	NOP 0
	NOP 0
	NOP 0
	NOP 0
	NOP 0
	NOP 0
	NOP 0
	NOP 0
	NOP 0
	NOP 0
	NOP 0
	NOP 0
	NOP 0
	NOP 0
	NOP 0
	NOP 0
	NOP 0
	NOP 0
	NOP 0
	NOP 0
	NOP 0
	NOP 0
	NOP 0
	NOP 0
	NOP 0
	NOP 0
	NOP 0
	NOP 0
	NOP 0
	NOP 0
	NOP 0
	NOP 0
	NOP 0
	NOP 0
	NOP 0
	NOP 0
	NOP 0
	NOP 0
	NOP 0
	NOP 0
	NOP 0
	NOP 0
	NOP 0
	NOP 0
	NOP 0
	NOP 0
	NOP 0
	NOP 0
	NOP 0
	NOP 0
	NOP 0
	NOP 0
	NOP 0
	NOP 0
	NOP 0
	NOP 0
	NOP 0
	NOP 0
	NOP 0
	NOP 0
	NOP 0
	NOP 0
	NOP 0
	NOP 0
	NOP 0
	NOP 0
	NOP 0
	NOP 0
	NOP 0
	NOP 0
	NOP 0
	NOP 0
	NOP 0
	NOP 0
	NOP 0
	NOP 0
	NOP 0
	NOP 0
	NOP 0
	NOP 0
	NOP 0
	NOP 0
	NOP 0
	NOP 0
	NOP 0
	NOP 0
	NOP 0
	NOP 0
	NOP 0
	NOP 0
	NOP 0
	NOP 0
	NOP 0
	NOP 0
	NOP 0
	NOP 0
	NOP 0
	NOP 0
	NOP 0
	NOP 0
	NOP 0
	NOP 0
	NOP 0
	NOP 0
	NOP 0
	NOP 0
	NOP 0
	NOP 0
	NOP 0
	NOP 0
	NOP 0
	NOP 0
	NOP 0
	NOP 0
	NOP 0
	NOP 0
	NOP 0
	NOP 0
	NOP 0
	NOP 0
	NOP 0
	NOP 0
	NOP 0
	NOP 0
	NOP 0
	NOP 0
	NOP 0
	NOP 0
	NOP 0
	NOP 0
	NOP 0
	NOP 0
	NOP 0
	NOP 0
	NOP 0
	NOP 0
	NOP 0
	NOP 0
	NOP 0
	NOP 0
	NOP 0
	NOP 0
	NOP 0
	NOP 0
	NOP 0
	NOP 0
	NOP 0
	NOP 0
	NOP 0
	NOP 0
	NOP 0
	NOP 0
	NOP 0
	NOP 0
	NOP 0
	NOP 0
	NOP 0
	NOP 0
	NOP 0
	NOP 0
	NOP 0
	NOP 0
	NOP 0
	NOP 0
	NOP 0
	NOP 0
	NOP 0
	NOP 0
	NOP 0
	NOP 0
	NOP 0
	NOP 0
	NOP 0
	NOP 0
	NOP 0
	NOP 0
	NOP 0
	NOP 0
	NOP 0
	NOP 0
	NOP 0
	NOP 0
	NOP 0
	NOP 0
	NOP 0
	NOP 0
	NOP 0
	NOP 0
	NOP 0
	NOP 0
	NOP 0
	NOP 0
	NOP 0
	NOP 0
	NOP 0
	NOP 0
	NOP 0
	NOP 0
	NOP 0
	NOP 0
	NOP 0
	NOP 0
	NOP 0
	NOP 0
	NOP 0
	NOP 0
	NOP 0
	NOP 0
	NOP 0
	NOP 0
	NOP 0
	NOP 0
	NOP 0
	NOP 0
	NOP 0
	NOP 0
	NOP 0
	NOP 0
	NOP 0
	NOP 0
	NOP 0
	NOP 0
	NOP 0
	NOP 0
	NOP 0
	NOP 0
	NOP 0
	NOP 0
	NOP 0
	NOP 0
	NOP 0
	NOP 0
	NOP 0
	NOP 0
	NOP 0
	NOP 0
	NOP 0
	NOP 0
	NOP 0
	NOP 0
	NOP 0
	NOP 0
	NOP 0
	NOP 0
	NOP 0
	NOP 0
	NOP 0
	NOP 0
	NOP 0
	NOP 0
	NOP 0
	NOP 0
	NOP 0
	NOP 0
	NOP 0
	NOP 0
	NOP 0
	NOP 0
	NOP 0
	NOP 0
	NOP 0
	NOP 0
	NOP 0
	NOP 0
	NOP 0
	NOP 0
	NOP 0
	NOP 0
	NOP 0
	NOP 0
	NOP 0
	NOP 0
	NOP 0
	NOP 0
	NOP 0
	NOP 0
	NOP 0
	NOP 0
	NOP 0
	NOP 0
	NOP 0
	NOP 0
	NOP 0
	NOP 0
	NOP 0
	NOP 0
	NOP 0
	NOP 0
	NOP 0
	NOP 0
	NOP 0
	NOP 0
	NOP 0
	NOP 0
	NOP 0
	NOP 0
	NOP 0
	NOP 0
	NOP 0
	NOP 0
	NOP 0
	NOP 0
	NOP 0
	NOP 0
	NOP 0
	NOP 0
	NOP 0
	NOP 0
	NOP 0
	NOP 0
	NOP 0
	NOP 0
	NOP 0
	NOP 0
	NOP 0
	NOP 0
	NOP 0
	NOP 0
	NOP 0
	NOP 0
	NOP 0
	NOP 0
	NOP 0
	NOP 0
	NOP 0
	NOP 0
	NOP 0
	NOP 0
	NOP 0
	NOP 0
	NOP 0
	NOP 0
	NOP 0
	NOP 0
	NOP 0
	NOP 0
	NOP 0
	NOP 0
	NOP 0
	NOP 0
	NOP 0
	NOP 0
	NOP 0
	NOP 0
	NOP 0
	NOP 0
	NOP 0
	NOP 0
	NOP 0
	NOP 0
	NOP 0
	NOP 0
	NOP 0
	NOP 0
	NOP 0
	NOP 0
	NOP 0
	NOP 0
	NOP 0
	NOP 0
	NOP 0
	NOP 0
	NOP 0
	NOP 0
	NOP 0
	NOP 0
	NOP 0
	NOP 0
	NOP 0
	NOP 0
	NOP 0
	NOP 0
	NOP 0
	NOP 0
	NOP 0
	NOP 0
	NOP 0
	NOP 0
	NOP 0
	NOP 0
	NOP 0
	NOP 0
	NOP 0
	NOP 0
	NOP 0
	NOP 0
	NOP 0
	NOP 0
	NOP 0
	NOP 0
	NOP 0
	NOP 0
	NOP 0
	NOP 0
	NOP 0
	NOP 0
	NOP 0
	NOP 0
	NOP 0
	NOP 0
	NOP 0
	NOP 0
	NOP 0
	NOP 0
	NOP 0
	NOP 0
	NOP 0
	NOP 0
	NOP 0
	NOP 0
	NOP 0
	NOP 0
	NOP 0
	NOP 0
	NOP 0
	NOP 0
	NOP 0
	NOP 0
	NOP 0
	NOP 0
	NOP 0
	NOP 0
	NOP 0
	NOP 0
	NOP 0
	NOP 0
	NOP 0
	NOP 0
	NOP 0
	NOP 0
	NOP 0
	NOP 0
	NOP 0
	NOP 0
	NOP 0
	NOP 0
	NOP 0
	NOP 0
	NOP 0
	NOP 0
	NOP 0
	NOP 0
	NOP 0
	NOP 0
	NOP 0
	NOP 0
	NOP 0
	NOP 0
	NOP 0
	NOP 0
	NOP 0
	NOP 0
	NOP 0
	NOP 0
	NOP 0
	NOP 0
	NOP 0
	NOP 0
	NOP 0
	NOP 0
	NOP 0
	NOP 0
	NOP 0
	NOP 0
	NOP 0
	NOP 0
	NOP 0
	NOP 0
	NOP 0
	NOP 0
	NOP 0
	NOP 0
	NOP 0
	NOP 0
	NOP 0
	NOP 0
	NOP 0
	NOP 0
	NOP 0
	NOP 0
	NOP 0
	NOP 0
	NOP 0
	NOP 0
	NOP 0
	NOP 0
	NOP 0
	NOP 0
	NOP 0
	NOP 0
	NOP 0
	NOP 0
	NOP 0
	NOP 0
	NOP 0
	NOP 0
	NOP 0
	NOP 0
	NOP 0
	NOP 0
	NOP 0
	NOP 0
	NOP 0
	NOP 0
	NOP 0
	NOP 0
	NOP 0
	NOP 0
	NOP 0
	NOP 0
	NOP 0
	NOP 0
	NOP 0
	NOP 0
	NOP 0
	NOP 0
	NOP 0
	NOP 0
	NOP 0
	NOP 0
	NOP 0
	NOP 0
	NOP 0
	NOP 0
	NOP 0
	NOP 0
	NOP 0
	NOP 0
	NOP 0
	NOP 0
	NOP 0
	NOP 0
	NOP 0
	NOP 0
	NOP 0
	NOP 0
	NOP 0
	NOP 0
	NOP 0
	NOP 0
	NOP 0
	NOP 0
	NOP 0
	NOP 0
	NOP 0
	NOP 0
	NOP 0
	NOP 0
	NOP 0
	NOP 0
	NOP 0
	NOP 0
	NOP 0
	NOP 0
	NOP 0
	NOP 0
	NOP 0
	NOP 0
	NOP 0
	NOP 0
	NOP 0
	NOP 0
	NOP 0
	NOP 0
	NOP 0
	NOP 0
	NOP 0
	NOP 0
	NOP 0
	NOP 0
	NOP 0
	NOP 0
	NOP 0
	NOP 0
	NOP 0
	NOP 0
	NOP 0
	NOP 0
	NOP 0
	NOP 0
	NOP 0
	NOP 0
	NOP 0
	NOP 0
	NOP 0
	NOP 0
	NOP 0
	NOP 0
	NOP 0
	NOP 0
	NOP 0
	NOP 0
	NOP 0
	NOP 0
	NOP 0
	NOP 0
	NOP 0
	NOP 0
	NOP 0
	NOP 0
	NOP 0
	NOP 0
	NOP 0
	NOP 0
	NOP 0
	NOP 0
	NOP 0
	NOP 0
	NOP 0
	NOP 0
	NOP 0
	NOP 0
	NOP 0
	NOP 0
	NOP 0
	NOP 0
	NOP 0
	NOP 0
	NOP 0
	NOP 0
	NOP 0
	NOP 0
	NOP 0
	NOP 0
	NOP 0
	NOP 0
	NOP 0
	NOP 0
	NOP 0
	NOP 0
	NOP 0
	NOP 0
	NOP 0
	NOP 0
	NOP 0
	NOP 0
	NOP 0
	NOP 0
	NOP 0
	NOP 0
	NOP 0
	NOP 0
	NOP 0
	NOP 0
	NOP 0
	NOP 0
	NOP 0
	NOP 0
	NOP 0
	NOP 0
	NOP 0
	NOP 0
	NOP 0
	NOP 0
	NOP 0
	NOP 0
	NOP 0
	NOP 0
	NOP 0
	NOP 0
	NOP 0
	NOP 0
	NOP 0
	NOP 0
	NOP 0
	NOP 0
	NOP 0
	NOP 0
	NOP 0
	NOP 0
	NOP 0
	NOP 0
	NOP 0
	NOP 0
	NOP 0
	NOP 0
	NOP 0
	NOP 0
	NOP 0
	NOP 0
	NOP 0
	NOP 0
	NOP 0
	NOP 0
	NOP 0
	NOP 0
	NOP 0
	NOP 0
	NOP 0
	NOP 0
	NOP 0
	NOP 0
	NOP 0
	NOP 0
	NOP 0
	NOP 0
	NOP 0
	NOP 0
	NOP 0
	NOP 0
	NOP 0
	NOP 0
	NOP 0
	NOP 0
	NOP 0
	NOP 0
	NOP 0
	NOP 0
	NOP 0
	NOP 0
	NOP 0
	NOP 0
	NOP 0
	NOP 0
	NOP 0
	NOP 0
	NOP 0
	NOP 0
	NOP 0
	NOP 0
	NOP 0
	NOP 0
	NOP 0
	NOP 0
	NOP 0
	NOP 0
	NOP 0
	NOP 0
	NOP 0
	NOP 0
	NOP 0
	NOP 0
	NOP 0
	NOP 0
	NOP 0
	NOP 0
	NOP 0
	NOP 0
	NOP 0
	NOP 0
	NOP 0
	NOP 0
	NOP 0
	NOP 0
	NOP 0
	NOP 0
	NOP 0
	NOP 0
	NOP 0
	NOP 0
	NOP 0
	NOP 0
	NOP 0
	NOP 0
	NOP 0
	NOP 0
	NOP 0
	NOP 0
	NOP 0
	NOP 0
	NOP 0
	NOP 0
	NOP 0
	NOP 0
	NOP 0
	NOP 0
	NOP 0
	NOP 0
	NOP 0
	NOP 0
	NOP 0
	NOP 0
	NOP 0
	NOP 0
	NOP 0
	NOP 0
	NOP 0
	NOP 0
	NOP 0
	NOP 0
	NOP 0
	NOP 0
	NOP 0
	NOP 0
	NOP 0
	NOP 0
	NOP 0
	NOP 0
	NOP 0
	NOP 0
	NOP 0
	NOP 0
	NOP 0
	NOP 0
	NOP 0
	NOP 0
	NOP 0
	NOP 0
	NOP 0
	NOP 0
	NOP 0
	NOP 0
	NOP 0
	NOP 0
	NOP 0
	NOP 0
	NOP 0
	NOP 0
	NOP 0
	NOP 0
	NOP 0
	NOP 0
	NOP 0
	NOP 0
	NOP 0
	NOP 0
	NOP 0
	NOP 0
	NOP 0
	NOP 0
	NOP 0
	NOP 0
	NOP 0
	NOP 0
	NOP 0
	NOP 0
	NOP 0
	NOP 0
	NOP 0
	NOP 0
	NOP 0
	NOP 0
	NOP 0
	NOP 0
	NOP 0
	NOP 0
	NOP 0
	NOP 0
	NOP 0
	NOP 0
	NOP 0
	NOP 0
	NOP 0
	NOP 0
	NOP 0
	NOP 0
	NOP 0
	NOP 0
	NOP 0
	NOP 0
	NOP 0
	NOP 0
	NOP 0
	NOP 0
	NOP 0
	NOP 0
	NOP 0
	NOP 0
	NOP 0
	NOP 0
	NOP 0
	NOP 0
	NOP 0
	NOP 0
	NOP 0
	NOP 0
	NOP 0
	NOP 0
	NOP 0
	NOP 0
	NOP 0
	NOP 0
	NOP 0
	NOP 0
	NOP 0
	NOP 0
	NOP 0
	NOP 0
	NOP 0
	NOP 0
	NOP 0
	NOP 0
	NOP 0
	NOP 0
	NOP 0
	NOP 0
	NOP 0
	NOP 0
	NOP 0
	NOP 0
	NOP 0
	NOP 0
	NOP 0
	NOP 0
	NOP 0
	NOP 0
	NOP 0
	NOP 0
	NOP 0
	NOP 0
	NOP 0
	NOP 0
	NOP 0
	NOP 0
	NOP 0
	NOP 0
	NOP 0
	NOP 0
	NOP 0
	NOP 0
	NOP 0
	NOP 0
	NOP 0
	NOP 0
	NOP 0
	NOP 0
	NOP 0
	NOP 0
	NOP 0
	NOP 0
	NOP 0
	NOP 0
	NOP 0
	NOP 0
	NOP 0
	NOP 0
	NOP 0
	NOP 0
	NOP 0
	NOP 0
	NOP 0
	NOP 0
	NOP 0
	NOP 0
	NOP 0
	NOP 0
	NOP 0
	NOP 0
	NOP 0
	NOP 0
	NOP 0
	NOP 0
	NOP 0
	NOP 0
	NOP 0
	NOP 0
	NOP 0
	NOP 0
	NOP 0
	NOP 0
	NOP 0
	NOP 0
	NOP 0
	NOP 0
	NOP 0
	NOP 0
	NOP 0
	NOP 0
	NOP 0
	NOP 0
	NOP 0
	NOP 0
	NOP 0
	NOP 0
	NOP 0
	NOP 0
	NOP 0
	NOP 0
	NOP 0
	NOP 0
	NOP 0
	NOP 0
	NOP 0
	NOP 0
	NOP 0
	NOP 0
	NOP 0
	NOP 0
	NOP 0
	NOP 0
	NOP 0
	NOP 0
	NOP 0
	NOP 0
	NOP 0
	NOP 0
	NOP 0
	NOP 0
	NOP 0
	NOP 0
	NOP 0
	NOP 0
	NOP 0
	NOP 0
	NOP 0
	NOP 0
	NOP 0
	NOP 0
	NOP 0
	NOP 0
	NOP 0
	NOP 0
	NOP 0
	NOP 0
	NOP 0
	NOP 0
	NOP 0
	NOP 0
	NOP 0
	NOP 0
	NOP 0
	NOP 0
	NOP 0
	NOP 0
	NOP 0
	NOP 0
	NOP 0
	NOP 0
	NOP 0
	NOP 0
	NOP 0
	NOP 0
	NOP 0
	NOP 0
	NOP 0
	NOP 0
	NOP 0
	NOP 0
	NOP 0
	NOP 0
	NOP 0
	NOP 0
	NOP 0
	NOP 0
	NOP 0
	NOP 0
	NOP 0
	NOP 0
	NOP 0
	NOP 0
	NOP 0
	NOP 0
	NOP 0
	NOP 0
	NOP 0
	NOP 0
	NOP 0
	NOP 0
	NOP 0
	NOP 0
	NOP 0
	NOP 0
	NOP 0
	NOP 0
	NOP 0
	NOP 0
	NOP 0
	NOP 0
	NOP 0
	NOP 0
	NOP 0
	NOP 0
	NOP 0
	NOP 0
	NOP 0
	NOP 0
	NOP 0
	NOP 0
	NOP 0
	NOP 0
	NOP 0
	NOP 0
	NOP 0
	NOP 0
	NOP 0
	NOP 0
	NOP 0
	NOP 0
	NOP 0
	NOP 0
	NOP 0
	NOP 0
	NOP 0
	NOP 0
	NOP 0
	NOP 0
	NOP 0
	NOP 0
	NOP 0
	NOP 0
	NOP 0
	NOP 0
	NOP 0
	NOP 0
	NOP 0
	NOP 0
	NOP 0
	NOP 0
	NOP 0
	NOP 0
	NOP 0
	NOP 0
	NOP 0
	NOP 0
	NOP 0
	NOP 0
	NOP 0
	NOP 0
	NOP 0
	NOP 0
	NOP 0
	NOP 0
	NOP 0
	NOP 0
	NOP 0
	NOP 0
	NOP 0
	NOP 0
	NOP 0
	NOP 0
	NOP 0
	NOP 0
	NOP 0
	NOP 0
	NOP 0
	NOP 0
	NOP 0
	NOP 0
	NOP 0
	NOP 0
	NOP 0
	NOP 0
	NOP 0
	NOP 0
	NOP 0
	NOP 0
	NOP 0
	NOP 0
	NOP 0
	NOP 0
	NOP 0
	NOP 0
	NOP 0
	NOP 0
	NOP 0
	NOP 0
	NOP 0
	NOP 0
	NOP 0
	NOP 0
	NOP 0
	NOP 0
	NOP 0
	NOP 0
	NOP 0
	NOP 0
	NOP 0
	NOP 0
	NOP 0
	NOP 0
	NOP 0
	NOP 0
	NOP 0
	NOP 0
	NOP 0
	NOP 0
	NOP 0
	NOP 0
	NOP 0
	NOP 0
	NOP 0
	NOP 0
	NOP 0
	NOP 0
	NOP 0
	NOP 0
	NOP 0
	NOP 0
	NOP 0
	NOP 0
	NOP 0
	NOP 0
	NOP 0
	NOP 0
	NOP 0
	NOP 0
	NOP 0
	NOP 0
	NOP 0
	NOP 0
	NOP 0
	NOP 0
	NOP 0
	NOP 0
	NOP 0
	NOP 0
	NOP 0
	NOP 0
	NOP 0
	NOP 0
	NOP 0
	NOP 0
	NOP 0
	NOP 0
	NOP 0
	NOP 0
	NOP 0
	NOP 0
	NOP 0
	NOP 0
	NOP 0
	NOP 0
	NOP 0
	NOP 0
	NOP 0
	NOP 0
	NOP 0
	NOP 0
	NOP 0
	NOP 0
	NOP 0
	NOP 0
	NOP 0
	NOP 0
	NOP 0
	NOP 0
	NOP 0
	NOP 0
	NOP 0
	NOP 0
	NOP 0
	NOP 0
	NOP 0
	NOP 0
	NOP 0
	NOP 0
	NOP 0
	NOP 0
	NOP 0
	NOP 0
	NOP 0
	NOP 0
	NOP 0
	NOP 0
	NOP 0
	NOP 0
	NOP 0
	NOP 0
	NOP 0
	NOP 0
	NOP 0
	NOP 0
	NOP 0
	NOP 0
	NOP 0
	NOP 0
	NOP 0
	NOP 0
	NOP 0
	NOP 0
	NOP 0
	NOP 0
	NOP 0
	NOP 0
	NOP 0
	NOP 0
	NOP 0
	NOP 0
	NOP 0
	NOP 0
	NOP 0
	NOP 0
	NOP 0
	NOP 0
	NOP 0
	NOP 0
	NOP 0
	NOP 0
	NOP 0
	NOP 0
	NOP 0
	NOP 0
	NOP 0
	NOP 0
	NOP 0
	NOP 0
	NOP 0
	NOP 0
	NOP 0
	NOP 0
	NOP 0
	NOP 0
	NOP 0
	NOP 0
	NOP 0
	NOP 0
	NOP 0
	NOP 0
	NOP 0
	NOP 0
	NOP 0
	NOP 0
	NOP 0
	NOP 0
	NOP 0
	NOP 0
	NOP 0
	NOP 0
	NOP 0
	NOP 0
	NOP 0
	NOP 0
	NOP 0
	NOP 0
	NOP 0
	NOP 0
	NOP 0
	NOP 0
	NOP 0
	NOP 0
	NOP 0
	NOP 0
	NOP 0
	NOP 0
	NOP 0
	NOP 0
	NOP 0
	NOP 0
	NOP 0
	NOP 0
	NOP 0
	NOP 0
	NOP 0
	NOP 0
	NOP 0
	NOP 0
	NOP 0
	NOP 0
	NOP 0
	NOP 0
	NOP 0
	NOP 0
	NOP 0
	NOP 0
	NOP 0
	NOP 0
	NOP 0
	NOP 0
	NOP 0
	NOP 0
	NOP 0
	NOP 0
	NOP 0
	NOP 0
	NOP 0
	NOP 0
	NOP 0
	NOP 0
	NOP 0
	NOP 0
	NOP 0
	NOP 0
	NOP 0
	NOP 0
	NOP 0
	NOP 0
	NOP 0
	NOP 0
	NOP 0
	NOP 0
	NOP 0
	NOP 0
	NOP 0
	NOP 0
	NOP 0
	NOP 0
	NOP 0
	NOP 0
	NOP 0
	NOP 0
	NOP 0
	NOP 0
	NOP 0
	NOP 0
	NOP 0
	NOP 0
	NOP 0
	NOP 0
	NOP 0
	NOP 0
	NOP 0
	NOP 0
	NOP 0
	NOP 0
	NOP 0
	NOP 0
	NOP 0
	NOP 0
	NOP 0
	NOP 0
	NOP 0
	NOP 0
	NOP 0
	NOP 0
	NOP 0
	NOP 0
	NOP 0
	NOP 0
	NOP 0
	NOP 0
	NOP 0
	NOP 0
	NOP 0
	NOP 0
	NOP 0
	NOP 0
	NOP 0
	NOP 0
	NOP 0
	NOP 0
	NOP 0
	NOP 0
	NOP 0
	NOP 0
	NOP 0
	NOP 0
	NOP 0
	NOP 0
	NOP 0
	NOP 0
	NOP 0
	NOP 0
	NOP 0
	NOP 0
	NOP 0
	NOP 0
	NOP 0
	NOP 0
	NOP 0
	NOP 0
	NOP 0
	NOP 0
	NOP 0
	NOP 0
	NOP 0
	NOP 0
	NOP 0
	NOP 0
	NOP 0
	NOP 0
	NOP 0
	NOP 0
	NOP 0
	NOP 0
	NOP 0
	NOP 0
	NOP 0
	NOP 0
	NOP 0
	NOP 0
	NOP 0
	NOP 0
	NOP 0
	NOP 0
	NOP 0
	NOP 0
	NOP 0
	NOP 0
	NOP 0
	NOP 0
	NOP 0
	NOP 0
	NOP 0
	NOP 0
	NOP 0
	NOP 0
	NOP 0
	NOP 0
	NOP 0
	NOP 0
	NOP 0
	NOP 0
	NOP 0
	NOP 0
	NOP 0
	NOP 0
	NOP 0
	NOP 0
	NOP 0
	NOP 0
	NOP 0
	NOP 0
	NOP 0
	NOP 0
	NOP 0
	NOP 0
	NOP 0
	NOP 0
	NOP 0
	NOP 0
	NOP 0
	NOP 0
	NOP 0
	NOP 0
	NOP 0
	NOP 0
	NOP 0
	NOP 0
	NOP 0
	NOP 0
	NOP 0
	NOP 0
	NOP 0
	NOP 0
	NOP 0
	NOP 0
	NOP 0
	NOP 0
	NOP 0
	NOP 0
	NOP 0
	NOP 0
	NOP 0
	NOP 0
	NOP 0
	NOP 0
	NOP 0
	NOP 0
	NOP 0
	NOP 0
	NOP 0
	NOP 0
	NOP 0
	NOP 0
	NOP 0
	NOP 0
	NOP 0
	NOP 0
	NOP 0
	NOP 0
	NOP 0
	NOP 0
	NOP 0
	NOP 0
	NOP 0
	NOP 0
	NOP 0
	NOP 0
	NOP 0
	NOP 0
	NOP 0
	NOP 0
	NOP 0
	NOP 0
	NOP 0
	NOP 0
	NOP 0
	NOP 0
	NOP 0
	NOP 0
	NOP 0
	NOP 0
	NOP 0
	NOP 0
	NOP 0
	NOP 0
	NOP 0
	NOP 0
	NOP 0
	NOP 0
	NOP 0
	NOP 0
	NOP 0
	NOP 0
	NOP 0
	NOP 0
	NOP 0
	NOP 0
	NOP 0
	NOP 0
	NOP 0
	NOP 0
	NOP 0
	NOP 0
	NOP 0
	NOP 0
	NOP 0
	NOP 0
	NOP 0
	NOP 0
	NOP 0
	NOP 0
	NOP 0
	NOP 0
	NOP 0
	NOP 0
	NOP 0
	NOP 0
	NOP 0
	NOP 0
	NOP 0
	NOP 0
	NOP 0
	NOP 0
	NOP 0
	NOP 0
	NOP 0
	NOP 0
	NOP 0
	NOP 0
	NOP 0
	NOP 0
	NOP 0
	NOP 0
	NOP 0
	NOP 0
	NOP 0
	NOP 0
	NOP 0
	NOP 0
	NOP 0
	NOP 0
	NOP 0
	NOP 0
	NOP 0
	NOP 0
	NOP 0
	NOP 0
	NOP 0
	NOP 0
	NOP 0
	NOP 0
	NOP 0
	NOP 0
	NOP 0
	NOP 0
	NOP 0
	NOP 0
	NOP 0
	NOP 0
	NOP 0
	NOP 0
	NOP 0
	NOP 0
	NOP 0
	NOP 0
	NOP 0
	NOP 0
	NOP 0
	NOP 0
	NOP 0
	NOP 0
	NOP 0
	NOP 0
	NOP 0
	NOP 0
	NOP 0
	NOP 0
	NOP 0
	NOP 0
	NOP 0
	NOP 0
	NOP 0
	NOP 0
	NOP 0
	NOP 0
	NOP 0
	NOP 0
	NOP 0
	NOP 0
	NOP 0
	NOP 0
	NOP 0
	NOP 0
	NOP 0
	NOP 0
	NOP 0
	NOP 0
	NOP 0
	NOP 0
	NOP 0
	NOP 0
	NOP 0
	NOP 0
	NOP 0
	NOP 0
	NOP 0
	NOP 0
	NOP 0
	NOP 0
	NOP 0
	NOP 0
	NOP 0
	NOP 0
	NOP 0
	NOP 0
	NOP 0
	NOP 0
	NOP 0
	NOP 0
	NOP 0
	NOP 0
	NOP 0
	NOP 0
	NOP 0
	NOP 0
	NOP 0
	NOP 0
	NOP 0
	NOP 0
	NOP 0
	NOP 0
	NOP 0
	NOP 0
	NOP 0
	NOP 0
	NOP 0
	NOP 0
	NOP 0
	NOP 0
	NOP 0
	NOP 0
	NOP 0
	NOP 0
	NOP 0
	NOP 0
	NOP 0
	NOP 0
	NOP 0
	NOP 0
	NOP 0
	NOP 0
	NOP 0
	NOP 0
	NOP 0
	NOP 0
	NOP 0
	NOP 0
	NOP 0
	NOP 0
	NOP 0
	NOP 0
	NOP 0
	NOP 0
	NOP 0
	NOP 0
	NOP 0
	NOP 0
	NOP 0
	NOP 0
	NOP 0
	NOP 0
	NOP 0
	NOP 0
	NOP 0
	NOP 0
	NOP 0
	NOP 0
	NOP 0
	NOP 0
	NOP 0
	NOP 0
	NOP 0
	NOP 0
	NOP 0
	NOP 0
	NOP 0
	NOP 0
	NOP 0
	NOP 0
	NOP 0
	NOP 0
	NOP 0
	NOP 0
	NOP 0
	NOP 0
	NOP 0
	NOP 0
	NOP 0
	NOP 0
	NOP 0
	NOP 0
	NOP 0
	NOP 0
	NOP 0
	NOP 0
	NOP 0
	NOP 0
	NOP 0
	NOP 0
	NOP 0
	NOP 0
	NOP 0
	NOP 0
	NOP 0
	NOP 0
	NOP 0
	NOP 0
	NOP 0
	NOP 0
	NOP 0
	NOP 0
	NOP 0
	NOP 0
	NOP 0
	NOP 0
	NOP 0
	NOP 0
	NOP 0
	NOP 0
	NOP 0
	NOP 0
	NOP 0
	NOP 0
	NOP 0
	NOP 0
	NOP 0
	NOP 0
	NOP 0
	NOP 0
	NOP 0
	NOP 0
	NOP 0
	NOP 0
	NOP 0
	NOP 0
	NOP 0
	NOP 0
	NOP 0
	NOP 0
	NOP 0
	NOP 0
	NOP 0
	NOP 0
	NOP 0
	NOP 0
	NOP 0
	NOP 0
	NOP 0
	NOP 0
	NOP 0
	NOP 0
	NOP 0
	NOP 0
	NOP 0
	NOP 0
	NOP 0
	NOP 0
	NOP 0
	NOP 0
	NOP 0
	NOP 0
	NOP 0
	NOP 0
	NOP 0
	NOP 0
	NOP 0
	NOP 0
	NOP 0
	NOP 0
	NOP 0
	NOP 0
	NOP 0
	NOP 0
	NOP 0
	NOP 0
	NOP 0
	NOP 0
	NOP 0
	NOP 0
	NOP 0
	NOP 0
	NOP 0
	NOP 0
	NOP 0
	NOP 0
	NOP 0
	NOP 0
	NOP 0
	NOP 0
	NOP 0
	NOP 0
	NOP 0
	NOP 0
	NOP 0
	NOP 0
	NOP 0
	NOP 0
	NOP 0
	NOP 0
	NOP 0
	NOP 0
	NOP 0
	NOP 0
	NOP 0
	NOP 0
	NOP 0
	NOP 0
	NOP 0
	NOP 0
	NOP 0
	NOP 0
	NOP 0
	NOP 0
	NOP 0
	NOP 0
	NOP 0
	NOP 0
	NOP 0
	NOP 0
	NOP 0
	NOP 0
	NOP 0
	NOP 0
	NOP 0
	NOP 0
	NOP 0
	NOP 0
	NOP 0
	NOP 0
	NOP 0
	NOP 0
	NOP 0
	NOP 0
	NOP 0
	NOP 0
	NOP 0
	NOP 0
	NOP 0
	NOP 0
	NOP 0
	NOP 0
	NOP 0
	NOP 0
	NOP 0
	NOP 0
	NOP 0
	NOP 0
	NOP 0
	NOP 0
	NOP 0
	NOP 0
	NOP 0
	NOP 0
	NOP 0
	NOP 0
	NOP 0
	NOP 0
	NOP 0
	NOP 0
	NOP 0
	NOP 0
	NOP 0
	NOP 0
	NOP 0
	NOP 0
	NOP 0
	NOP 0
	NOP 0
	NOP 0
	NOP 0
	NOP 0
	NOP 0
	NOP 0
	NOP 0
	NOP 0
	NOP 0
	NOP 0
	NOP 0
	NOP 0
	NOP 0
	NOP 0
	NOP 0
	NOP 0
	NOP 0
	NOP 0
	NOP 0
	NOP 0
	NOP 0
	NOP 0
	NOP 0
	NOP 0
	NOP 0
	NOP 0
	NOP 0
	NOP 0
	NOP 0
	NOP 0
	NOP 0
	NOP 0
	NOP 0
	NOP 0
	NOP 0
	NOP 0
	NOP 0
	NOP 0
	NOP 0
	NOP 0
	NOP 0
	NOP 0
	NOP 0
	NOP 0
	NOP 0
	NOP 0
	NOP 0
	NOP 0
	NOP 0
	NOP 0
	NOP 0
	NOP 0
	NOP 0
	NOP 0
	NOP 0
	NOP 0
	NOP 0
	NOP 0
	NOP 0
	NOP 0
	NOP 0
	NOP 0
	NOP 0
	NOP 0
	NOP 0
	NOP 0
	NOP 0
	NOP 0
	NOP 0
	NOP 0
	NOP 0
	NOP 0
	NOP 0
	NOP 0
	NOP 0
	NOP 0
	NOP 0
	NOP 0
	NOP 0
	NOP 0
	NOP 0
	NOP 0
	NOP 0
	NOP 0
	NOP 0
	NOP 0
	NOP 0
	NOP 0
	NOP 0
	NOP 0
	NOP 0
	NOP 0
	NOP 0
	NOP 0
	NOP 0
	NOP 0
	NOP 0
	NOP 0
	NOP 0
	NOP 0
	NOP 0
	NOP 0
	NOP 0
	NOP 0
	NOP 0
	NOP 0
	NOP 0
	NOP 0
	NOP 0
	NOP 0
	NOP 0
	NOP 0
	NOP 0
	NOP 0
	NOP 0
	NOP 0
	NOP 0
	NOP 0
	NOP 0
	NOP 0
	NOP 0
	NOP 0
	NOP 0
	NOP 0
	NOP 0
	NOP 0
	NOP 0
	NOP 0
	NOP 0
	NOP 0
	NOP 0
	NOP 0
	NOP 0
	NOP 0
	NOP 0
	NOP 0
	NOP 0
	NOP 0
	NOP 0
	NOP 0
	NOP 0
	NOP 0
	NOP 0
	NOP 0
	NOP 0
	NOP 0
	NOP 0
	NOP 0
	NOP 0
	NOP 0
	NOP 0
	NOP 0
	NOP 0
	NOP 0
	NOP 0
	NOP 0
	NOP 0
	NOP 0
	NOP 0
	NOP 0
	NOP 0
	NOP 0
	NOP 0
	NOP 0
	NOP 0
	NOP 0
	NOP 0
	NOP 0
	NOP 0
	NOP 0
	NOP 0
	NOP 0
	NOP 0
	NOP 0
	NOP 0
	NOP 0
	NOP 0
	NOP 0
	NOP 0
	NOP 0
	NOP 0
	NOP 0
	NOP 0
	NOP 0
	NOP 0
	NOP 0
	NOP 0
	NOP 0
	NOP 0
	NOP 0
	NOP 0
	NOP 0
	NOP 0
	NOP 0
	NOP 0
	NOP 0
	NOP 0
	NOP 0
	NOP 0
	NOP 0
	NOP 0
	NOP 0
	NOP 0
	NOP 0
	NOP 0
	NOP 0
	NOP 0
	NOP 0
	NOP 0
	NOP 0
	NOP 0
	NOP 0
	NOP 0
	NOP 0
	NOP 0
	NOP 0
	NOP 0
	NOP 0
	NOP 0
	NOP 0
	NOP 0
	NOP 0
	NOP 0
	NOP 0
	NOP 0
	NOP 0
	NOP 0
	NOP 0
	NOP 0
	NOP 0
	NOP 0
	NOP 0
	NOP 0
	NOP 0
	NOP 0
	NOP 0
	NOP 0
	NOP 0
	NOP 0
	NOP 0
	NOP 0
	NOP 0
	NOP 0
	NOP 0
	NOP 0
	NOP 0
	NOP 0
	NOP 0
	NOP 0
	NOP 0
	NOP 0
	NOP 0
	NOP 0
	NOP 0
	NOP 0
	NOP 0
	NOP 0
	NOP 0
	NOP 0
	NOP 0
	NOP 0
	NOP 0
	NOP 0
	NOP 0
	NOP 0
	NOP 0
	NOP 0
	NOP 0
	NOP 0
	NOP 0
	NOP 0
	NOP 0
	NOP 0
	NOP 0
	NOP 0
	NOP 0
	NOP 0
	NOP 0
	NOP 0
	NOP 0
	NOP 0
	NOP 0
	NOP 0
	NOP 0
	NOP 0
	NOP 0
	NOP 0
	NOP 0
	NOP 0
	NOP 0
	NOP 0
	NOP 0
	NOP 0
	NOP 0
	NOP 0
	NOP 0
	NOP 0
	NOP 0
	NOP 0
	NOP 0
	NOP 0
	NOP 0
	NOP 0
	NOP 0
	NOP 0
	NOP 0
	NOP 0
	NOP 0
	NOP 0
	NOP 0
	NOP 0
	NOP 0
	NOP 0
	NOP 0
	NOP 0
	NOP 0
	NOP 0
	NOP 0
	NOP 0
	NOP 0
	NOP 0
	NOP 0
	NOP 0
	NOP 0
	NOP 0
	NOP 0
	NOP 0
	NOP 0
	NOP 0
	NOP 0
	NOP 0
	NOP 0
	NOP 0
	NOP 0
	NOP 0
	NOP 0
	NOP 0
	NOP 0
	NOP 0
	NOP 0
	NOP 0
	NOP 0
	NOP 0
	NOP 0
	NOP 0
	NOP 0
	NOP 0
	NOP 0
	NOP 0
	NOP 0
	NOP 0
	NOP 0
	NOP 0
	NOP 0
	NOP 0
	NOP 0
	NOP 0
	NOP 0
	NOP 0
	NOP 0
	NOP 0
	NOP 0
	NOP 0
	NOP 0
	NOP 0
	NOP 0
	NOP 0
	NOP 0
	NOP 0
	NOP 0
	NOP 0
	NOP 0
	NOP 0
	NOP 0
	NOP 0
	NOP 0
	NOP 0
	NOP 0
	NOP 0
	NOP 0
	NOP 0
	NOP 0
	NOP 0
	NOP 0
	NOP 0
	NOP 0
	NOP 0
	NOP 0
	NOP 0
	NOP 0
	NOP 0
	NOP 0
	NOP 0
	NOP 0
	NOP 0
	NOP 0
	NOP 0
	NOP 0
	NOP 0
	NOP 0
	NOP 0
	NOP 0
	NOP 0
	NOP 0
	NOP 0
	NOP 0
	NOP 0
	NOP 0
	NOP 0
	NOP 0
	NOP 0
	NOP 0
	NOP 0
	NOP 0
	NOP 0
	NOP 0
	NOP 0
	NOP 0
	NOP 0
	NOP 0
	NOP 0
	NOP 0
	NOP 0
	NOP 0
	NOP 0
	NOP 0
	NOP 0
	NOP 0
	NOP 0
	NOP 0
	NOP 0
	NOP 0
	NOP 0
	NOP 0
	NOP 0
	NOP 0
	NOP 0
	NOP 0
	NOP 0
	NOP 0
	NOP 0
	NOP 0
	NOP 0
	NOP 0
	NOP 0
	NOP 0
	NOP 0
	NOP 0
	NOP 0
	NOP 0
	NOP 0
	NOP 0
	NOP 0
	NOP 0
	NOP 0
	NOP 0
	NOP 0
	NOP 0
	NOP 0
	NOP 0
	NOP 0
	NOP 0
	NOP 0
	NOP 0
	NOP 0
	NOP 0
	NOP 0
	NOP 0
	NOP 0
	NOP 0
	NOP 0
	NOP 0
	NOP 0
	NOP 0
	NOP 0
	NOP 0
	NOP 0
	NOP 0
	NOP 0
	NOP 0
	NOP 0
	NOP 0
	NOP 0
	NOP 0
	NOP 0
	NOP 0
	NOP 0
	NOP 0
	NOP 0
	NOP 0
	NOP 0
	NOP 0
	NOP 0
	NOP 0
	NOP 0
	NOP 0
	NOP 0
	NOP 0
	NOP 0
	NOP 0
	NOP 0
	NOP 0
	NOP 0
	NOP 0
	NOP 0
	NOP 0
	NOP 0
	NOP 0
	NOP 0
	NOP 0
	NOP 0
	NOP 0
	NOP 0
	NOP 0
	NOP 0
	NOP 0
	NOP 0
	NOP 0
	NOP 0
	NOP 0
	NOP 0
	NOP 0
	NOP 0
	NOP 0
	NOP 0
	NOP 0
	NOP 0
	NOP 0
	NOP 0
	NOP 0
	NOP 0
	NOP 0
	NOP 0
	NOP 0
	NOP 0
	NOP 0
	NOP 0
	NOP 0
	NOP 0
	NOP 0
	NOP 0
	NOP 0
	NOP 0
	NOP 0
	NOP 0
	NOP 0
	NOP 0
	NOP 0
	NOP 0
	NOP 0
	NOP 0
	NOP 0
	NOP 0
	NOP 0
	NOP 0
	NOP 0
	NOP 0
	NOP 0
	NOP 0
	NOP 0
	NOP 0
	NOP 0
	NOP 0
	NOP 0
	NOP 0
	NOP 0
	NOP 0
	NOP 0
	NOP 0
	NOP 0
	NOP 0
	NOP 0
	NOP 0
	NOP 0
	NOP 0
	NOP 0
	NOP 0
	NOP 0
	NOP 0
	NOP 0
	NOP 0
	NOP 0
	NOP 0
	NOP 0
	NOP 0
	NOP 0
	NOP 0
	NOP 0
	NOP 0
	NOP 0
	NOP 0
	NOP 0
	NOP 0
	NOP 0
	NOP 0
	NOP 0
	NOP 0
	NOP 0
	NOP 0
	NOP 0
	NOP 0
	NOP 0
	NOP 0
	NOP 0
	NOP 0
	NOP 0
	NOP 0
	NOP 0
	NOP 0
	NOP 0
	NOP 0
	NOP 0
	NOP 0
	NOP 0
	NOP 0
	NOP 0
	NOP 0
	NOP 0
	NOP 0
	NOP 0
	NOP 0
	NOP 0
	NOP 0
	NOP 0
	NOP 0
	NOP 0
	NOP 0
	NOP 0
	NOP 0
	NOP 0
	NOP 0
	NOP 0
	NOP 0
	NOP 0
	NOP 0
	NOP 0
	NOP 0
	NOP 0
	NOP 0
	NOP 0
	NOP 0
	NOP 0
	NOP 0
	NOP 0
	NOP 0
	NOP 0
	NOP 0
	NOP 0
	NOP 0
	NOP 0
	NOP 0
	NOP 0
	NOP 0
	NOP 0
	NOP 0
	NOP 0
	NOP 0
	NOP 0
	NOP 0
	NOP 0
	NOP 0
	NOP 0
	NOP 0
	NOP 0
	NOP 0
	NOP 0
	NOP 0
	NOP 0
	NOP 0
	NOP 0
	NOP 0
	NOP 0
	NOP 0
	NOP 0
	NOP 0
	NOP 0
	NOP 0
	NOP 0
	NOP 0
	NOP 0
	NOP 0
	NOP 0
	NOP 0
	NOP 0
	NOP 0
	NOP 0
	NOP 0
	NOP 0
	NOP 0
	NOP 0
	NOP 0
	NOP 0
	NOP 0
	NOP 0
	NOP 0
	NOP 0
	NOP 0
	NOP 0
	NOP 0
	NOP 0
	NOP 0
	NOP 0
	NOP 0
	NOP 0
	NOP 0
	NOP 0
	NOP 0
	NOP 0
	NOP 0
	NOP 0
	NOP 0
	NOP 0
	NOP 0
	NOP 0
	NOP 0
	NOP 0
	NOP 0
	NOP 0
	NOP 0
	NOP 0
	NOP 0
	NOP 0
	NOP 0
	NOP 0
	NOP 0
	NOP 0
	NOP 0
	NOP 0
	NOP 0
	NOP 0
	NOP 0
	NOP 0
	NOP 0
	NOP 0
	NOP 0
	NOP 0
	NOP 0
	NOP 0
	NOP 0
	NOP 0
	NOP 0
	NOP 0
	NOP 0
	NOP 0
	NOP 0
	NOP 0
	NOP 0
	NOP 0
	NOP 0
	NOP 0
	NOP 0
	NOP 0
	NOP 0
	NOP 0
	NOP 0
	NOP 0
	NOP 0
	NOP 0
	NOP 0
	NOP 0
	NOP 0
	NOP 0
	NOP 0
	NOP 0
	NOP 0
	NOP 0
	NOP 0
	NOP 0
	NOP 0
	NOP 0
	NOP 0
	NOP 0
	NOP 0
	NOP 0
	NOP 0
	NOP 0
	NOP 0
	NOP 0
	NOP 0
	NOP 0
	NOP 0
	NOP 0
	NOP 0
	NOP 0
	NOP 0
	NOP 0
	NOP 0
	NOP 0
	NOP 0
	NOP 0
	NOP 0
	NOP 0
	NOP 0
	NOP 0
	NOP 0
	NOP 0
	NOP 0
	NOP 0
	NOP 0
	NOP 0
	NOP 0
	NOP 0
	NOP 0
	NOP 0
	NOP 0
	NOP 0
	NOP 0
	NOP 0
	NOP 0
	NOP 0
	NOP 0
	NOP 0
	NOP 0
	NOP 0
	NOP 0
	NOP 0
	NOP 0
	NOP 0
	NOP 0
	NOP 0
	NOP 0
	NOP 0
	NOP 0
	NOP 0
	NOP 0
	NOP 0
	NOP 0
	NOP 0
	NOP 0
	NOP 0
	NOP 0
	NOP 0
	NOP 0
	NOP 0
	NOP 0
	NOP 0
	NOP 0
	NOP 0
	NOP 0
	NOP 0
	NOP 0
	NOP 0
	NOP 0
	NOP 0
	NOP 0
	NOP 0
	NOP 0
	NOP 0
	NOP 0
	NOP 0
	NOP 0
	NOP 0
	NOP 0
	NOP 0
	NOP 0
	NOP 0
	NOP 0
	NOP 0
	NOP 0
	NOP 0
	NOP 0
	NOP 0
	NOP 0
	NOP 0
	NOP 0
	NOP 0
	NOP 0
	NOP 0
	NOP 0
	NOP 0
	NOP 0
	NOP 0
	NOP 0
	NOP 0
	NOP 0
	NOP 0
	NOP 0
	NOP 0
	NOP 0
	NOP 0
	NOP 0
	NOP 0
	NOP 0
	NOP 0
	NOP 0
	NOP 0
	NOP 0
	NOP 0
	NOP 0
	NOP 0
	NOP 0
	NOP 0
	NOP 0
	NOP 0
	NOP 0
	NOP 0
	NOP 0
	NOP 0
	NOP 0
	NOP 0
	NOP 0
	NOP 0
	NOP 0
	NOP 0
	NOP 0
	NOP 0
	NOP 0
	NOP 0
	NOP 0
	NOP 0
	NOP 0
	NOP 0
	NOP 0
	NOP 0
	NOP 0
	NOP 0
	NOP 0
	NOP 0
	NOP 0
	NOP 0
	NOP 0
	NOP 0
	NOP 0
	NOP 0
	NOP 0
	NOP 0
	NOP 0
	NOP 0
	NOP 0
	NOP 0
	NOP 0
	NOP 0
	NOP 0
	NOP 0
	NOP 0
	NOP 0
	NOP 0
	NOP 0
	NOP 0
	NOP 0
	NOP 0
	NOP 0
	NOP 0
	NOP 0
	NOP 0
	NOP 0
	NOP 0
	NOP 0
	NOP 0
	NOP 0
	NOP 0
	NOP 0
	NOP 0
	NOP 0
	NOP 0
	NOP 0
	NOP 0
	NOP 0
	NOP 0
	NOP 0
	NOP 0
	NOP 0
	NOP 0
	NOP 0
	NOP 0
	NOP 0
	NOP 0
	NOP 0
	NOP 0
	NOP 0
	NOP 0
	NOP 0
	NOP 0
	NOP 0
	NOP 0
	NOP 0
	NOP 0
	NOP 0
	NOP 0
	NOP 0
	NOP 0
	NOP 0
	NOP 0
	NOP 0
	NOP 0
	NOP 0
	NOP 0
	NOP 0
	NOP 0
	NOP 0
	NOP 0
	NOP 0
	NOP 0
	NOP 0
	NOP 0
	NOP 0
	NOP 0
	NOP 0
	NOP 0
	NOP 0
	NOP 0
	NOP 0
	NOP 0
	NOP 0
	NOP 0
	NOP 0
	NOP 0
	NOP 0
	NOP 0
	NOP 0
	NOP 0
	NOP 0
	NOP 0
	NOP 0
	NOP 0
	NOP 0
	NOP 0
	NOP 0
	NOP 0
	NOP 0
	NOP 0
	NOP 0
	NOP 0
	NOP 0
	NOP 0
	NOP 0
	NOP 0
	NOP 0
	NOP 0
	NOP 0
	NOP 0
	NOP 0
	NOP 0
	NOP 0
	NOP 0
	NOP 0
	NOP 0
	NOP 0
	NOP 0
	NOP 0
	NOP 0
	NOP 0
	NOP 0
	NOP 0
	NOP 0
	NOP 0
	NOP 0
	NOP 0
	NOP 0
	NOP 0
	NOP 0
	NOP 0
	NOP 0
	NOP 0
	NOP 0
	NOP 0
	NOP 0
	NOP 0
	NOP 0
	NOP 0
	NOP 0
	NOP 0
	NOP 0
	NOP 0
	NOP 0
	NOP 0
	NOP 0
	NOP 0
	NOP 0
	NOP 0
	NOP 0
	NOP 0
	NOP 0
	NOP 0
	NOP 0
	NOP 0
	NOP 0
	NOP 0
	NOP 0
	NOP 0
	NOP 0
	NOP 0
	NOP 0
	NOP 0
	NOP 0
	NOP 0
	NOP 0
	NOP 0
	NOP 0
	NOP 0
	NOP 0
	NOP 0
	NOP 0
	NOP 0
	NOP 0
	NOP 0
	NOP 0
	NOP 0
	NOP 0
	NOP 0
	NOP 0
	NOP 0
	NOP 0
	NOP 0
	NOP 0
	NOP 0
	NOP 0
	NOP 0
	NOP 0
	NOP 0
	NOP 0
	NOP 0
	NOP 0
	NOP 0
	NOP 0
	NOP 0
	NOP 0
	NOP 0
	NOP 0
	NOP 0
	NOP 0
	NOP 0
	NOP 0
	NOP 0
	NOP 0
	NOP 0
	NOP 0
	NOP 0
	NOP 0
	NOP 0
	NOP 0
	NOP 0
	NOP 0
	NOP 0
	NOP 0
	NOP 0
	NOP 0
	NOP 0
	NOP 0
	NOP 0
	NOP 0
	NOP 0
	NOP 0
	NOP 0
	NOP 0
	NOP 0
	NOP 0
	NOP 0
	NOP 0
	NOP 0
	NOP 0
	NOP 0
	NOP 0
	NOP 0
	NOP 0
	NOP 0
	NOP 0
	NOP 0
	NOP 0
	NOP 0
	NOP 0
	NOP 0
	NOP 0
	NOP 0
	NOP 0
	NOP 0
	NOP 0
	NOP 0
	NOP 0
	NOP 0
	NOP 0
	NOP 0
	NOP 0
	NOP 0
	NOP 0
	NOP 0
	NOP 0
	NOP 0
	NOP 0
	NOP 0
	NOP 0
	NOP 0
	NOP 0
	NOP 0
	NOP 0
	NOP 0
	NOP 0
	NOP 0
	NOP 0
	NOP 0
	NOP 0
	NOP 0
	NOP 0
	NOP 0
	NOP 0
	NOP 0
	NOP 0
	NOP 0
	NOP 0
	NOP 0
	NOP 0
	NOP 0
	NOP 0
	NOP 0
	NOP 0
	NOP 0
	NOP 0
	NOP 0
	NOP 0
	NOP 0
	NOP 0
	NOP 0
	NOP 0
	NOP 0
	NOP 0
	NOP 0
	NOP 0
	NOP 0
	NOP 0
	NOP 0
	NOP 0
	NOP 0
	NOP 0
	NOP 0
	NOP 0
	NOP 0
	NOP 0
	NOP 0
	NOP 0
	NOP 0
	NOP 0
	NOP 0
	NOP 0
	NOP 0
	NOP 0
	NOP 0
	NOP 0
	NOP 0
	NOP 0
	NOP 0
	NOP 0
	NOP 0
	NOP 0
	NOP 0
	NOP 0
	NOP 0
	NOP 0
	NOP 0
	NOP 0
	NOP 0
	NOP 0
	NOP 0
	NOP 0
	NOP 0
	NOP 0
	NOP 0
	NOP 0
	NOP 0
	NOP 0
	NOP 0
	NOP 0
	NOP 0
	NOP 0
	NOP 0
	NOP 0
	NOP 0
	NOP 0
	NOP 0
	NOP 0
	NOP 0
	NOP 0
	NOP 0
	NOP 0
	NOP 0
	NOP 0
	NOP 0
	NOP 0
	NOP 0
	NOP 0
	NOP 0
	NOP 0
	NOP 0
	NOP 0
	NOP 0
	NOP 0
	NOP 0
	NOP 0
	NOP 0
	NOP 0
	NOP 0
	NOP 0
	NOP 0
	NOP 0
	NOP 0
	NOP 0
	NOP 0
	NOP 0
	NOP 0
	NOP 0
	NOP 0
	NOP 0
	NOP 0
	NOP 0
	NOP 0
	NOP 0
	NOP 0
	NOP 0
	NOP 0
	NOP 0
	NOP 0
	NOP 0
	NOP 0
	NOP 0
	NOP 0
	NOP 0
	NOP 0
	NOP 0
	NOP 0
	NOP 0
	NOP 0
	NOP 0
	NOP 0
	NOP 0
	NOP 0
	NOP 0
	NOP 0
	NOP 0
	NOP 0
	NOP 0
	NOP 0
	NOP 0
	NOP 0
	NOP 0
	NOP 0
	NOP 0
	NOP 0
	NOP 0
	NOP 0
	NOP 0
	NOP 0
	NOP 0
	NOP 0
	NOP 0
	NOP 0
	NOP 0
	NOP 0
	NOP 0
	NOP 0
	NOP 0
	NOP 0
	NOP 0
	NOP 0
	NOP 0
	NOP 0
	NOP 0
	NOP 0
	NOP 0
	NOP 0
	NOP 0
	NOP 0
	NOP 0
	NOP 0
	NOP 0
	NOP 0
	NOP 0
	NOP 0
	NOP 0
	NOP 0
	NOP 0
	NOP 0
	NOP 0
	NOP 0
	NOP 0
	NOP 0
	NOP 0
	NOP 0
	NOP 0
	NOP 0
	NOP 0
	NOP 0
	NOP 0
	NOP 0
	NOP 0
	NOP 0
	NOP 0
	NOP 0
	NOP 0
	NOP 0
	NOP 0
	NOP 0
	NOP 0
	NOP 0
	NOP 0
	NOP 0
	NOP 0
	NOP 0
	NOP 0
	NOP 0
	NOP 0
	NOP 0
	NOP 0
	NOP 0
	NOP 0
	NOP 0
	NOP 0
	NOP 0
	NOP 0
	NOP 0
	NOP 0
	NOP 0
	NOP 0
	NOP 0
	NOP 0
	NOP 0
	NOP 0
	NOP 0
	NOP 0
	NOP 0
	NOP 0
	NOP 0
	NOP 0
	NOP 0
	NOP 0
	NOP 0
	NOP 0
	NOP 0
	NOP 0
	NOP 0
	NOP 0
	NOP 0
	NOP 0
	NOP 0
	NOP 0
	NOP 0
	NOP 0
	NOP 0
	NOP 0
	NOP 0
	NOP 0
	NOP 0
	NOP 0
	NOP 0
	NOP 0
	NOP 0
	NOP 0
	NOP 0
	NOP 0
	NOP 0
	NOP 0
	NOP 0
	NOP 0
	NOP 0
	NOP 0
	NOP 0
	NOP 0
	NOP 0
	NOP 0
	NOP 0
	NOP 0
	NOP 0
	NOP 0
	NOP 0
	NOP 0
	NOP 0
	NOP 0
	NOP 0
	NOP 0
	NOP 0
	NOP 0
	NOP 0
	NOP 0
	NOP 0
	NOP 0
	NOP 0
	NOP 0
	NOP 0
	NOP 0
	NOP 0
	NOP 0
	NOP 0
	NOP 0
	NOP 0
	NOP 0
	NOP 0
	NOP 0
	NOP 0
	NOP 0
	NOP 0
	NOP 0
	NOP 0
	NOP 0
	NOP 0
	NOP 0
	NOP 0
	NOP 0
	NOP 0
	NOP 0
	NOP 0
	NOP 0
	NOP 0
	NOP 0
	NOP 0
	NOP 0
	NOP 0
	NOP 0
	NOP 0
	NOP 0
	NOP 0
	NOP 0
	NOP 0
	NOP 0
	NOP 0
	NOP 0
	NOP 0
	NOP 0
	NOP 0
	NOP 0
	NOP 0
	NOP 0
	NOP 0
	NOP 0
	NOP 0
	NOP 0
	NOP 0
	NOP 0
	NOP 0
	NOP 0
	NOP 0
	NOP 0
	NOP 0
	NOP 0
	NOP 0
	NOP 0
	NOP 0
	NOP 0
	NOP 0
	NOP 0
	NOP 0
	NOP 0
	NOP 0
	NOP 0
	NOP 0
	NOP 0
	NOP 0
	NOP 0
	NOP 0
	NOP 0
	NOP 0
	NOP 0
	NOP 0
	NOP 0
	NOP 0
	NOP 0
	NOP 0
	NOP 0
	NOP 0
	NOP 0
	NOP 0
	NOP 0
	NOP 0
	NOP 0
	NOP 0
	NOP 0
	NOP 0
	NOP 0
	NOP 0
	NOP 0
	NOP 0
	NOP 0
	NOP 0
	NOP 0
	NOP 0
	NOP 0
	NOP 0
	NOP 0
	NOP 0
	NOP 0
	NOP 0
	NOP 0
	NOP 0
	NOP 0
	NOP 0
	NOP 0
	NOP 0
	NOP 0
	NOP 0
	NOP 0
	NOP 0
	NOP 0
	NOP 0
	NOP 0
	NOP 0
	NOP 0
	NOP 0
	NOP 0
	NOP 0
	NOP 0
	NOP 0
	NOP 0
	NOP 0
	NOP 0
	NOP 0
	NOP 0
	NOP 0
	NOP 0
	NOP 0
	NOP 0
	NOP 0
	NOP 0
	NOP 0
	NOP 0
	NOP 0
	NOP 0
	NOP 0
	NOP 0
	NOP 0
	NOP 0
	NOP 0
	NOP 0
	NOP 0
	NOP 0
	NOP 0
	NOP 0
	NOP 0
	NOP 0
	NOP 0
	NOP 0
	NOP 0
	NOP 0
	NOP 0
	NOP 0
	NOP 0
	NOP 0
	NOP 0
	NOP 0
	NOP 0
	NOP 0
	NOP 0
	NOP 0
	NOP 0
	NOP 0
	NOP 0
	NOP 0
	NOP 0
	NOP 0
	NOP 0
	NOP 0
	NOP 0
	NOP 0
	NOP 0
	NOP 0
	NOP 0
	NOP 0
	NOP 0
	NOP 0
	NOP 0
	NOP 0
	NOP 0
	NOP 0
	NOP 0
	NOP 0
	NOP 0
	NOP 0
	NOP 0
	NOP 0
	NOP 0
	NOP 0
	NOP 0
	NOP 0
	NOP 0
	NOP 0
	NOP 0
	NOP 0
	NOP 0
	NOP 0
	NOP 0
	NOP 0
	NOP 0
	NOP 0
	NOP 0
	NOP 0
	NOP 0
	NOP 0
	NOP 0
	NOP 0
	NOP 0
	NOP 0
	NOP 0
	NOP 0
	NOP 0
	NOP 0
	NOP 0
	NOP 0
	NOP 0
	NOP 0
	NOP 0
	NOP 0
	NOP 0
	NOP 0
	NOP 0
	NOP 0
	NOP 0
	NOP 0
	NOP 0
	NOP 0
	NOP 0
	NOP 0
	NOP 0
	NOP 0
	NOP 0
	NOP 0
	NOP 0
	NOP 0
	NOP 0
	NOP 0
	NOP 0
	NOP 0
	NOP 0
	NOP 0
	NOP 0
	NOP 0
	NOP 0
	NOP 0
	NOP 0
	NOP 0
	NOP 0
	NOP 0
	NOP 0
	NOP 0
	NOP 0
	NOP 0
	NOP 0
	NOP 0
	NOP 0
	NOP 0
	NOP 0
	NOP 0
	NOP 0
	NOP 0
	NOP 0
	NOP 0
	NOP 0
	NOP 0
	NOP 0
	NOP 0
	NOP 0
	NOP 0
	NOP 0
	NOP 0
	NOP 0
	NOP 0
	NOP 0
	NOP 0
	NOP 0
	NOP 0
	NOP 0
	NOP 0
	NOP 0
	NOP 0
	NOP 0
	NOP 0
	NOP 0
	NOP 0
	NOP 0
	NOP 0
	NOP 0
	NOP 0
	NOP 0
	NOP 0
	NOP 0
	NOP 0
	NOP 0
	NOP 0
	NOP 0
	NOP 0
	NOP 0
	NOP 0
	NOP 0
	NOP 0
	NOP 0
	NOP 0
	NOP 0
	NOP 0
	NOP 0
	NOP 0
	NOP 0
	NOP 0
	NOP 0
	NOP 0
	NOP 0
	NOP 0
	NOP 0
	NOP 0
	NOP 0
	NOP 0
	NOP 0
	NOP 0
	NOP 0
	NOP 0
	NOP 0
	NOP 0
	NOP 0
	NOP 0
	NOP 0
	NOP 0
	NOP 0
	NOP 0
	NOP 0
	NOP 0
	NOP 0
	NOP 0
	NOP 0
	NOP 0
	NOP 0
	NOP 0
	NOP 0
	NOP 0
	NOP 0
	NOP 0
	NOP 0
	NOP 0
	NOP 0
	NOP 0
	NOP 0
	NOP 0
	NOP 0
	NOP 0
	NOP 0
	NOP 0
	NOP 0
	NOP 0
	NOP 0
	NOP 0
	NOP 0
	NOP 0
	NOP 0
	NOP 0
	NOP 0
	NOP 0
	NOP 0
	NOP 0
	NOP 0
	NOP 0
	NOP 0
	NOP 0
	NOP 0
	NOP 0
	NOP 0
	NOP 0
	NOP 0
	NOP 0
	NOP 0
	NOP 0
	NOP 0
	NOP 0
	NOP 0
	NOP 0
	NOP 0
	NOP 0
	NOP 0
	NOP 0
	NOP 0
	NOP 0
	NOP 0
	NOP 0
	NOP 0
	NOP 0
	NOP 0
	NOP 0
	NOP 0
	NOP 0
	NOP 0
	NOP 0
	NOP 0
	NOP 0
	NOP 0
	NOP 0
	NOP 0
	NOP 0
	NOP 0
	NOP 0
	NOP 0
	NOP 0
	NOP 0
	NOP 0
	NOP 0
	NOP 0
	NOP 0
	NOP 0
	NOP 0
	NOP 0
	NOP 0
	NOP 0
	NOP 0
	NOP 0
	NOP 0
	NOP 0
	NOP 0
	NOP 0
	NOP 0
	NOP 0
	NOP 0
	NOP 0
	NOP 0
	NOP 0
	NOP 0
	NOP 0
	NOP 0
	NOP 0
	NOP 0
	NOP 0
	NOP 0
	NOP 0
	NOP 0
	NOP 0
	NOP 0
	NOP 0
	NOP 0
	NOP 0
	NOP 0
	NOP 0
	NOP 0
	NOP 0
	NOP 0
	NOP 0
	NOP 0
	NOP 0
	NOP 0
	NOP 0
	NOP 0
	NOP 0
	NOP 0
	NOP 0
	NOP 0
	NOP 0
	NOP 0
	NOP 0
	NOP 0
	NOP 0
	NOP 0
	NOP 0
	NOP 0
	NOP 0
	NOP 0
	NOP 0
	NOP 0
	NOP 0
	NOP 0
	NOP 0
	NOP 0
	NOP 0
	NOP 0
	NOP 0
	NOP 0
	NOP 0
	NOP 0
	NOP 0
	NOP 0
	NOP 0
	NOP 0
	NOP 0
	NOP 0
	NOP 0
	NOP 0
	NOP 0
	NOP 0
	NOP 0
	NOP 0
	NOP 0
	NOP 0
	NOP 0
	NOP 0
	NOP 0
	NOP 0
	NOP 0
	NOP 0
	NOP 0
	NOP 0
	NOP 0
	NOP 0
	NOP 0
	NOP 0
	NOP 0
	NOP 0
	NOP 0
	NOP 0
	NOP 0
	NOP 0
	NOP 0
	NOP 0
	NOP 0
	NOP 0
	NOP 0
	NOP 0
	NOP 0
	NOP 0
	NOP 0
	NOP 0
	NOP 0
	NOP 0
	NOP 0
	NOP 0
	NOP 0
	NOP 0
	NOP 0
	NOP 0
	NOP 0
	NOP 0
	NOP 0
	NOP 0
	NOP 0
	NOP 0
	NOP 0
	NOP 0
	NOP 0
	NOP 0
	NOP 0
	NOP 0
	NOP 0
	NOP 0
	NOP 0
	NOP 0
	NOP 0
	NOP 0
	NOP 0
	NOP 0
	NOP 0
	NOP 0
	NOP 0
	NOP 0
	NOP 0
	NOP 0
	NOP 0
	NOP 0
	NOP 0
	NOP 0
	NOP 0
	NOP 0
	NOP 0
	NOP 0
	NOP 0
	NOP 0
	NOP 0
	NOP 0
	NOP 0
	NOP 0
	NOP 0
	NOP 0
	NOP 0
	NOP 0
	NOP 0
	NOP 0
	NOP 0
	NOP 0
	NOP 0
	NOP 0
	NOP 0
	NOP 0
	NOP 0
	NOP 0
	NOP 0
	NOP 0
	NOP 0
	NOP 0
	NOP 0
	NOP 0
	NOP 0
	NOP 0
	NOP 0
	NOP 0
	NOP 0
	NOP 0
	NOP 0
	NOP 0
	NOP 0
	NOP 0
	NOP 0
	NOP 0
	NOP 0
	NOP 0
	NOP 0
	NOP 0
	NOP 0
	NOP 0
	NOP 0
	NOP 0
	NOP 0
	NOP 0
	NOP 0
	NOP 0
	NOP 0
	NOP 0
	NOP 0
	NOP 0
	NOP 0
	NOP 0
	NOP 0
	NOP 0
	NOP 0
	NOP 0
	NOP 0
	NOP 0
	NOP 0
	NOP 0
	NOP 0
	NOP 0
	NOP 0
	NOP 0
	NOP 0
	NOP 0
	NOP 0
	NOP 0
	NOP 0
	NOP 0
	NOP 0
	NOP 0
	NOP 0
	NOP 0
	NOP 0
	NOP 0
	NOP 0
	NOP 0
	NOP 0
	NOP 0
	NOP 0
	NOP 0
	NOP 0
	NOP 0
	NOP 0
	NOP 0
	NOP 0
	NOP 0
	NOP 0
	NOP 0
	NOP 0
	NOP 0
	NOP 0
	NOP 0
	NOP 0
	NOP 0
	NOP 0
	NOP 0
	NOP 0
	NOP 0
	NOP 0
	NOP 0
	NOP 0
	NOP 0
	NOP 0
	NOP 0
	NOP 0
	NOP 0
	NOP 0
	NOP 0
	NOP 0
	NOP 0
	NOP 0
	NOP 0
	NOP 0
	NOP 0
	NOP 0
	NOP 0
	NOP 0
	NOP 0
	NOP 0
	NOP 0
	NOP 0
	NOP 0
	NOP 0
	NOP 0
	NOP 0
	NOP 0
	NOP 0
	NOP 0
	NOP 0
	NOP 0
	NOP 0
	NOP 0
	NOP 0
	NOP 0
	NOP 0
	NOP 0
	NOP 0
	NOP 0
	NOP 0
	NOP 0
	NOP 0
	NOP 0
	NOP 0
	NOP 0
	NOP 0
	NOP 0
	NOP 0
	NOP 0
	NOP 0
	NOP 0
	NOP 0
	NOP 0
	NOP 0
	NOP 0
	NOP 0
	NOP 0
	NOP 0
	NOP 0
	NOP 0
	NOP 0
	NOP 0
	NOP 0
	NOP 0
	NOP 0
	NOP 0
	NOP 0
	NOP 0
	NOP 0
	NOP 0
	NOP 0
	NOP 0
	NOP 0
	NOP 0
	NOP 0
	NOP 0
	NOP 0
	NOP 0
	NOP 0
	NOP 0
	NOP 0
	NOP 0
	NOP 0
	NOP 0
	NOP 0
	NOP 0
	NOP 0
	NOP 0
	NOP 0
	NOP 0
	NOP 0
	NOP 0
	NOP 0
	NOP 0
	NOP 0
	NOP 0
	NOP 0
	NOP 0
	NOP 0
	NOP 0
	NOP 0
	NOP 0
	NOP 0
	NOP 0
	NOP 0
	NOP 0
	NOP 0
	NOP 0
	NOP 0
	NOP 0
	NOP 0
	NOP 0
	NOP 0
	NOP 0
	NOP 0
	NOP 0
	NOP 0
	NOP 0
	NOP 0
	NOP 0
	NOP 0
	NOP 0
	NOP 0
	NOP 0
	NOP 0
	NOP 0
	NOP 0
	NOP 0
	NOP 0
	NOP 0
	NOP 0
	NOP 0
	NOP 0
	NOP 0
	NOP 0
	NOP 0
	NOP 0
	NOP 0
	NOP 0
	NOP 0
	NOP 0
	NOP 0
	NOP 0
	NOP 0
	NOP 0
	NOP 0
	NOP 0
	NOP 0
	NOP 0
	NOP 0
	NOP 0
	NOP 0
	NOP 0
	NOP 0
	NOP 0
	NOP 0
	NOP 0
	NOP 0
	NOP 0
	NOP 0
	NOP 0
	NOP 0
	NOP 0
	NOP 0
	NOP 0
	NOP 0
	NOP 0
	NOP 0
	NOP 0
	NOP 0
	NOP 0
	NOP 0
	NOP 0
	NOP 0
	NOP 0
	NOP 0
	NOP 0
	NOP 0
	NOP 0
	NOP 0
	NOP 0
	NOP 0
	NOP 0
	NOP 0
	NOP 0
	NOP 0
	NOP 0
	NOP 0
	NOP 0
	NOP 0
	NOP 0
	NOP 0
	NOP 0
	NOP 0
	NOP 0
	NOP 0
	NOP 0
	NOP 0
	NOP 0
	NOP 0
	NOP 0
	NOP 0
	NOP 0
	NOP 0
	NOP 0
	NOP 0
	NOP 0
	NOP 0
	NOP 0
	NOP 0
	NOP 0
	NOP 0
	NOP 0
	NOP 0
	NOP 0
	NOP 0
	NOP 0
	NOP 0
	NOP 0
	NOP 0
	NOP 0
	NOP 0
	NOP 0
	NOP 0
	NOP 0
	NOP 0
	NOP 0
	NOP 0
	NOP 0
	NOP 0
	NOP 0
	NOP 0
	NOP 0
	NOP 0
	NOP 0
	NOP 0
	NOP 0
	NOP 0
	NOP 0
	NOP 0
	NOP 0
	NOP 0
	NOP 0
	NOP 0
	NOP 0
	NOP 0
	NOP 0
	NOP 0
	NOP 0
	NOP 0
	NOP 0
	NOP 0
	NOP 0
	NOP 0
	NOP 0
	NOP 0
	NOP 0
	NOP 0
	NOP 0
	NOP 0
	NOP 0
	NOP 0
	NOP 0
	NOP 0
	NOP 0
	NOP 0
	NOP 0
	NOP 0
	NOP 0
	NOP 0
	NOP 0
	NOP 0
	NOP 0
	NOP 0
	NOP 0
	NOP 0
	NOP 0
	NOP 0
	NOP 0
	NOP 0
	NOP 0
	NOP 0
	NOP 0
	NOP 0
	NOP 0
	NOP 0
	NOP 0
	NOP 0
	NOP 0
	NOP 0
	NOP 0
	NOP 0
	NOP 0
	NOP 0
	NOP 0
	NOP 0
	NOP 0
	NOP 0
	NOP 0
	NOP 0
	NOP 0
	NOP 0
	NOP 0
	NOP 0
	NOP 0
	NOP 0
	NOP 0
	NOP 0
	NOP 0
	NOP 0
	NOP 0
	NOP 0
	NOP 0
	NOP 0
	NOP 0
	NOP 0
	NOP 0
	NOP 0
	NOP 0
	NOP 0
	NOP 0
	NOP 0
	NOP 0
	NOP 0
	NOP 0
	NOP 0
	NOP 0
	NOP 0
	NOP 0
	NOP 0
	NOP 0
	NOP 0
	NOP 0
	NOP 0
	NOP 0
	NOP 0
	NOP 0
	NOP 0
	NOP 0
	NOP 0
	NOP 0
	NOP 0
	NOP 0
	NOP 0
	NOP 0
	NOP 0
	NOP 0
	NOP 0
	NOP 0
	NOP 0
	NOP 0
	NOP 0
	NOP 0
	NOP 0
	NOP 0
	NOP 0
	NOP 0
	NOP 0
	NOP 0
	NOP 0
	NOP 0
	NOP 0
	NOP 0
	NOP 0
	NOP 0
	NOP 0
	NOP 0
	NOP 0
	NOP 0
	NOP 0
	NOP 0
	NOP 0
	NOP 0
	NOP 0
	NOP 0
	NOP 0
	NOP 0
	NOP 0
	NOP 0
	NOP 0
	NOP 0
	NOP 0
	NOP 0
	NOP 0
	NOP 0
	NOP 0
	NOP 0
	NOP 0
	NOP 0
	NOP 0
	NOP 0
	NOP 0
	NOP 0
	NOP 0
	NOP 0
	NOP 0
	NOP 0
	NOP 0
	NOP 0
	NOP 0
	NOP 0
	NOP 0
	NOP 0
	NOP 0
	NOP 0
	NOP 0
	NOP 0
	NOP 0
	NOP 0
	NOP 0
	NOP 0
	NOP 0
	NOP 0
	NOP 0
	NOP 0
	NOP 0
	NOP 0
	NOP 0
	NOP 0
	NOP 0
	NOP 0
	NOP 0
	NOP 0
	NOP 0
	NOP 0
	NOP 0
	NOP 0
	NOP 0
	NOP 0
	NOP 0
	NOP 0
	NOP 0
	NOP 0
	NOP 0
	NOP 0
	NOP 0
	NOP 0
	NOP 0
	NOP 0
	NOP 0
	NOP 0
	NOP 0
	NOP 0
	NOP 0
	NOP 0
	NOP 0
	NOP 0
	NOP 0
	NOP 0
	NOP 0
	NOP 0
	NOP 0
	NOP 0
	NOP 0
	NOP 0
	NOP 0
	NOP 0
	NOP 0
	NOP 0
	NOP 0
	NOP 0
	NOP 0
	NOP 0
	NOP 0
	NOP 0
	NOP 0
	NOP 0
	NOP 0
	NOP 0
	NOP 0
	NOP 0
	NOP 0
	NOP 0
	NOP 0
	NOP 0
	NOP 0
	NOP 0
	NOP 0
	NOP 0
	NOP 0
	NOP 0
	NOP 0
	NOP 0
	NOP 0
	NOP 0
	NOP 0
	NOP 0
	NOP 0
	NOP 0
	NOP 0
	NOP 0
	NOP 0
	NOP 0
	NOP 0
	NOP 0
	NOP 0
	NOP 0
	NOP 0
	NOP 0
	NOP 0
	NOP 0
	NOP 0
	NOP 0
	NOP 0
	NOP 0
	NOP 0
	NOP 0
	NOP 0
	NOP 0
	NOP 0
	NOP 0
	NOP 0
	NOP 0
	NOP 0
	NOP 0
	NOP 0
	NOP 0
	NOP 0
	NOP 0
	NOP 0
	NOP 0
	NOP 0
	NOP 0
	NOP 0
	NOP 0
	NOP 0
	NOP 0
	NOP 0
	NOP 0
	NOP 0
	NOP 0
	NOP 0
	NOP 0
	NOP 0
	NOP 0
	NOP 0
	NOP 0
	NOP 0
	NOP 0
	NOP 0
	NOP 0
	NOP 0
	NOP 0
	NOP 0
	NOP 0
	NOP 0
	NOP 0
	NOP 0
	NOP 0
	NOP 0
	NOP 0
	NOP 0
	NOP 0
	NOP 0
	NOP 0
	NOP 0
	NOP 0
	NOP 0
	NOP 0
	NOP 0
	NOP 0
	NOP 0
	NOP 0
	NOP 0
	NOP 0
	NOP 0
	NOP 0
	NOP 0
	NOP 0
	NOP 0
	NOP 0
	NOP 0
	NOP 0
	NOP 0
	NOP 0
	NOP 0
	NOP 0
	NOP 0
	NOP 0
	NOP 0
	NOP 0
	NOP 0
	NOP 0
	NOP 0
	NOP 0
	NOP 0
	NOP 0
	NOP 0
	NOP 0
	NOP 0
	NOP 0
	NOP 0
	NOP 0
	NOP 0
	NOP 0
	NOP 0
	NOP 0
	NOP 0
	NOP 0
	NOP 0
	NOP 0
	NOP 0
	NOP 0
	NOP 0
	NOP 0
	NOP 0
	NOP 0
	NOP 0
	NOP 0
	NOP 0
	NOP 0
	NOP 0
	NOP 0
	NOP 0
	NOP 0
	NOP 0
	NOP 0
	NOP 0
	NOP 0
	NOP 0
	NOP 0
	NOP 0
	NOP 0
	NOP 0
	NOP 0
	NOP 0
	NOP 0
	NOP 0
	NOP 0
	NOP 0
	NOP 0
	NOP 0
	NOP 0
	NOP 0
	NOP 0
	NOP 0
	NOP 0
	NOP 0
	NOP 0
	NOP 0
	NOP 0
	NOP 0
	NOP 0
	NOP 0
	NOP 0
	NOP 0
	NOP 0
	NOP 0
	NOP 0
	NOP 0
	NOP 0
	NOP 0
	NOP 0
	NOP 0
	NOP 0
	NOP 0
	NOP 0
	NOP 0
	NOP 0
	NOP 0
	NOP 0
	NOP 0
	NOP 0
	NOP 0
	NOP 0
	NOP 0
	NOP 0
	NOP 0
	NOP 0
	NOP 0
	NOP 0
	NOP 0
	NOP 0
	NOP 0
	NOP 0
	NOP 0
	NOP 0
	NOP 0
	NOP 0
	NOP 0
	NOP 0
	NOP 0
	NOP 0
	NOP 0
	NOP 0
	NOP 0
	NOP 0
	NOP 0
	NOP 0
	NOP 0
	NOP 0
	NOP 0
	NOP 0
	NOP 0
	NOP 0
	NOP 0
	NOP 0
	NOP 0
	NOP 0
	NOP 0
	NOP 0
	NOP 0
	NOP 0
	NOP 0
	NOP 0
	NOP 0
	NOP 0
	NOP 0
	NOP 0
	NOP 0
	NOP 0
	NOP 0
	NOP 0
	NOP 0
	NOP 0
	NOP 0
	NOP 0
	NOP 0
	NOP 0
	NOP 0
	NOP 0
	NOP 0
	NOP 0
	NOP 0
	NOP 0
	NOP 0
	NOP 0
	NOP 0
	NOP 0
	NOP 0
	NOP 0
	NOP 0
	NOP 0
	NOP 0
	NOP 0
	NOP 0
	NOP 0
	NOP 0
	NOP 0
	NOP 0
	NOP 0
	NOP 0
	NOP 0
	NOP 0
	NOP 0
	NOP 0
	NOP 0
	NOP 0
	NOP 0
	NOP 0
	NOP 0
	NOP 0
	NOP 0
	NOP 0
	NOP 0
	NOP 0
	NOP 0
	NOP 0
	NOP 0
	NOP 0
	NOP 0
	NOP 0
	NOP 0
	NOP 0
	NOP 0
	NOP 0
	NOP 0
	NOP 0
	NOP 0
	NOP 0
	NOP 0
	NOP 0
	NOP 0
	NOP 0
	NOP 0
	NOP 0
	NOP 0
	NOP 0
	NOP 0
	NOP 0
	NOP 0
	NOP 0
	NOP 0
	NOP 0
	NOP 0
	NOP 0
	NOP 0
	NOP 0
	NOP 0
	NOP 0
	NOP 0
	NOP 0
	NOP 0
	NOP 0
	NOP 0
	NOP 0
	NOP 0
	NOP 0
	NOP 0
	NOP 0
	NOP 0
	NOP 0
	NOP 0
	NOP 0
	NOP 0
	NOP 0
	NOP 0
	NOP 0
	NOP 0
	NOP 0
	NOP 0
	NOP 0
	NOP 0
	NOP 0
	NOP 0
	NOP 0
	NOP 0
	NOP 0
	NOP 0
	NOP 0
	NOP 0
	NOP 0
	NOP 0
	NOP 0
	NOP 0
	NOP 0
	NOP 0
	NOP 0
	NOP 0
	NOP 0
	NOP 0
	NOP 0
	NOP 0
	NOP 0
	NOP 0
	NOP 0
	NOP 0
	NOP 0
	NOP 0
	NOP 0
	NOP 0
	NOP 0
	NOP 0
	NOP 0
	NOP 0
	NOP 0
	NOP 0
	NOP 0
	NOP 0
	NOP 0
	NOP 0
	NOP 0
	NOP 0
	NOP 0
	NOP 0
	NOP 0
	NOP 0
	NOP 0
	NOP 0
	NOP 0
	NOP 0
	NOP 0
	NOP 0
	NOP 0
	NOP 0
	NOP 0
	NOP 0
	NOP 0
	NOP 0
	NOP 0
	NOP 0
	NOP 0
	NOP 0
	NOP 0
	NOP 0
	NOP 0
	NOP 0
	NOP 0
	NOP 0
	NOP 0
	NOP 0
	NOP 0
	NOP 0
	NOP 0
	NOP 0
	NOP 0
	NOP 0
	NOP 0
	NOP 0
	NOP 0
	NOP 0
	NOP 0
	NOP 0
	NOP 0
	NOP 0
	NOP 0
	NOP 0
	NOP 0
	NOP 0
	NOP 0
	NOP 0
	NOP 0
	NOP 0
	NOP 0
	NOP 0
	NOP 0
	NOP 0
	NOP 0
	NOP 0
	NOP 0
	NOP 0
	NOP 0
	NOP 0
	NOP 0
	NOP 0
	NOP 0
	NOP 0
	NOP 0
	NOP 0
	NOP 0
	NOP 0
	NOP 0
	NOP 0
	NOP 0
	NOP 0
	NOP 0
	NOP 0
	NOP 0
	NOP 0
	NOP 0
	NOP 0
	NOP 0
	NOP 0
	NOP 0
	NOP 0
	NOP 0
	NOP 0
	NOP 0
	NOP 0
	NOP 0
	NOP 0
	NOP 0
	NOP 0
	NOP 0
	NOP 0
	NOP 0
	NOP 0
	NOP 0
	NOP 0
	NOP 0
	NOP 0
	NOP 0
	NOP 0
	NOP 0
	NOP 0
	NOP 0
	NOP 0
	NOP 0
	NOP 0
	NOP 0
	NOP 0
	NOP 0
	NOP 0
	NOP 0
	NOP 0
	NOP 0
	NOP 0
	NOP 0
	NOP 0
	NOP 0
	NOP 0
	NOP 0
	NOP 0
	NOP 0
	NOP 0
	NOP 0
	NOP 0
	NOP 0
	NOP 0
	NOP 0
	NOP 0
	NOP 0
	NOP 0
	NOP 0
	NOP 0
	NOP 0
	NOP 0
	NOP 0
	NOP 0
	NOP 0
	NOP 0
	NOP 0
	NOP 0
	NOP 0
	NOP 0
	NOP 0
	NOP 0
	NOP 0
	NOP 0
	NOP 0
	NOP 0
	NOP 0
	NOP 0
	NOP 0
	NOP 0
	NOP 0
	NOP 0
	NOP 0
	NOP 0
	NOP 0
	NOP 0
	NOP 0
	NOP 0
	NOP 0
	NOP 0
	NOP 0
	NOP 0
	NOP 0
	NOP 0
	NOP 0
	NOP 0
	NOP 0
	NOP 0
	NOP 0
	NOP 0
	NOP 0
	NOP 0
	NOP 0
	NOP 0
	NOP 0
	NOP 0
	NOP 0
	NOP 0
	NOP 0
	NOP 0
	NOP 0
	NOP 0
	NOP 0
	NOP 0
	NOP 0
	NOP 0
	NOP 0
	NOP 0
	NOP 0
	NOP 0
	NOP 0
	NOP 0
	NOP 0
	NOP 0
	NOP 0
	NOP 0
	NOP 0
	NOP 0
	NOP 0
	NOP 0
	NOP 0
	NOP 0
	NOP 0
	NOP 0
	NOP 0
	NOP 0
	NOP 0
	NOP 0
	NOP 0
	NOP 0
	NOP 0
	NOP 0
	NOP 0
	NOP 0
	NOP 0
	NOP 0
	NOP 0
	NOP 0
	NOP 0
	NOP 0
	NOP 0
	NOP 0
	NOP 0
	NOP 0
	NOP 0
	NOP 0
	NOP 0
	NOP 0
	NOP 0
	NOP 0
	NOP 0
	NOP 0
	NOP 0
	NOP 0
	NOP 0
	NOP 0
	NOP 0
	NOP 0
	NOP 0
	NOP 0
	NOP 0
	NOP 0
	NOP 0
	NOP 0
	NOP 0
	NOP 0
	NOP 0
	NOP 0
	NOP 0
	NOP 0
	NOP 0
	NOP 0
	NOP 0
	NOP 0
	NOP 0
	NOP 0
	NOP 0
	NOP 0
	NOP 0
	NOP 0
	NOP 0
	NOP 0
	NOP 0
	NOP 0
	NOP 0
	NOP 0
	NOP 0
	NOP 0
	NOP 0
	NOP 0
	NOP 0
	NOP 0
	NOP 0
	NOP 0
	NOP 0
	NOP 0
	NOP 0
	NOP 0
	NOP 0
	NOP 0
	NOP 0
	NOP 0
	NOP 0
	NOP 0
	NOP 0
	NOP 0
	NOP 0
	NOP 0
	NOP 0
	NOP 0
	NOP 0
	NOP 0
	NOP 0
	NOP 0
	NOP 0
	NOP 0
	NOP 0
	NOP 0
	NOP 0
	NOP 0
	NOP 0
	NOP 0
	NOP 0
	NOP 0
	NOP 0
	NOP 0
	NOP 0
	NOP 0
	NOP 0
	NOP 0
	NOP 0
	NOP 0
	NOP 0
	NOP 0
	NOP 0
	NOP 0
	NOP 0
	NOP 0
	NOP 0
	NOP 0
	NOP 0
	NOP 0
	NOP 0
	NOP 0
	NOP 0
	NOP 0
	NOP 0
	NOP 0
	NOP 0
	NOP 0
	NOP 0
	NOP 0
	NOP 0
	NOP 0
	NOP 0
	NOP 0
	NOP 0
	NOP 0
	NOP 0
	NOP 0
	NOP 0
	NOP 0
	NOP 0
	NOP 0
	NOP 0
	NOP 0
	NOP 0
	NOP 0
	NOP 0
	NOP 0
	NOP 0
	NOP 0
	NOP 0
	NOP 0
	NOP 0
	NOP 0
	NOP 0
	NOP 0
	NOP 0
	NOP 0
	NOP 0
	NOP 0
	NOP 0
	NOP 0
	NOP 0
	NOP 0
	NOP 0
	NOP 0
	NOP 0
	NOP 0
	NOP 0
	NOP 0
	NOP 0
	NOP 0
	NOP 0
	NOP 0
	NOP 0
	NOP 0
	NOP 0
	NOP 0
	NOP 0
	NOP 0
	NOP 0
	NOP 0
	NOP 0
	NOP 0
	NOP 0
	NOP 0
	NOP 0
	NOP 0
	NOP 0
	NOP 0
	NOP 0
	NOP 0
	NOP 0
	NOP 0
	NOP 0
	NOP 0
	NOP 0
	NOP 0
	NOP 0
	NOP 0
	NOP 0
	NOP 0
	NOP 0
	NOP 0
	NOP 0
	NOP 0
	NOP 0
	NOP 0
	NOP 0
	NOP 0
	NOP 0
	NOP 0
	NOP 0
	NOP 0
	NOP 0
	NOP 0
	NOP 0
	NOP 0
	NOP 0
	NOP 0
	NOP 0
	NOP 0
	NOP 0
	NOP 0
	NOP 0
	NOP 0
	NOP 0
	NOP 0
	NOP 0
	NOP 0
	NOP 0
	NOP 0
	NOP 0
	NOP 0
	NOP 0
	NOP 0
	NOP 0
	NOP 0
	NOP 0
	NOP 0
	NOP 0
	NOP 0
	NOP 0
	NOP 0
	NOP 0
	NOP 0
	NOP 0
	NOP 0
	NOP 0
	NOP 0
	NOP 0
	NOP 0
	NOP 0
	NOP 0
	NOP 0
	NOP 0
	NOP 0
	NOP 0
	NOP 0
	NOP 0
	NOP 0
	NOP 0
	NOP 0
	NOP 0
	NOP 0
	NOP 0
	NOP 0
	NOP 0
	NOP 0
	NOP 0
	NOP 0
	NOP 0
	NOP 0
	NOP 0
	NOP 0
	NOP 0
	NOP 0
	NOP 0
	NOP 0
	NOP 0
	NOP 0
	NOP 0
	NOP 0
	NOP 0
	NOP 0
	NOP 0
	NOP 0
	NOP 0
	NOP 0
	NOP 0
	NOP 0
	NOP 0
	NOP 0
	NOP 0
	NOP 0
	NOP 0
	NOP 0
	NOP 0
	NOP 0
	NOP 0
	NOP 0
	NOP 0
	NOP 0
	NOP 0
	NOP 0
	NOP 0
	NOP 0
	NOP 0
	NOP 0
	NOP 0
	NOP 0
	NOP 0
	NOP 0
	NOP 0
	NOP 0
	NOP 0
	NOP 0
	NOP 0
	NOP 0
	NOP 0
	NOP 0
	NOP 0
	NOP 0
	NOP 0
	NOP 0
	NOP 0
	NOP 0
	NOP 0
	NOP 0
	NOP 0
	NOP 0
	NOP 0
	NOP 0
	NOP 0
	NOP 0
	NOP 0
	NOP 0
	NOP 0
	NOP 0
	NOP 0
	NOP 0
	NOP 0
	NOP 0
	NOP 0
	NOP 0
	NOP 0
	NOP 0
	NOP 0
	NOP 0
	NOP 0
	NOP 0
	NOP 0
	NOP 0
	NOP 0
	NOP 0
	NOP 0
	NOP 0
	NOP 0
	NOP 0
	NOP 0
	NOP 0
	NOP 0
	NOP 0
	NOP 0
	NOP 0
	NOP 0
	NOP 0
	NOP 0
	NOP 0
	NOP 0
	NOP 0
	NOP 0
	NOP 0
	NOP 0
	NOP 0
	NOP 0
	NOP 0
	NOP 0
	NOP 0
	NOP 0
	NOP 0
	NOP 0
	NOP 0
	NOP 0
	NOP 0
	NOP 0
	NOP 0
	NOP 0
	NOP 0
	NOP 0
	NOP 0
	NOP 0
	NOP 0
	NOP 0
	NOP 0
	NOP 0
	NOP 0
	NOP 0
	NOP 0
	NOP 0
	NOP 0
	NOP 0
	NOP 0
	NOP 0
	NOP 0
	NOP 0
	NOP 0
	NOP 0
	NOP 0
	NOP 0
	NOP 0
	NOP 0
	NOP 0
	NOP 0
	NOP 0
	NOP 0
	NOP 0
	NOP 0
	NOP 0
	NOP 0
	NOP 0
	NOP 0
	NOP 0
	NOP 0
	NOP 0
	NOP 0
	NOP 0
	NOP 0
	NOP 0
	NOP 0
	NOP 0
	NOP 0
	NOP 0
	NOP 0
	NOP 0
	NOP 0
	NOP 0
	NOP 0
	NOP 0
	NOP 0
	NOP 0
	NOP 0
	NOP 0
	NOP 0
	NOP 0
	NOP 0
	NOP 0
	NOP 0
	NOP 0
	NOP 0
	NOP 0
	NOP 0
	NOP 0
	NOP 0
	NOP 0
	NOP 0
	NOP 0
	NOP 0
	NOP 0
	NOP 0
	NOP 0
	NOP 0
	NOP 0
	NOP 0
	NOP 0
	NOP 0
	NOP 0
	NOP 0
	NOP 0
	NOP 0
	NOP 0
	NOP 0
	NOP 0
	NOP 0
	NOP 0
	NOP 0
	NOP 0
	NOP 0
	NOP 0
	NOP 0
	NOP 0
	NOP 0
	NOP 0
	NOP 0
	NOP 0
	NOP 0
	NOP 0
	NOP 0
	NOP 0
	NOP 0
	NOP 0
	NOP 0
	NOP 0
	NOP 0
	NOP 0
	NOP 0
	NOP 0
	NOP 0
	NOP 0
	NOP 0
	NOP 0
	NOP 0
	NOP 0
	NOP 0
	NOP 0
	NOP 0
	NOP 0
	NOP 0
	NOP 0
	NOP 0
	NOP 0
	NOP 0
	NOP 0
	NOP 0
	NOP 0
	NOP 0
	NOP 0
	NOP 0
	NOP 0
	NOP 0
	NOP 0
	NOP 0
	NOP 0
	NOP 0
	NOP 0
	NOP 0
	NOP 0
	NOP 0
	NOP 0
	NOP 0
	NOP 0
	NOP 0
	NOP 0
	NOP 0
	NOP 0
	NOP 0
	NOP 0
	NOP 0
	NOP 0
	NOP 0
	NOP 0
	NOP 0
	NOP 0
	NOP 0
	NOP 0
	NOP 0
	NOP 0
	NOP 0
	NOP 0
	NOP 0
	NOP 0
	NOP 0
	NOP 0
	NOP 0
	NOP 0
	NOP 0
	NOP 0
	NOP 0
	NOP 0
	NOP 0
	NOP 0
	NOP 0
	NOP 0
	NOP 0
	NOP 0
	NOP 0
	NOP 0
	NOP 0
	NOP 0
	NOP 0
	NOP 0
	NOP 0
	NOP 0
	NOP 0
	NOP 0
	NOP 0
	NOP 0
	NOP 0
	NOP 0
	NOP 0
	NOP 0
	NOP 0
	NOP 0
	NOP 0
	NOP 0
	NOP 0
	NOP 0
	NOP 0
	NOP 0
	NOP 0
	NOP 0
	NOP 0
	NOP 0
	NOP 0
	NOP 0
	NOP 0
	NOP 0
	NOP 0
	NOP 0
	NOP 0
	NOP 0
	NOP 0
	NOP 0
	NOP 0
	NOP 0
	NOP 0
	NOP 0
	NOP 0
	NOP 0
	NOP 0
	NOP 0
	NOP 0
	NOP 0
	NOP 0
	NOP 0
	NOP 0
	NOP 0
	NOP 0
	NOP 0
	NOP 0
	NOP 0
	NOP 0
	NOP 0
	NOP 0
	NOP 0
	NOP 0
	NOP 0
	NOP 0
	NOP 0
	NOP 0
	NOP 0
	NOP 0
	NOP 0
	NOP 0
	NOP 0
	NOP 0
	NOP 0
	NOP 0
	NOP 0
	NOP 0
	NOP 0
	NOP 0
	NOP 0
	NOP 0
	NOP 0
	NOP 0
	NOP 0
	NOP 0
	NOP 0
	NOP 0
	NOP 0
	NOP 0
	NOP 0
	NOP 0
	NOP 0
	NOP 0
	NOP 0
	NOP 0
	NOP 0
	NOP 0
	NOP 0
	NOP 0
	NOP 0
	NOP 0
	NOP 0
	NOP 0
	NOP 0
	NOP 0
	NOP 0
	NOP 0
	NOP 0
	NOP 0
	NOP 0
	NOP 0
	NOP 0
	NOP 0
	NOP 0
	NOP 0
	NOP 0
	NOP 0
	NOP 0
	NOP 0
	NOP 0
	NOP 0
	NOP 0
	NOP 0
	NOP 0
	NOP 0
	NOP 0
	NOP 0
	NOP 0
	NOP 0
	NOP 0
	NOP 0
	NOP 0
	NOP 0
	NOP 0
	NOP 0
	NOP 0
	NOP 0
	NOP 0
	NOP 0
	NOP 0
	NOP 0
	NOP 0
	NOP 0
	NOP 0
	NOP 0
	NOP 0
	NOP 0
	NOP 0
	NOP 0
	NOP 0
	NOP 0
	NOP 0
	NOP 0
	NOP 0
	NOP 0
	NOP 0
	NOP 0
	NOP 0
	NOP 0
	NOP 0
	NOP 0
	NOP 0
	NOP 0
	NOP 0
	NOP 0
	NOP 0
	NOP 0
	NOP 0
	NOP 0
	NOP 0
	NOP 0
	NOP 0
	NOP 0
	NOP 0
	NOP 0
	NOP 0
	NOP 0
	NOP 0
	NOP 0
	NOP 0
	NOP 0
	NOP 0
	NOP 0
	NOP 0
	NOP 0
	NOP 0
	NOP 0
	NOP 0
	NOP 0
	NOP 0
	NOP 0
	NOP 0
	NOP 0
	NOP 0
	NOP 0
	NOP 0
	NOP 0
	NOP 0
	NOP 0
	NOP 0
	NOP 0
	NOP 0
	NOP 0
	NOP 0
	NOP 0
	NOP 0
	NOP 0
	NOP 0
	NOP 0
	NOP 0
	NOP 0
	NOP 0
	NOP 0
	NOP 0
	NOP 0
	NOP 0
	NOP 0
	NOP 0
	NOP 0
	NOP 0
	NOP 0
	NOP 0
	NOP 0
	NOP 0
	NOP 0
	NOP 0
	NOP 0
	NOP 0
	NOP 0
	NOP 0
	NOP 0
	NOP 0
	NOP 0
	NOP 0
	NOP 0
	NOP 0
	NOP 0
	NOP 0
	NOP 0
	NOP 0
	NOP 0
	NOP 0
	NOP 0
	NOP 0
	NOP 0
	NOP 0
	NOP 0
	NOP 0
	NOP 0
	NOP 0
	NOP 0
	NOP 0
	NOP 0
	NOP 0
	NOP 0
	NOP 0
	NOP 0
	NOP 0
	NOP 0
	NOP 0
	NOP 0
	NOP 0
	NOP 0
	NOP 0
	NOP 0
	NOP 0
	NOP 0
	NOP 0
	NOP 0
	NOP 0
	NOP 0
	NOP 0
	NOP 0
	NOP 0
	NOP 0
	NOP 0
	NOP 0
	NOP 0
	NOP 0
	NOP 0
	NOP 0
	NOP 0
	NOP 0
	NOP 0
	NOP 0
	NOP 0
	NOP 0
	NOP 0
	NOP 0
	NOP 0
	NOP 0
	NOP 0
	NOP 0
	NOP 0
	NOP 0
	NOP 0
	NOP 0
	NOP 0
	NOP 0
	NOP 0
	NOP 0
	NOP 0
	NOP 0
	NOP 0
	NOP 0
	NOP 0
	NOP 0
	NOP 0
	NOP 0
	NOP 0
	NOP 0
	NOP 0
	NOP 0
	NOP 0
	NOP 0
	NOP 0
	NOP 0
	NOP 0
	NOP 0
	NOP 0
	NOP 0
	NOP 0
	NOP 0
	NOP 0
	NOP 0
	NOP 0
	NOP 0
	NOP 0
	NOP 0
	NOP 0
	NOP 0
	NOP 0
	NOP 0
	NOP 0
	NOP 0
	NOP 0
	NOP 0
	NOP 0
	NOP 0
	NOP 0
	NOP 0
	NOP 0
	NOP 0
	NOP 0
	NOP 0
	NOP 0
	NOP 0
	NOP 0
	NOP 0
	NOP 0
	NOP 0
	NOP 0
	NOP 0
	NOP 0
	NOP 0
	NOP 0
	NOP 0
	NOP 0
	NOP 0
	NOP 0
	NOP 0
	NOP 0
	NOP 0
	NOP 0
	NOP 0
	NOP 0
	NOP 0
	NOP 0
	NOP 0
	NOP 0
	NOP 0
	NOP 0
	NOP 0
	NOP 0
	NOP 0
	NOP 0
	NOP 0
	NOP 0
	NOP 0
	NOP 0
	NOP 0
	NOP 0
	NOP 0
	NOP 0
	NOP 0
	NOP 0
	NOP 0
	NOP 0
	NOP 0
	NOP 0
	NOP 0
	NOP 0
	NOP 0
	NOP 0
	NOP 0
	NOP 0
	NOP 0
	NOP 0
	NOP 0
	NOP 0
	NOP 0
	NOP 0
	NOP 0
	NOP 0
	NOP 0
	NOP 0
	NOP 0
	NOP 0
	NOP 0
	NOP 0
	NOP 0
	NOP 0
	NOP 0
	NOP 0
	NOP 0
	NOP 0
	NOP 0
	NOP 0
	NOP 0
	NOP 0
	NOP 0
	NOP 0
	NOP 0
	NOP 0
	NOP 0
	NOP 0
	NOP 0
	NOP 0
	NOP 0
	NOP 0
	NOP 0
	NOP 0
	NOP 0
	NOP 0
	NOP 0
	NOP 0
	NOP 0
	NOP 0
	NOP 0
	NOP 0
	NOP 0
	NOP 0
	NOP 0
	NOP 0
	NOP 0
	NOP 0
	NOP 0
	NOP 0
	NOP 0
	NOP 0
	NOP 0
	NOP 0
	NOP 0
	NOP 0
	NOP 0
	NOP 0
	NOP 0
	NOP 0
	NOP 0
	NOP 0
	NOP 0
	NOP 0
	NOP 0
	NOP 0
	NOP 0
	NOP 0
	NOP 0
	NOP 0
	NOP 0
	NOP 0
	NOP 0
	NOP 0
	NOP 0
	NOP 0
	NOP 0
	NOP 0
	NOP 0
	NOP 0
	NOP 0
	NOP 0
	NOP 0
	NOP 0
	NOP 0
	NOP 0
	NOP 0
	NOP 0
	NOP 0
	NOP 0
	NOP 0
	NOP 0
	NOP 0
	NOP 0
	NOP 0
	NOP 0
	NOP 0
	NOP 0
	NOP 0
	NOP 0
	NOP 0
	NOP 0
	NOP 0
	NOP 0
	NOP 0
	NOP 0
	NOP 0
	NOP 0
	NOP 0
	NOP 0
	NOP 0
	NOP 0
	NOP 0
	NOP 0
	NOP 0
	NOP 0
	NOP 0
	NOP 0
	NOP 0
	NOP 0
	NOP 0
	NOP 0
	NOP 0
	NOP 0
	NOP 0
	NOP 0
	NOP 0
	NOP 0
	NOP 0
	NOP 0
	NOP 0
	NOP 0
	NOP 0
	NOP 0
	NOP 0
	NOP 0
	NOP 0
	NOP 0
	NOP 0
	NOP 0
	NOP 0
	NOP 0
	NOP 0
	NOP 0
	NOP 0
	NOP 0
	NOP 0
	NOP 0
	NOP 0
	NOP 0
	NOP 0
	NOP 0
	NOP 0
	NOP 0
	NOP 0
	NOP 0
	NOP 0
	NOP 0
	NOP 0
	NOP 0
	NOP 0
	NOP 0
	NOP 0
	NOP 0
	NOP 0
	NOP 0
	NOP 0
	NOP 0
	NOP 0
	NOP 0
	NOP 0
	NOP 0
	NOP 0
	NOP 0
	NOP 0
	NOP 0
	NOP 0
	NOP 0
	NOP 0
	NOP 0
	NOP 0
	NOP 0
	NOP 0
	NOP 0
	NOP 0
	NOP 0
	NOP 0
	NOP 0
	NOP 0
	NOP 0
	NOP 0
	NOP 0
	NOP 0
	NOP 0
	NOP 0
	NOP 0
	NOP 0
	NOP 0
	NOP 0
	NOP 0
	NOP 0
	NOP 0
	NOP 0
	NOP 0
	NOP 0
	NOP 0
	NOP 0
	NOP 0
	NOP 0
	NOP 0
	NOP 0
	NOP 0
	NOP 0
	NOP 0
	NOP 0
	NOP 0
	NOP 0
	NOP 0
	NOP 0
	NOP 0
	NOP 0
	NOP 0
	NOP 0
	NOP 0
	NOP 0
	NOP 0
	NOP 0
	NOP 0
	NOP 0
	NOP 0
	NOP 0
	NOP 0
	NOP 0
	NOP 0
	NOP 0
	NOP 0
	NOP 0
	NOP 0
	NOP 0
	NOP 0
	NOP 0
	NOP 0
	NOP 0
	NOP 0
	NOP 0
	NOP 0
	NOP 0
	NOP 0
	NOP 0
	NOP 0
	NOP 0
	NOP 0
	NOP 0
	NOP 0
	NOP 0
	NOP 0
	NOP 0
	NOP 0
	NOP 0
	NOP 0
	NOP 0
	NOP 0
	NOP 0
	NOP 0
	NOP 0
	NOP 0
	NOP 0
	NOP 0
	NOP 0
	NOP 0
	NOP 0
	NOP 0
	NOP 0
	NOP 0
	NOP 0
	NOP 0
	NOP 0
	NOP 0
	NOP 0
	NOP 0
	NOP 0
	NOP 0
	NOP 0
	NOP 0
	NOP 0
	NOP 0
	NOP 0
	NOP 0
	NOP 0
	NOP 0
	NOP 0
	NOP 0
	NOP 0
	NOP 0
	NOP 0
	NOP 0
	NOP 0
	NOP 0
	NOP 0
	NOP 0
	NOP 0
	NOP 0
	NOP 0
	NOP 0
	NOP 0
	NOP 0
	NOP 0
	NOP 0
	NOP 0
	NOP 0
	NOP 0
	NOP 0
	NOP 0
	NOP 0
	NOP 0
	NOP 0
	NOP 0
	NOP 0
	NOP 0
	NOP 0
	NOP 0
	NOP 0
	NOP 0
	NOP 0
	NOP 0
	NOP 0
	NOP 0
	NOP 0
	NOP 0
	NOP 0
	NOP 0
	NOP 0
	NOP 0
	NOP 0
	NOP 0
	NOP 0
	NOP 0
	NOP 0
	NOP 0
	NOP 0
	NOP 0
	NOP 0
	NOP 0
	NOP 0
	NOP 0
	NOP 0
	NOP 0
	NOP 0
	NOP 0
	NOP 0
	NOP 0
	NOP 0
	NOP 0
	NOP 0
	NOP 0
	NOP 0
	NOP 0
	NOP 0
	NOP 0
	NOP 0
	NOP 0
	NOP 0
	NOP 0
	NOP 0
	NOP 0
	NOP 0
	NOP 0
	NOP 0
	NOP 0
	NOP 0
	NOP 0
	NOP 0
	NOP 0
	NOP 0
	NOP 0
	NOP 0
	NOP 0
	NOP 0
	NOP 0
	NOP 0
	NOP 0
	NOP 0
	NOP 0
	NOP 0
	NOP 0
	NOP 0
	NOP 0
	NOP 0
	NOP 0
	NOP 0
	NOP 0
	NOP 0
	NOP 0
	NOP 0
	NOP 0
	NOP 0
	NOP 0
	NOP 0
	NOP 0
	NOP 0
	NOP 0
	NOP 0
	NOP 0
	NOP 0
	NOP 0
	NOP 0
	NOP 0
	NOP 0
	NOP 0
	NOP 0
	NOP 0
	NOP 0
	NOP 0
	NOP 0
	NOP 0
	NOP 0
	NOP 0
	NOP 0
	NOP 0
	NOP 0
	NOP 0
	NOP 0
	NOP 0
	NOP 0
	NOP 0
	NOP 0
	NOP 0
	NOP 0
	NOP 0
	NOP 0
	NOP 0
	NOP 0
	NOP 0
	NOP 0
	NOP 0
	NOP 0
	NOP 0
	NOP 0
	NOP 0
	NOP 0
	NOP 0
	NOP 0
	NOP 0
	NOP 0
	NOP 0
	NOP 0
	NOP 0
	NOP 0
	NOP 0
	NOP 0
	NOP 0
	NOP 0
	NOP 0
	NOP 0
	NOP 0
	NOP 0
	NOP 0
	NOP 0
	NOP 0
	NOP 0
	NOP 0
	NOP 0
	NOP 0
	NOP 0
	NOP 0
	NOP 0
	NOP 0
	NOP 0
	NOP 0
	NOP 0
	NOP 0
	NOP 0
	NOP 0
	NOP 0
	NOP 0
	NOP 0
	NOP 0
	NOP 0
	NOP 0
	NOP 0
	NOP 0
	NOP 0
	NOP 0
	NOP 0
	NOP 0
	NOP 0
	NOP 0
	NOP 0
	NOP 0
	NOP 0
	NOP 0
	NOP 0
	NOP 0
	NOP 0
	NOP 0
	NOP 0
	NOP 0
	NOP 0
	NOP 0
	NOP 0
	NOP 0
	NOP 0
	NOP 0
	NOP 0
	NOP 0
	NOP 0
	NOP 0
	NOP 0
	NOP 0
	NOP 0
	NOP 0
	NOP 0
	NOP 0
	NOP 0
	NOP 0
	NOP 0
	NOP 0
	NOP 0
	NOP 0
	NOP 0
	NOP 0
	NOP 0
	NOP 0
	NOP 0
	NOP 0
	NOP 0
	NOP 0
	NOP 0
	NOP 0
	NOP 0
	NOP 0
	NOP 0
	NOP 0
	NOP 0
	NOP 0
	NOP 0
	NOP 0
	NOP 0
	NOP 0
	NOP 0
	NOP 0
	NOP 0
	NOP 0
	NOP 0
	NOP 0
	NOP 0
	NOP 0
	NOP 0
	NOP 0
	NOP 0
	NOP 0
	NOP 0
	NOP 0
	NOP 0
	NOP 0
	NOP 0
	NOP 0
	NOP 0
	NOP 0
	NOP 0
	NOP 0
	NOP 0
	NOP 0
	NOP 0
	NOP 0
	NOP 0
	NOP 0
	NOP 0
	NOP 0
	NOP 0
	NOP 0
	NOP 0
	NOP 0
	NOP 0
	NOP 0
	NOP 0
	NOP 0
	NOP 0
	NOP 0
	NOP 0
	NOP 0
	NOP 0
	NOP 0
	NOP 0
	NOP 0
	NOP 0
	NOP 0
	NOP 0
	NOP 0
	NOP 0
	NOP 0
	NOP 0
	NOP 0
	NOP 0
	NOP 0
	NOP 0
	NOP 0
	NOP 0
	NOP 0
	NOP 0
	NOP 0
	NOP 0
	NOP 0
	NOP 0
	NOP 0
	NOP 0
	NOP 0
	NOP 0
	NOP 0
	NOP 0
	NOP 0
	NOP 0
	NOP 0
	NOP 0
	NOP 0
	NOP 0
	NOP 0
	NOP 0
	NOP 0
	NOP 0
	NOP 0
	NOP 0
	NOP 0
	NOP 0
	NOP 0
	NOP 0
	NOP 0
	NOP 0
	NOP 0
	NOP 0
	NOP 0
	NOP 0
	NOP 0
	NOP 0
	NOP 0
	NOP 0
	NOP 0
	NOP 0
	NOP 0
	NOP 0
	NOP 0
	NOP 0
	NOP 0
	NOP 0
	NOP 0
	NOP 0
	NOP 0
	NOP 0
	NOP 0
	NOP 0
	NOP 0
	NOP 0
	NOP 0
	NOP 0
	NOP 0
	NOP 0
	NOP 0
	NOP 0
	NOP 0
	NOP 0
	NOP 0
	NOP 0
	NOP 0
	NOP 0
	NOP 0
	NOP 0
	NOP 0
	NOP 0
	NOP 0
	NOP 0
	NOP 0
	NOP 0
	NOP 0
	NOP 0
	NOP 0
	NOP 0
	NOP 0
	NOP 0
	NOP 0
	NOP 0
	NOP 0
	NOP 0
	NOP 0
	NOP 0
	NOP 0
	NOP 0
	NOP 0
	NOP 0
	NOP 0
	NOP 0
	NOP 0
	NOP 0
	NOP 0
	NOP 0
	NOP 0
	NOP 0
	NOP 0
	NOP 0
	NOP 0
	NOP 0
	NOP 0
	NOP 0
	NOP 0
	NOP 0
	NOP 0
	NOP 0
	NOP 0
	NOP 0
	NOP 0
	NOP 0
	NOP 0
	NOP 0
	NOP 0
	NOP 0
	NOP 0
	NOP 0
	NOP 0
	NOP 0
	NOP 0
	NOP 0
	NOP 0
	NOP 0
	NOP 0
	NOP 0
	NOP 0
	NOP 0
	NOP 0
	NOP 0
	NOP 0
	NOP 0
	NOP 0
	NOP 0
	NOP 0
	NOP 0
	NOP 0
	NOP 0
	NOP 0
	NOP 0
	NOP 0
	NOP 0
	NOP 0
	NOP 0
	NOP 0
	NOP 0
	NOP 0
	NOP 0
	NOP 0
	NOP 0
	NOP 0
	NOP 0
	NOP 0
	NOP 0
	NOP 0
	NOP 0
	NOP 0
	NOP 0
	NOP 0
	NOP 0
	NOP 0
	NOP 0
	NOP 0
	NOP 0
	NOP 0
	NOP 0
	NOP 0
	NOP 0
	NOP 0
	NOP 0
	NOP 0
	NOP 0
	NOP 0
	NOP 0
	NOP 0
	NOP 0
	NOP 0
	NOP 0
	NOP 0
	NOP 0
	NOP 0
	NOP 0
	NOP 0
	NOP 0
	NOP 0
	NOP 0
	NOP 0
	NOP 0
	NOP 0
	NOP 0
	NOP 0
	NOP 0
	NOP 0
	NOP 0
	NOP 0
	NOP 0
	NOP 0
	NOP 0
	NOP 0
	NOP 0
	NOP 0
	NOP 0
	NOP 0
	NOP 0
	NOP 0
	NOP 0
	NOP 0
	NOP 0
	NOP 0
	NOP 0
	NOP 0
	NOP 0
	NOP 0
	NOP 0
	NOP 0
	NOP 0
	NOP 0
	NOP 0
	NOP 0
	NOP 0
	NOP 0
	NOP 0
	NOP 0
	NOP 0
	NOP 0
	NOP 0
	NOP 0
	NOP 0
	NOP 0
	NOP 0
	NOP 0
	NOP 0
	NOP 0
	NOP 0
	NOP 0
	NOP 0
	NOP 0
	NOP 0
	NOP 0
	NOP 0
	NOP 0
	NOP 0
	NOP 0
	NOP 0
	NOP 0
	NOP 0
	NOP 0
	NOP 0
	NOP 0
	NOP 0
	NOP 0
	NOP 0
	NOP 0
	NOP 0
	NOP 0
	NOP 0
	NOP 0
	NOP 0
	NOP 0
	NOP 0
	NOP 0
	NOP 0
	NOP 0
	NOP 0
	NOP 0
	NOP 0
	NOP 0
	NOP 0
	NOP 0
	NOP 0
	NOP 0
	NOP 0
	NOP 0
	NOP 0
	NOP 0
	NOP 0
	NOP 0
	NOP 0
	NOP 0
	NOP 0
	NOP 0
	NOP 0
	NOP 0
	NOP 0
	NOP 0
	NOP 0
	NOP 0
	NOP 0
	NOP 0
	NOP 0
	NOP 0
	NOP 0
	NOP 0
	NOP 0
	NOP 0
	NOP 0
	NOP 0
	NOP 0
	NOP 0
	NOP 0
	NOP 0
	NOP 0
	NOP 0
	NOP 0
	NOP 0
	NOP 0
	NOP 0
	NOP 0
	NOP 0
	NOP 0
	NOP 0
	NOP 0
	NOP 0
	NOP 0
	NOP 0
	NOP 0
	NOP 0
	NOP 0
	NOP 0
	NOP 0
	NOP 0
	NOP 0
	NOP 0
	NOP 0
	NOP 0
	NOP 0
	NOP 0
	NOP 0
	NOP 0
	NOP 0
	NOP 0
	NOP 0
	NOP 0
	NOP 0
	NOP 0
	NOP 0
	NOP 0
	NOP 0
	NOP 0
	NOP 0
	NOP 0
	NOP 0
	NOP 0
	NOP 0
	NOP 0
	NOP 0
	NOP 0
	NOP 0
	NOP 0
	NOP 0
	NOP 0
	NOP 0
	NOP 0
	NOP 0
	NOP 0
	NOP 0
	NOP 0
	NOP 0
	NOP 0
	NOP 0
	NOP 0
	NOP 0
	NOP 0
	NOP 0
	NOP 0
	NOP 0
	NOP 0
	NOP 0
	NOP 0
	NOP 0
	NOP 0
	NOP 0
	NOP 0
	NOP 0
	NOP 0
	NOP 0
	NOP 0
	NOP 0
	NOP 0
	NOP 0
	NOP 0
	NOP 0
	NOP 0
	NOP 0
	NOP 0
	NOP 0
	NOP 0
	NOP 0
	NOP 0
	NOP 0
	NOP 0
	NOP 0
	NOP 0
	NOP 0
	NOP 0
	NOP 0
	NOP 0
	NOP 0
	NOP 0
	NOP 0
	NOP 0
	NOP 0
	NOP 0
	NOP 0
	NOP 0
	NOP 0
	NOP 0
	NOP 0
	NOP 0
	NOP 0
	NOP 0
	NOP 0
	NOP 0
	NOP 0
	NOP 0
	NOP 0
	NOP 0
	NOP 0
	NOP 0
	NOP 0
	NOP 0
	NOP 0
	NOP 0
	NOP 0
	NOP 0
	NOP 0
	NOP 0
	NOP 0
	NOP 0
	NOP 0
	NOP 0
	NOP 0
	NOP 0
	NOP 0
	NOP 0
	NOP 0
	NOP 0
	NOP 0
	NOP 0
	NOP 0
	NOP 0
	NOP 0
	NOP 0
	NOP 0
	NOP 0
	NOP 0
	NOP 0
	NOP 0
	NOP 0
	NOP 0
	NOP 0
	NOP 0
	NOP 0
	NOP 0
	NOP 0
	NOP 0
	NOP 0
	NOP 0
	NOP 0
	NOP 0
	NOP 0
	NOP 0
	NOP 0
	NOP 0
	NOP 0
	NOP 0
	NOP 0
	NOP 0
	NOP 0
	NOP 0
	NOP 0
	NOP 0
	NOP 0
	NOP 0
	NOP 0
	NOP 0
	NOP 0
	NOP 0
	NOP 0
	NOP 0
	NOP 0
	NOP 0
	NOP 0
	NOP 0
	NOP 0
	NOP 0
	NOP 0
	NOP 0
	NOP 0
	NOP 0
	NOP 0
	NOP 0
	NOP 0
	NOP 0
	NOP 0
	NOP 0
	NOP 0
	NOP 0
	NOP 0
	NOP 0
	NOP 0
	NOP 0
	NOP 0
	NOP 0
	NOP 0
	NOP 0
	NOP 0
	NOP 0
	NOP 0
	NOP 0
	NOP 0
	NOP 0
	NOP 0
	NOP 0
	NOP 0
	NOP 0
	NOP 0
	NOP 0
	NOP 0
	NOP 0
	NOP 0
	NOP 0
	NOP 0
	NOP 0
	NOP 0
	NOP 0
	NOP 0
	NOP 0
	NOP 0
	NOP 0
	NOP 0
	NOP 0
	NOP 0
	NOP 0
	NOP 0
	NOP 0
	NOP 0
	NOP 0
	NOP 0
	NOP 0
	NOP 0
	NOP 0
	NOP 0
	NOP 0
	NOP 0
	NOP 0
	NOP 0
	NOP 0
	NOP 0
	NOP 0
	NOP 0
	NOP 0
	NOP 0
	NOP 0
	NOP 0
	NOP 0
	NOP 0
	NOP 0
	NOP 0
	NOP 0
	NOP 0
	NOP 0
	NOP 0
	NOP 0
	NOP 0
	NOP 0
	NOP 0
	NOP 0
	NOP 0
	NOP 0
	NOP 0
	NOP 0
	NOP 0
	NOP 0
	NOP 0
	NOP 0
	NOP 0
	NOP 0
	NOP 0
	NOP 0
	NOP 0
	NOP 0
	NOP 0
	NOP 0
	NOP 0
	NOP 0
	NOP 0
	NOP 0
	NOP 0
	NOP 0
	NOP 0
	NOP 0
	NOP 0
	NOP 0
	NOP 0
	NOP 0
	NOP 0
	NOP 0
	NOP 0
	NOP 0
	NOP 0
	NOP 0
	NOP 0
	NOP 0
	NOP 0
	NOP 0
	NOP 0
	NOP 0
	NOP 0
	NOP 0
	NOP 0
	NOP 0
	NOP 0
	NOP 0
	NOP 0
	NOP 0
	NOP 0
	NOP 0
	NOP 0
	NOP 0
	NOP 0
	NOP 0
	NOP 0
	NOP 0
	NOP 0
	NOP 0
	NOP 0
	NOP 0
	NOP 0
	NOP 0
	NOP 0
	NOP 0
	NOP 0
	NOP 0
	NOP 0
	NOP 0
	NOP 0
	NOP 0
	NOP 0
	NOP 0
	NOP 0
	NOP 0
	NOP 0
	NOP 0
	NOP 0
	NOP 0
	NOP 0
	NOP 0
	NOP 0
	NOP 0
	NOP 0
	NOP 0
	NOP 0
	NOP 0
	NOP 0
	NOP 0
	NOP 0
	NOP 0
	NOP 0
	NOP 0
	NOP 0
	NOP 0
	NOP 0
	NOP 0
	NOP 0
	NOP 0
	NOP 0
	NOP 0
	NOP 0
	NOP 0
	NOP 0
	NOP 0
	NOP 0
	NOP 0
	NOP 0
	NOP 0
	NOP 0
	NOP 0
	NOP 0
	NOP 0
	NOP 0
	NOP 0
	NOP 0
	NOP 0
	NOP 0
	NOP 0
	NOP 0
	NOP 0
	NOP 0
	NOP 0
	NOP 0
	NOP 0
	NOP 0
	NOP 0
	NOP 0
	NOP 0
	NOP 0
	NOP 0
	NOP 0
	NOP 0
	NOP 0
	NOP 0
	NOP 0
	NOP 0
	NOP 0
	NOP 0
	NOP 0
	NOP 0
	NOP 0
	NOP 0
	NOP 0
	NOP 0
	NOP 0
	NOP 0
	NOP 0
	NOP 0
	NOP 0
	NOP 0
	NOP 0
	NOP 0
	NOP 0
	NOP 0
	NOP 0
	NOP 0
	NOP 0
	NOP 0
	NOP 0
	NOP 0
	NOP 0
	NOP 0
	NOP 0
	NOP 0
	NOP 0
	NOP 0
	NOP 0
	NOP 0
	NOP 0
	NOP 0
	NOP 0
	NOP 0
	NOP 0
	NOP 0
	NOP 0
	NOP 0
	NOP 0
	NOP 0
	NOP 0
	NOP 0
	NOP 0
	NOP 0
	NOP 0
	NOP 0
	NOP 0
	NOP 0
	NOP 0
	NOP 0
	NOP 0
	NOP 0
	NOP 0
	NOP 0
	NOP 0
	NOP 0
	NOP 0
	NOP 0
	NOP 0
	NOP 0
	NOP 0
	NOP 0
	NOP 0
	NOP 0
	NOP 0
	NOP 0
	NOP 0
	NOP 0
	NOP 0
	NOP 0
	NOP 0
	NOP 0
	NOP 0
	NOP 0
	NOP 0
	NOP 0
	NOP 0
	NOP 0
	NOP 0
	NOP 0
	NOP 0
	NOP 0
	NOP 0
	NOP 0
	NOP 0
	NOP 0
	NOP 0
	NOP 0
	NOP 0
	NOP 0
	NOP 0
	NOP 0
	NOP 0
	NOP 0
	NOP 0
	NOP 0
	NOP 0
	NOP 0
	NOP 0
	NOP 0
	NOP 0
	NOP 0
	NOP 0
	NOP 0
	NOP 0
	NOP 0
	NOP 0
	NOP 0
	NOP 0
	NOP 0
	NOP 0
	NOP 0
	NOP 0
	NOP 0
	NOP 0
	NOP 0
	NOP 0
	NOP 0
	NOP 0
	NOP 0
	NOP 0
	NOP 0
	NOP 0
	NOP 0
	NOP 0
	NOP 0
	NOP 0
	NOP 0
	NOP 0
	NOP 0
	NOP 0
	NOP 0
	NOP 0
	NOP 0
	NOP 0
	NOP 0
	NOP 0
	NOP 0
	NOP 0
	NOP 0
	NOP 0
	NOP 0
	NOP 0
	NOP 0
	NOP 0
	NOP 0
	NOP 0
	NOP 0
	NOP 0
	NOP 0
	NOP 0
	NOP 0
	NOP 0
	NOP 0
	NOP 0
	NOP 0
	NOP 0
	NOP 0
	NOP 0
	NOP 0
	NOP 0
	NOP 0
	NOP 0
	NOP 0
	NOP 0
	NOP 0
	NOP 0
	NOP 0
	NOP 0
	NOP 0
	NOP 0
	NOP 0
	NOP 0
	NOP 0
	NOP 0
	NOP 0
	NOP 0
	NOP 0
	NOP 0
	NOP 0
	NOP 0
	NOP 0
	NOP 0
	NOP 0
	NOP 0
	NOP 0
	NOP 0
	NOP 0
	NOP 0
	NOP 0
	NOP 0
	NOP 0
	NOP 0
	NOP 0
	NOP 0
	NOP 0
	NOP 0
	NOP 0
	NOP 0
	NOP 0
	NOP 0
	NOP 0
	NOP 0
	NOP 0
	NOP 0
	NOP 0
	NOP 0
	NOP 0
	NOP 0
	NOP 0
	NOP 0
	NOP 0
	NOP 0
	NOP 0
	NOP 0
	NOP 0
	NOP 0
	NOP 0
	NOP 0
	NOP 0
	NOP 0
	NOP 0
	NOP 0
	NOP 0
	NOP 0
	NOP 0
	NOP 0
	NOP 0
	NOP 0
	NOP 0
	NOP 0
	NOP 0
	NOP 0
	NOP 0
	NOP 0
	NOP 0
	NOP 0
	NOP 0
	NOP 0
	NOP 0
	NOP 0
	NOP 0
	NOP 0
	NOP 0
	NOP 0
	NOP 0
	NOP 0
	NOP 0
	NOP 0
	NOP 0
	NOP 0
	NOP 0
	NOP 0
	NOP 0
	NOP 0
	NOP 0
	NOP 0
	NOP 0
	NOP 0
	NOP 0
	NOP 0
	NOP 0
	NOP 0
	NOP 0
	NOP 0
	NOP 0
	NOP 0
	NOP 0
	NOP 0
	NOP 0
	NOP 0
	NOP 0
	NOP 0
	NOP 0
	NOP 0
	NOP 0
	NOP 0
	NOP 0
	NOP 0
	NOP 0
	NOP 0
	NOP 0
	NOP 0
	NOP 0
	NOP 0
	NOP 0
	NOP 0
	NOP 0
	NOP 0
	NOP 0
	NOP 0
	NOP 0
	NOP 0
	NOP 0
	NOP 0
	NOP 0
	NOP 0
	NOP 0
	NOP 0
	NOP 0
	NOP 0
	NOP 0
	NOP 0
	NOP 0
	NOP 0
	NOP 0
	NOP 0
	NOP 0
	NOP 0
	NOP 0
	NOP 0
	NOP 0
	NOP 0
	NOP 0
	NOP 0
	NOP 0
	NOP 0
	NOP 0
	NOP 0
	NOP 0
	NOP 0
	NOP 0
	NOP 0
	NOP 0
	NOP 0
	NOP 0
	NOP 0
	NOP 0
	NOP 0
	NOP 0
	NOP 0
	NOP 0
	NOP 0
	NOP 0
	NOP 0
	NOP 0
	NOP 0
	NOP 0
	NOP 0
	NOP 0
	NOP 0
	NOP 0
	NOP 0
	NOP 0
	NOP 0
	NOP 0
	NOP 0
	NOP 0
	NOP 0
	NOP 0
	NOP 0
	NOP 0
	NOP 0
	NOP 0
	NOP 0
	NOP 0
	NOP 0
	NOP 0
	NOP 0
	NOP 0
	NOP 0
	NOP 0
	NOP 0
	NOP 0
	NOP 0
	NOP 0
	NOP 0
	NOP 0
	NOP 0
	NOP 0
	NOP 0
	NOP 0
	NOP 0
	NOP 0
	NOP 0
	NOP 0
	NOP 0
	NOP 0
	NOP 0
	NOP 0
	NOP 0
	NOP 0
	NOP 0
	NOP 0
	NOP 0
	NOP 0
	NOP 0
	NOP 0
	NOP 0
	NOP 0
	NOP 0
	NOP 0
	NOP 0
	NOP 0
	NOP 0
	NOP 0
	NOP 0
	NOP 0
	NOP 0
	NOP 0
	NOP 0
	NOP 0
	NOP 0
	NOP 0
	NOP 0
	NOP 0
	NOP 0
	NOP 0
	NOP 0
	NOP 0
	NOP 0
	NOP 0
	NOP 0
	NOP 0
	NOP 0
	NOP 0
	NOP 0
	NOP 0
	NOP 0
	NOP 0
	NOP 0
	NOP 0
	NOP 0
	NOP 0
	NOP 0
	NOP 0
	NOP 0
	NOP 0
	NOP 0
	NOP 0
	NOP 0
	NOP 0
	NOP 0
	NOP 0
	NOP 0
	NOP 0
	NOP 0
	NOP 0
	NOP 0
	NOP 0
	NOP 0
	NOP 0
	NOP 0
	NOP 0
	NOP 0
	NOP 0
	NOP 0
	NOP 0
	NOP 0
	NOP 0
	NOP 0
	NOP 0
	NOP 0
	NOP 0
	NOP 0
	NOP 0
	NOP 0
	NOP 0
	NOP 0
	NOP 0
	NOP 0
	NOP 0
	NOP 0
	NOP 0
	NOP 0
	NOP 0
	NOP 0
	NOP 0
	NOP 0
	NOP 0
	NOP 0
	NOP 0
	NOP 0
	NOP 0
	NOP 0
	NOP 0
	NOP 0
	NOP 0
	NOP 0
	NOP 0
	NOP 0
	NOP 0
	NOP 0
	NOP 0
	NOP 0
	NOP 0
	NOP 0
	NOP 0
	NOP 0
	NOP 0
	NOP 0
	NOP 0
	NOP 0
	NOP 0
	NOP 0
	NOP 0
	NOP 0
	NOP 0
	NOP 0
	NOP 0
	NOP 0
	NOP 0
	NOP 0
	NOP 0
	NOP 0
	NOP 0
	NOP 0
	NOP 0
	NOP 0
	NOP 0
	NOP 0
	NOP 0
	NOP 0
	NOP 0
	NOP 0
	NOP 0
	NOP 0
	NOP 0
	NOP 0
	NOP 0
	NOP 0
	NOP 0
	NOP 0
	NOP 0
	NOP 0
	NOP 0
	NOP 0
	NOP 0
	NOP 0
	NOP 0
	NOP 0
	NOP 0
	NOP 0
	NOP 0
	NOP 0
	NOP 0
	NOP 0
	NOP 0
	NOP 0
	NOP 0
	NOP 0
	NOP 0
	NOP 0
	NOP 0
	NOP 0
	NOP 0
	NOP 0
	NOP 0
	NOP 0
	NOP 0
	NOP 0
	NOP 0
	NOP 0
	NOP 0
	NOP 0
	NOP 0
	NOP 0
	NOP 0
	NOP 0
	NOP 0
	NOP 0
	NOP 0
	NOP 0
	NOP 0
	NOP 0
	NOP 0
	NOP 0
	NOP 0
	NOP 0
	NOP 0
	NOP 0
	NOP 0
	NOP 0
	NOP 0
	NOP 0
	NOP 0
	NOP 0
	NOP 0
	NOP 0
	NOP 0
	NOP 0
	NOP 0
	NOP 0
	NOP 0
	NOP 0
	NOP 0
	NOP 0
	NOP 0
	NOP 0
	NOP 0
	NOP 0
	NOP 0
	NOP 0
	NOP 0
	NOP 0
	NOP 0
	NOP 0
	NOP 0
	NOP 0
	NOP 0
	NOP 0
	NOP 0
	NOP 0
	NOP 0
	NOP 0
	NOP 0
	NOP 0
	NOP 0
	NOP 0
	NOP 0
	NOP 0
	NOP 0
	NOP 0
	NOP 0
	NOP 0
	NOP 0
	NOP 0
	NOP 0
	NOP 0
	NOP 0
	NOP 0
	NOP 0
	NOP 0
	NOP 0
	NOP 0
	NOP 0
	NOP 0
	NOP 0
	NOP 0
	NOP 0
	NOP 0
	NOP 0
	NOP 0
	NOP 0
	NOP 0
	NOP 0
	NOP 0
	NOP 0
	NOP 0
	NOP 0
	NOP 0
	NOP 0
	NOP 0
	NOP 0
	NOP 0
	NOP 0
	NOP 0
	NOP 0
	NOP 0
	NOP 0
	NOP 0
	NOP 0
	NOP 0
	NOP 0
	NOP 0
	NOP 0
	NOP 0
	NOP 0
	NOP 0
	NOP 0
	NOP 0
	NOP 0
	NOP 0
	NOP 0
	NOP 0
	NOP 0
	NOP 0
	NOP 0
	NOP 0
	NOP 0
	NOP 0
	NOP 0
	NOP 0
	NOP 0
	NOP 0
	NOP 0
	NOP 0
	NOP 0
	NOP 0
	NOP 0
	NOP 0
	NOP 0
	NOP 0
	NOP 0
	NOP 0
	NOP 0
	NOP 0
	NOP 0
	NOP 0
	NOP 0
	NOP 0
	NOP 0
	NOP 0
	NOP 0
	NOP 0
	NOP 0
	NOP 0
	NOP 0
	NOP 0
	NOP 0
	NOP 0
	NOP 0
	NOP 0
	NOP 0
	NOP 0
	NOP 0
	NOP 0
	NOP 0
	NOP 0
	NOP 0
	NOP 0
	NOP 0
	NOP 0
	NOP 0
	NOP 0
	NOP 0
	NOP 0
	NOP 0
	NOP 0
	NOP 0
	NOP 0
	NOP 0
	NOP 0
	NOP 0
	NOP 0
	NOP 0
	NOP 0
	NOP 0
	NOP 0
	NOP 0
	NOP 0
	NOP 0
	NOP 0
	NOP 0
	NOP 0
	NOP 0
	NOP 0
	NOP 0
	NOP 0
	NOP 0
	NOP 0
	NOP 0
	NOP 0
	NOP 0
	NOP 0
	NOP 0
	NOP 0
	NOP 0
	NOP 0
	NOP 0
	NOP 0
	NOP 0
	NOP 0
	NOP 0
	NOP 0
	NOP 0
	NOP 0
	NOP 0
	NOP 0
	NOP 0
	NOP 0
	NOP 0
	NOP 0
	NOP 0
	NOP 0
	NOP 0
	NOP 0
	NOP 0
	NOP 0
	NOP 0
	NOP 0
	NOP 0
	NOP 0
	NOP 0
	NOP 0
	NOP 0
	NOP 0
	NOP 0
	NOP 0
	NOP 0
	NOP 0
	NOP 0
	NOP 0
	NOP 0
	NOP 0
	NOP 0
	NOP 0
	NOP 0
	NOP 0
	NOP 0
	NOP 0
	NOP 0
	NOP 0
	NOP 0
	NOP 0
	NOP 0
	NOP 0
	NOP 0
	NOP 0
	NOP 0
	NOP 0
	NOP 0
	NOP 0
	NOP 0
	NOP 0
	NOP 0
	NOP 0
	NOP 0
	NOP 0
	NOP 0
	NOP 0
	NOP 0
	NOP 0
	NOP 0
	NOP 0
	NOP 0
	NOP 0
	NOP 0
	NOP 0
	NOP 0
	NOP 0
	NOP 0
	NOP 0
	NOP 0
	NOP 0
	NOP 0
	NOP 0
	NOP 0
	NOP 0
	NOP 0
	NOP 0
	NOP 0
	NOP 0
	NOP 0
	NOP 0
	NOP 0
	NOP 0
	NOP 0
	NOP 0
	NOP 0
	NOP 0
	NOP 0
	NOP 0
	NOP 0
	NOP 0
	NOP 0
	NOP 0
	NOP 0
	NOP 0
	NOP 0
	NOP 0
	NOP 0
	NOP 0
	NOP 0
	NOP 0
	NOP 0
	NOP 0
	NOP 0
	NOP 0
	NOP 0
	NOP 0
	NOP 0
	NOP 0
	NOP 0
	NOP 0
	NOP 0
	NOP 0
	NOP 0
	NOP 0
	NOP 0
	NOP 0
	NOP 0
	NOP 0
	NOP 0
	NOP 0
	NOP 0
	NOP 0
	NOP 0
	NOP 0
	NOP 0
	NOP 0
	NOP 0
	NOP 0
	NOP 0
	NOP 0
	NOP 0
	NOP 0
	NOP 0
	NOP 0
	NOP 0
	NOP 0
	NOP 0
	NOP 0
	NOP 0
	NOP 0
	NOP 0
	NOP 0
	NOP 0
	NOP 0
	NOP 0
	NOP 0
	NOP 0
	NOP 0
	NOP 0
	NOP 0
	NOP 0
	NOP 0
	NOP 0
	NOP 0
	NOP 0
	NOP 0
	NOP 0
	NOP 0
	NOP 0
	NOP 0
	NOP 0
	NOP 0
	NOP 0
	NOP 0
	NOP 0
	NOP 0
	NOP 0
	NOP 0
	NOP 0
	NOP 0
	NOP 0
	NOP 0
	NOP 0
	NOP 0
	NOP 0
	NOP 0
	NOP 0
	NOP 0
	NOP 0
	NOP 0
	NOP 0
	NOP 0
	NOP 0
	NOP 0
	NOP 0
	NOP 0
	NOP 0
	NOP 0
	NOP 0
	NOP 0
	NOP 0
	NOP 0
	NOP 0
	NOP 0
	NOP 0
	NOP 0
	NOP 0
	NOP 0
	NOP 0
	NOP 0
	NOP 0
	NOP 0
	NOP 0
	NOP 0
	NOP 0
	NOP 0
	NOP 0
	NOP 0
	NOP 0
	NOP 0
	NOP 0
	NOP 0
	NOP 0
	NOP 0
	NOP 0
	NOP 0
	NOP 0
	NOP 0
	NOP 0
	NOP 0
	NOP 0
	NOP 0
	NOP 0
	NOP 0
	NOP 0
	NOP 0
	NOP 0
	NOP 0
	NOP 0
	NOP 0
	NOP 0
	NOP 0
	NOP 0
	NOP 0
	NOP 0
	NOP 0
	NOP 0
	NOP 0
	NOP 0
	NOP 0
	NOP 0
	NOP 0
	NOP 0
	NOP 0
	NOP 0
	NOP 0
	NOP 0
	NOP 0
	NOP 0
	NOP 0
	NOP 0
	NOP 0
	NOP 0
	NOP 0
	NOP 0
	NOP 0
	NOP 0
	NOP 0
	NOP 0
	NOP 0
	NOP 0
	NOP 0
	NOP 0
	NOP 0
	NOP 0
	NOP 0
	NOP 0
	NOP 0
	NOP 0
	NOP 0
	NOP 0
	NOP 0
	NOP 0
	NOP 0
	NOP 0
	NOP 0
	NOP 0
	NOP 0
	NOP 0
	NOP 0
	NOP 0
	NOP 0
	NOP 0
	NOP 0
	NOP 0
	NOP 0
	NOP 0
	NOP 0
	NOP 0
	NOP 0
	NOP 0
	NOP 0
	NOP 0
	NOP 0
	NOP 0
	NOP 0
	NOP 0
	NOP 0
	NOP 0
	NOP 0
	NOP 0
	NOP 0
	NOP 0
	NOP 0
	NOP 0
	NOP 0
	NOP 0
	NOP 0
	NOP 0
	NOP 0
	NOP 0
	NOP 0
	NOP 0
	NOP 0
	NOP 0
	NOP 0
	NOP 0
	NOP 0
	NOP 0
	NOP 0
	NOP 0
	NOP 0
	NOP 0
	NOP 0
	NOP 0
	NOP 0
	NOP 0
	NOP 0
	NOP 0
	NOP 0
	NOP 0
	NOP 0
	NOP 0
	NOP 0
	NOP 0
	NOP 0
	NOP 0
	NOP 0
	NOP 0
	NOP 0
	NOP 0
	NOP 0
	NOP 0
	NOP 0
	NOP 0
	NOP 0
	NOP 0
	NOP 0
	NOP 0
	NOP 0
	NOP 0
	NOP 0
	NOP 0
	NOP 0
	NOP 0
	NOP 0
	NOP 0
	NOP 0
	NOP 0
	NOP 0
	NOP 0
	NOP 0
	NOP 0
	NOP 0
	NOP 0
	NOP 0
	NOP 0
	NOP 0
	NOP 0
	NOP 0
	NOP 0
	NOP 0
	NOP 0
	NOP 0
	NOP 0
	NOP 0
	NOP 0
	NOP 0
	NOP 0
	NOP 0
	NOP 0
	NOP 0
	NOP 0
	NOP 0
	NOP 0
	NOP 0
	NOP 0
	NOP 0
	NOP 0
	NOP 0
	NOP 0
	NOP 0
	NOP 0
	NOP 0
	NOP 0
	NOP 0
	NOP 0
	NOP 0
	NOP 0
	NOP 0
	NOP 0
	NOP 0
	NOP 0
	NOP 0
	NOP 0
	NOP 0
	NOP 0
	NOP 0
	NOP 0
	NOP 0
	NOP 0
	NOP 0
	NOP 0
	NOP 0
	NOP 0
	NOP 0
	NOP 0
	NOP 0
	NOP 0
	NOP 0
	NOP 0
	NOP 0
	NOP 0
	NOP 0
	NOP 0
	NOP 0
	NOP 0
	NOP 0
	NOP 0
	NOP 0
	NOP 0
	NOP 0
	NOP 0
	NOP 0
	NOP 0
	NOP 0
	NOP 0
	NOP 0
	NOP 0
	NOP 0
	NOP 0
	NOP 0
	NOP 0
	NOP 0
	NOP 0
	NOP 0
	NOP 0
	NOP 0
	NOP 0
	NOP 0
	NOP 0
	NOP 0
	NOP 0
	NOP 0
	NOP 0
	NOP 0
	NOP 0
	NOP 0
	NOP 0
	NOP 0
	NOP 0
	NOP 0
	NOP 0
	NOP 0
	NOP 0
	NOP 0
	NOP 0
	NOP 0
	NOP 0
	NOP 0
	NOP 0
	NOP 0
	NOP 0
	NOP 0
	NOP 0
	NOP 0
	NOP 0
	NOP 0
	NOP 0
	NOP 0
	NOP 0
	NOP 0
	NOP 0
	NOP 0
	NOP 0
	NOP 0
	NOP 0
	NOP 0
	NOP 0
	NOP 0
	NOP 0
	NOP 0
	NOP 0
	NOP 0
	NOP 0
	NOP 0
	NOP 0
	NOP 0
	NOP 0
	NOP 0
	NOP 0
	NOP 0
	NOP 0
	NOP 0
	NOP 0
	NOP 0
	NOP 0
	NOP 0
	NOP 0
	NOP 0
	NOP 0
	NOP 0
	NOP 0
	NOP 0
	NOP 0
	NOP 0
	NOP 0
	NOP 0
	NOP 0
	NOP 0
	NOP 0
	NOP 0
	NOP 0
	NOP 0
	NOP 0
	NOP 0
	NOP 0
	NOP 0
	NOP 0
	NOP 0
	NOP 0
	NOP 0
	NOP 0
	NOP 0
	NOP 0
	NOP 0
	NOP 0
	NOP 0
	NOP 0
	NOP 0
	NOP 0
	NOP 0
	NOP 0
	NOP 0
	NOP 0
	NOP 0
	NOP 0
	NOP 0
	NOP 0
	NOP 0
	NOP 0
	NOP 0
	NOP 0
	NOP 0
	NOP 0
	NOP 0
	NOP 0
	NOP 0
	NOP 0
	NOP 0
	NOP 0
	NOP 0
	NOP 0
	NOP 0
	NOP 0
	NOP 0
	NOP 0
	NOP 0
	NOP 0
	NOP 0
	NOP 0
	NOP 0
	NOP 0
	NOP 0
	NOP 0
	NOP 0
	NOP 0
	NOP 0
	NOP 0
	NOP 0
	NOP 0
	NOP 0
	NOP 0
	NOP 0
	NOP 0
	NOP 0
	NOP 0
	NOP 0
	NOP 0
	NOP 0
	NOP 0
	NOP 0
	NOP 0
	NOP 0
	NOP 0
	NOP 0
	NOP 0
	NOP 0
	NOP 0
	NOP 0
	NOP 0
	NOP 0
	NOP 0
	NOP 0
	NOP 0
	NOP 0
	NOP 0
	NOP 0
	NOP 0
	NOP 0
	NOP 0
	NOP 0
	NOP 0
	NOP 0
	NOP 0
	NOP 0
	NOP 0
	NOP 0
	NOP 0
	NOP 0
	NOP 0
	NOP 0
	NOP 0
	NOP 0
	NOP 0
	NOP 0
	NOP 0
	NOP 0
	NOP 0
	NOP 0
	NOP 0
	NOP 0
	NOP 0
	NOP 0
	NOP 0
	NOP 0
	NOP 0
	NOP 0
	NOP 0
	NOP 0
	NOP 0
	NOP 0
	NOP 0
	NOP 0
	NOP 0
	NOP 0
	NOP 0
	NOP 0
	NOP 0
	NOP 0
	NOP 0
	NOP 0
	NOP 0
	NOP 0
	NOP 0
	NOP 0
	NOP 0
	NOP 0
	NOP 0
	NOP 0
	NOP 0
	NOP 0
	NOP 0
	NOP 0
	NOP 0
	NOP 0
	NOP 0
	NOP 0
	NOP 0
	NOP 0
	NOP 0
	NOP 0
	NOP 0
	NOP 0
	NOP 0
	NOP 0
	NOP 0
	NOP 0
	NOP 0
	NOP 0
	NOP 0
	NOP 0
	NOP 0
	NOP 0
	NOP 0
	NOP 0
	NOP 0
	NOP 0
	NOP 0
	NOP 0
	NOP 0
	NOP 0
	NOP 0
	NOP 0
	NOP 0
	NOP 0
	NOP 0
	NOP 0
	NOP 0
	NOP 0
	NOP 0
	NOP 0
	NOP 0
	NOP 0
	NOP 0
	NOP 0
	NOP 0
	NOP 0
	NOP 0
	NOP 0
	NOP 0
	NOP 0
	NOP 0
	NOP 0
	NOP 0
	NOP 0
	NOP 0
	NOP 0
	NOP 0
	NOP 0
	NOP 0
	NOP 0
	NOP 0
	NOP 0
	NOP 0
	NOP 0
	NOP 0
	NOP 0
	NOP 0
	NOP 0
	NOP 0
	NOP 0
	NOP 0
	NOP 0
	NOP 0
	NOP 0
	NOP 0
	NOP 0
	NOP 0
	NOP 0
	NOP 0
	NOP 0
	NOP 0
	NOP 0
	NOP 0
	NOP 0
	NOP 0
	NOP 0
	NOP 0
	NOP 0
	NOP 0
	NOP 0
	NOP 0
	NOP 0
	NOP 0
	NOP 0
	NOP 0
	NOP 0
	NOP 0
	NOP 0
	NOP 0
	NOP 0
	NOP 0
	NOP 0
	NOP 0
	NOP 0
	NOP 0
	NOP 0
	NOP 0
	NOP 0
	NOP 0
	NOP 0
	NOP 0
	NOP 0
	NOP 0
	NOP 0
	NOP 0
	NOP 0
	NOP 0
	NOP 0
	NOP 0
	NOP 0
	NOP 0
	NOP 0
	NOP 0
	NOP 0
	NOP 0
	NOP 0
	NOP 0
	NOP 0
	NOP 0
	NOP 0
	NOP 0
	NOP 0
	NOP 0
	NOP 0
	NOP 0
	NOP 0
	NOP 0
	NOP 0
	NOP 0
	NOP 0
	NOP 0
	NOP 0
	NOP 0
	NOP 0
	NOP 0
	NOP 0
	NOP 0
	NOP 0
	NOP 0
	NOP 0
	NOP 0
	NOP 0
	NOP 0
	NOP 0
	NOP 0
	NOP 0
	NOP 0
	NOP 0
	NOP 0
	NOP 0
	NOP 0
	NOP 0
	NOP 0
	NOP 0
	NOP 0
	NOP 0
	NOP 0
	NOP 0
	NOP 0
	NOP 0
	NOP 0
	NOP 0
	NOP 0
	NOP 0
	NOP 0
	NOP 0
	NOP 0
	NOP 0
	NOP 0
	NOP 0
	NOP 0
	NOP 0
	NOP 0
	NOP 0
	NOP 0
	NOP 0
	NOP 0
	NOP 0
	NOP 0
	NOP 0
	NOP 0
	NOP 0
	NOP 0
	NOP 0
	NOP 0
	NOP 0
	NOP 0
	NOP 0
	NOP 0
	NOP 0
	NOP 0
	NOP 0
	NOP 0
	NOP 0
	NOP 0
	NOP 0
	NOP 0
	NOP 0
	NOP 0
	NOP 0
	NOP 0
	NOP 0
	NOP 0
	NOP 0
	NOP 0
	NOP 0
	NOP 0
	NOP 0
	NOP 0
	NOP 0
	NOP 0
	NOP 0
	NOP 0
	NOP 0
	NOP 0
	NOP 0
	NOP 0
	NOP 0
	NOP 0
	NOP 0
	NOP 0
	NOP 0
	NOP 0
	NOP 0
	NOP 0
	NOP 0
	NOP 0
	NOP 0
	NOP 0
	NOP 0
	NOP 0
	NOP 0
	NOP 0
	NOP 0
	NOP 0
	NOP 0
	NOP 0
	NOP 0
	NOP 0
	NOP 0
	NOP 0
	NOP 0
	NOP 0
	NOP 0
	NOP 0
	NOP 0
	NOP 0
	NOP 0
	NOP 0
	NOP 0
	NOP 0
	NOP 0
	NOP 0
	NOP 0
	NOP 0
	NOP 0
	NOP 0
	NOP 0
	NOP 0
	NOP 0
	NOP 0
	NOP 0
	NOP 0
	NOP 0
	NOP 0
	NOP 0
	NOP 0
	NOP 0
	NOP 0
	NOP 0
	NOP 0
	NOP 0
	NOP 0
	NOP 0
	NOP 0
	NOP 0
	NOP 0
	NOP 0
	NOP 0
	NOP 0
	NOP 0
	NOP 0
	NOP 0
	NOP 0
	NOP 0
	NOP 0
	NOP 0
	NOP 0
	NOP 0
	NOP 0
	NOP 0
	NOP 0
	NOP 0
	NOP 0
	NOP 0
	NOP 0
	NOP 0
	NOP 0
	NOP 0
	NOP 0
	NOP 0
	NOP 0
	NOP 0
	NOP 0
	NOP 0
	NOP 0
	NOP 0
	NOP 0
	NOP 0
	NOP 0
	NOP 0
	NOP 0
	NOP 0
	NOP 0
	NOP 0
	NOP 0
	NOP 0
	NOP 0
	NOP 0
	NOP 0
	NOP 0
	NOP 0
	NOP 0
	NOP 0
	NOP 0
	NOP 0
	NOP 0
	NOP 0
	NOP 0
	NOP 0
	NOP 0
	NOP 0
	NOP 0
	NOP 0
	NOP 0
	NOP 0
	NOP 0
	NOP 0
	NOP 0
	NOP 0
	NOP 0
	NOP 0
	NOP 0
	NOP 0
	NOP 0
	NOP 0
	NOP 0
	NOP 0
	NOP 0
	NOP 0
	NOP 0
	NOP 0
	NOP 0
	NOP 0
	NOP 0
	NOP 0
	NOP 0
	NOP 0
	NOP 0
	NOP 0
	NOP 0
	NOP 0
	NOP 0
	NOP 0
	NOP 0
	NOP 0
	NOP 0
	NOP 0
	NOP 0
	NOP 0
	NOP 0
	NOP 0
	NOP 0
	NOP 0
	NOP 0
	NOP 0
	NOP 0
	NOP 0
	NOP 0
	NOP 0
	NOP 0
	NOP 0
	NOP 0
	NOP 0
	NOP 0
	NOP 0
	NOP 0
	NOP 0
	NOP 0
	NOP 0
	NOP 0
	NOP 0
	NOP 0
	NOP 0
	NOP 0
	NOP 0
	NOP 0
	NOP 0
	NOP 0
	NOP 0
	NOP 0
	NOP 0
	NOP 0
	NOP 0
	NOP 0
	NOP 0
	NOP 0
	NOP 0
	NOP 0
	NOP 0
	NOP 0
	NOP 0
	NOP 0
	NOP 0
	NOP 0
	NOP 0
	NOP 0
	NOP 0
	NOP 0
	NOP 0
	NOP 0
	NOP 0
	NOP 0
	NOP 0
	NOP 0
	NOP 0
	NOP 0
	NOP 0
	NOP 0
	NOP 0
	NOP 0
	NOP 0
	NOP 0
	NOP 0
	NOP 0
	NOP 0
	NOP 0
	NOP 0
	NOP 0
	NOP 0
	NOP 0
	NOP 0
	NOP 0
	NOP 0
	NOP 0
	NOP 0
	NOP 0
	NOP 0
	NOP 0
	NOP 0
	NOP 0
	NOP 0
	NOP 0
	NOP 0
	NOP 0
	NOP 0
	NOP 0
	NOP 0
	NOP 0
	NOP 0
	NOP 0
	NOP 0
	NOP 0
	NOP 0
	NOP 0
	NOP 0
	NOP 0
	NOP 0
	NOP 0
	NOP 0
	NOP 0
	NOP 0
	NOP 0
	NOP 0
	NOP 0
	NOP 0
	NOP 0
	NOP 0
	NOP 0
	NOP 0
	NOP 0
	NOP 0
	NOP 0
	NOP 0
	NOP 0
	NOP 0
	NOP 0
	NOP 0
	NOP 0
	NOP 0
	NOP 0
	NOP 0
	NOP 0
	NOP 0
	NOP 0
	NOP 0
	NOP 0
	NOP 0
	NOP 0
	NOP 0
	NOP 0
	NOP 0
	NOP 0
	NOP 0
	NOP 0
	NOP 0
	NOP 0
	NOP 0
	NOP 0
	NOP 0
	NOP 0
	NOP 0
	NOP 0
	NOP 0
	NOP 0
	NOP 0
	NOP 0
	NOP 0
	NOP 0
	NOP 0
	NOP 0
	NOP 0
	NOP 0
	NOP 0
	NOP 0
	NOP 0
	NOP 0
	NOP 0
	NOP 0
	NOP 0
	NOP 0
	NOP 0
	NOP 0
	NOP 0
	NOP 0
	NOP 0
	NOP 0
	NOP 0
	NOP 0
	NOP 0
	NOP 0
	NOP 0
	NOP 0
	NOP 0
	NOP 0
	NOP 0
	NOP 0
	NOP 0
	NOP 0
	NOP 0
	NOP 0
	NOP 0
	NOP 0
	NOP 0
	NOP 0
	NOP 0
	NOP 0
	NOP 0
	NOP 0
	NOP 0
	NOP 0
	NOP 0
	NOP 0
	NOP 0
	NOP 0
	NOP 0
	NOP 0
	NOP 0
	NOP 0
	NOP 0
	NOP 0
	NOP 0
	NOP 0
	NOP 0
	NOP 0
	NOP 0
	NOP 0
	NOP 0
	NOP 0
	NOP 0
	NOP 0
	NOP 0
	NOP 0
	NOP 0
	NOP 0
	NOP 0
	NOP 0
	NOP 0
	NOP 0
	NOP 0
	NOP 0
	NOP 0
	NOP 0
	NOP 0
	NOP 0
	NOP 0
	NOP 0
	NOP 0
	NOP 0
	NOP 0
	NOP 0
	NOP 0
	NOP 0
	NOP 0
	NOP 0
	NOP 0
	NOP 0
	NOP 0
	NOP 0
	NOP 0
	NOP 0
	NOP 0
	NOP 0
	NOP 0
	NOP 0
	NOP 0
	NOP 0
	NOP 0
	NOP 0
	NOP 0
	NOP 0
	NOP 0
	NOP 0
	NOP 0
	NOP 0
	NOP 0
	NOP 0
	NOP 0
	NOP 0
	NOP 0
	NOP 0
	NOP 0
	NOP 0
	NOP 0
	NOP 0
	NOP 0
	NOP 0
	NOP 0
	NOP 0
	NOP 0
	NOP 0
	NOP 0
	NOP 0
	NOP 0
	NOP 0
	NOP 0
	NOP 0
	NOP 0
	NOP 0
	NOP 0
	NOP 0
	NOP 0
	NOP 0
	NOP 0
	NOP 0
	NOP 0
	NOP 0
	NOP 0
	NOP 0
	NOP 0
	NOP 0
	NOP 0
	NOP 0
	NOP 0
	NOP 0
	NOP 0
	NOP 0
	NOP 0
	NOP 0
	NOP 0
	NOP 0
	NOP 0
	NOP 0
	NOP 0
	NOP 0
	NOP 0
	NOP 0
	NOP 0
	NOP 0
	NOP 0
	NOP 0
	NOP 0
	NOP 0
	NOP 0
	NOP 0
	NOP 0
	NOP 0
	NOP 0
	NOP 0
	NOP 0
	NOP 0
	NOP 0
	NOP 0
	NOP 0
	NOP 0
	NOP 0
	NOP 0
	NOP 0
	NOP 0
	NOP 0
	NOP 0
	NOP 0
	NOP 0
	NOP 0
	NOP 0
	NOP 0
	NOP 0
	NOP 0
	NOP 0
	NOP 0
	NOP 0
	NOP 0
	NOP 0
	NOP 0
	NOP 0
	NOP 0
	NOP 0
	NOP 0
	NOP 0
	NOP 0
	NOP 0
	NOP 0
	NOP 0
	NOP 0
	NOP 0
	NOP 0
	NOP 0
	NOP 0
	NOP 0
	NOP 0
	NOP 0
	NOP 0
	NOP 0
	NOP 0
	NOP 0
	NOP 0
	NOP 0
	NOP 0
	NOP 0
	NOP 0
	NOP 0
	NOP 0
	NOP 0
	NOP 0
	NOP 0
	NOP 0
	NOP 0
	NOP 0
	NOP 0
	NOP 0
	NOP 0
	NOP 0
	NOP 0
	NOP 0
	NOP 0
	NOP 0
	NOP 0
	NOP 0
	NOP 0
	NOP 0
	NOP 0
	NOP 0
	NOP 0
	NOP 0
	NOP 0
	NOP 0
	NOP 0
	NOP 0
	NOP 0
	NOP 0
	NOP 0
	NOP 0
	NOP 0
	NOP 0
	NOP 0
	NOP 0
	NOP 0
	NOP 0
	NOP 0
	NOP 0
	NOP 0
	NOP 0
	NOP 0
	NOP 0
	NOP 0
	NOP 0
	NOP 0
	NOP 0
	NOP 0
	NOP 0
	NOP 0
	NOP 0
	NOP 0
	NOP 0
	NOP 0
	NOP 0
	NOP 0
	NOP 0
	NOP 0
	NOP 0
	NOP 0
	NOP 0
	NOP 0
	NOP 0
	NOP 0
	NOP 0
	NOP 0
	NOP 0
	NOP 0
	NOP 0
	NOP 0
	NOP 0
	NOP 0
	NOP 0
	NOP 0
	NOP 0
	NOP 0
	NOP 0
	NOP 0
	NOP 0
	NOP 0
	NOP 0
	NOP 0
	NOP 0
	NOP 0
	NOP 0
	NOP 0
	NOP 0
	NOP 0
	NOP 0
	NOP 0
	NOP 0
	NOP 0
	NOP 0
	NOP 0
	NOP 0
	NOP 0
	NOP 0
	NOP 0
	NOP 0
	NOP 0
	NOP 0
	NOP 0
	NOP 0
	NOP 0
	NOP 0
	NOP 0
	NOP 0
	NOP 0
	NOP 0
	NOP 0
	NOP 0
	NOP 0
	NOP 0
	NOP 0
	NOP 0
	NOP 0
	NOP 0
	NOP 0
	NOP 0
	NOP 0
	NOP 0
	NOP 0
	NOP 0
	NOP 0
	NOP 0
	NOP 0
	NOP 0
	NOP 0
	NOP 0
	NOP 0
	NOP 0
	NOP 0
	NOP 0
	NOP 0
	NOP 0
	NOP 0
	NOP 0
	NOP 0
	NOP 0
	NOP 0
	NOP 0
	NOP 0
	NOP 0
	NOP 0
	NOP 0
	NOP 0
	NOP 0
	NOP 0
	NOP 0
	NOP 0
	NOP 0
	NOP 0
	NOP 0
	NOP 0
	NOP 0
	NOP 0
	NOP 0
	NOP 0
	NOP 0
	NOP 0
	NOP 0
	NOP 0
	NOP 0
	NOP 0
	NOP 0
	NOP 0
	NOP 0
	NOP 0
	NOP 0
	NOP 0
	NOP 0
	NOP 0
	NOP 0
	NOP 0
	NOP 0
	NOP 0
	NOP 0
	NOP 0
	NOP 0
	NOP 0
	NOP 0
	NOP 0
	NOP 0
	NOP 0
	NOP 0
	NOP 0
	NOP 0
	NOP 0
	NOP 0
	NOP 0
	NOP 0
	NOP 0
	NOP 0
	NOP 0
	NOP 0
	NOP 0
	NOP 0
	NOP 0
	NOP 0
	NOP 0
	NOP 0
	NOP 0
	NOP 0
	NOP 0
	NOP 0
	NOP 0
	NOP 0
	NOP 0
	NOP 0
	NOP 0
	NOP 0
	NOP 0
	NOP 0
	NOP 0
	NOP 0
	NOP 0
	NOP 0
	NOP 0
	NOP 0
	NOP 0
	NOP 0
	NOP 0
	NOP 0
	NOP 0
	NOP 0
	NOP 0
	NOP 0
	NOP 0
	NOP 0
	NOP 0
	NOP 0
	NOP 0
	NOP 0
	NOP 0
	NOP 0
	NOP 0
	NOP 0
	NOP 0
	NOP 0
	NOP 0
	NOP 0
	NOP 0
	NOP 0
	NOP 0
	NOP 0
	NOP 0
	NOP 0
	NOP 0
	NOP 0
	NOP 0
	NOP 0
	NOP 0
	NOP 0
	NOP 0
	NOP 0
	NOP 0
	NOP 0
	NOP 0
	NOP 0
	NOP 0
	NOP 0
	NOP 0
	NOP 0
	NOP 0
	NOP 0
	NOP 0
	NOP 0
	NOP 0
	NOP 0
	NOP 0
	NOP 0
	NOP 0
	NOP 0
	NOP 0
	NOP 0
	NOP 0
	NOP 0
	NOP 0
	NOP 0
	NOP 0
	NOP 0
	NOP 0
	NOP 0
	NOP 0
	NOP 0
	NOP 0
	NOP 0
	NOP 0
	NOP 0
	NOP 0
	NOP 0
	NOP 0
	NOP 0
	NOP 0
	NOP 0
	NOP 0
	NOP 0
	NOP 0
	NOP 0
	NOP 0
	NOP 0
	NOP 0
	NOP 0
	NOP 0
	NOP 0
	NOP 0
	NOP 0
	NOP 0
	NOP 0
	NOP 0
	NOP 0
	NOP 0
	NOP 0
	NOP 0
	NOP 0
	NOP 0
	NOP 0
	NOP 0
	NOP 0
	NOP 0
	NOP 0
	NOP 0
	NOP 0
	NOP 0
	NOP 0
	NOP 0
	NOP 0
	NOP 0
	NOP 0
	NOP 0
	NOP 0
	NOP 0
	NOP 0
	NOP 0
	NOP 0
	NOP 0
	NOP 0
	NOP 0
	NOP 0
	NOP 0
	NOP 0
	NOP 0
	NOP 0
	NOP 0
	NOP 0
	NOP 0
	NOP 0
	NOP 0
	NOP 0
	NOP 0
	NOP 0
	NOP 0
	NOP 0
	NOP 0
	NOP 0
	NOP 0
	NOP 0
	NOP 0
	NOP 0
	NOP 0
	NOP 0
	NOP 0
	NOP 0
	NOP 0
	NOP 0
	NOP 0
	NOP 0
	NOP 0
	NOP 0
	NOP 0
	NOP 0
	NOP 0
	NOP 0
	NOP 0
	NOP 0
	NOP 0
	NOP 0
	NOP 0
	NOP 0
	NOP 0
	NOP 0
	NOP 0
	NOP 0
	NOP 0
	NOP 0
	NOP 0
	NOP 0
	NOP 0
	NOP 0
	NOP 0
	NOP 0
	NOP 0
	NOP 0
	NOP 0
	NOP 0
	NOP 0
	NOP 0
	NOP 0
	NOP 0
	NOP 0
	NOP 0
	NOP 0
	NOP 0
	NOP 0
	NOP 0
	NOP 0
	NOP 0
	NOP 0
	NOP 0
	NOP 0
	NOP 0
	NOP 0
	NOP 0
	NOP 0
	NOP 0
	NOP 0
	NOP 0
	NOP 0
	NOP 0
	NOP 0
	NOP 0
	NOP 0
	NOP 0
	NOP 0
	NOP 0
	NOP 0
	NOP 0
	NOP 0
	NOP 0
	NOP 0
	NOP 0
	NOP 0
	NOP 0
	NOP 0
	NOP 0
	NOP 0
	NOP 0
	NOP 0
	NOP 0
	NOP 0
	NOP 0
	NOP 0
	NOP 0
	NOP 0
	NOP 0
	NOP 0
	NOP 0
	NOP 0
	NOP 0
	NOP 0
	NOP 0
	NOP 0
	NOP 0
	NOP 0
	NOP 0
	NOP 0
	NOP 0
	NOP 0
	NOP 0
	NOP 0
	NOP 0
	NOP 0
	NOP 0
	NOP 0
	NOP 0
	NOP 0
	NOP 0
	NOP 0
	NOP 0
	NOP 0
	NOP 0
	NOP 0
	NOP 0
	NOP 0
	NOP 0
	NOP 0
	NOP 0
	NOP 0
	NOP 0
	NOP 0
	NOP 0
	NOP 0
	NOP 0
	NOP 0
	NOP 0
	NOP 0
	NOP 0
	NOP 0
	NOP 0
	NOP 0
	NOP 0
	NOP 0
	NOP 0
	NOP 0
	NOP 0
	NOP 0
	NOP 0
	NOP 0
	NOP 0
	NOP 0
	NOP 0
	NOP 0
	NOP 0
	NOP 0
	NOP 0
	NOP 0
	NOP 0
	NOP 0
	NOP 0
	NOP 0
	NOP 0
	NOP 0
	NOP 0
	NOP 0
	NOP 0
	NOP 0
	NOP 0
	NOP 0
	NOP 0
	NOP 0
	NOP 0
	NOP 0
	NOP 0
	NOP 0
	NOP 0
	NOP 0
	NOP 0
	NOP 0
	NOP 0
	NOP 0
	NOP 0
	NOP 0
	NOP 0
	NOP 0
	NOP 0
	NOP 0
	NOP 0
	NOP 0
	NOP 0
	NOP 0
	NOP 0
	NOP 0
	NOP 0
	NOP 0
	NOP 0
	NOP 0
	NOP 0
	NOP 0
	NOP 0
	NOP 0
	NOP 0
	NOP 0
	NOP 0
	NOP 0
	NOP 0
	NOP 0
	NOP 0
	NOP 0
	NOP 0
	NOP 0
	NOP 0
	NOP 0
	NOP 0
	NOP 0
	NOP 0
	NOP 0
	NOP 0
	NOP 0
	NOP 0
	NOP 0
	NOP 0
	NOP 0
	NOP 0
	NOP 0
	NOP 0
	NOP 0
	NOP 0
	NOP 0
	NOP 0
	NOP 0
	NOP 0
	NOP 0
	NOP 0
	NOP 0
	NOP 0
	NOP 0
	NOP 0
	NOP 0
	NOP 0
	NOP 0
	NOP 0
	NOP 0
	NOP 0
	NOP 0
	NOP 0
	NOP 0
	NOP 0
	NOP 0
	NOP 0
	NOP 0
	NOP 0
	NOP 0
	NOP 0
	NOP 0
	NOP 0
	NOP 0
	NOP 0
	NOP 0
	NOP 0
	NOP 0
	NOP 0
	NOP 0
	NOP 0
	NOP 0
	NOP 0
	NOP 0
	NOP 0
	NOP 0
	NOP 0
	NOP 0
	NOP 0
	NOP 0
	NOP 0
	NOP 0
	NOP 0
	NOP 0
	NOP 0
	NOP 0
	NOP 0
	NOP 0
	NOP 0
	NOP 0
	NOP 0
	NOP 0
	NOP 0
	NOP 0
	NOP 0
	NOP 0
	NOP 0
	NOP 0
	NOP 0
	NOP 0
	NOP 0
	NOP 0
	NOP 0
	NOP 0
	NOP 0
	NOP 0
	NOP 0
	NOP 0
	NOP 0
	NOP 0
	NOP 0
	NOP 0
	NOP 0
	NOP 0
	NOP 0
	NOP 0
	NOP 0
	NOP 0
	NOP 0
	NOP 0
	NOP 0
	NOP 0
	NOP 0
	NOP 0
	NOP 0
	NOP 0
	NOP 0
	NOP 0
	NOP 0
	NOP 0
	NOP 0
	NOP 0
	NOP 0
	NOP 0
	NOP 0
	NOP 0
	NOP 0
	NOP 0
	NOP 0
	NOP 0
	NOP 0
	NOP 0
	NOP 0
	NOP 0
	NOP 0
	NOP 0
	NOP 0
	NOP 0
	NOP 0
	NOP 0
	NOP 0
	NOP 0
	NOP 0
	NOP 0
	NOP 0
	NOP 0
	NOP 0
	NOP 0
	NOP 0
	NOP 0
	NOP 0
	NOP 0
	NOP 0
	NOP 0
	NOP 0
	NOP 0
	NOP 0
	NOP 0
	NOP 0
	NOP 0
	NOP 0
	NOP 0
	NOP 0
	NOP 0
	NOP 0
	NOP 0
	NOP 0
	NOP 0
	NOP 0
	NOP 0
	NOP 0
	NOP 0
	NOP 0
	NOP 0
	NOP 0
	NOP 0
	NOP 0
	NOP 0
	NOP 0
	NOP 0
	NOP 0
	NOP 0
	NOP 0
	NOP 0
	NOP 0
	NOP 0
	NOP 0
	NOP 0
	NOP 0
	NOP 0
	NOP 0
	NOP 0
	NOP 0
	NOP 0
	NOP 0
	NOP 0
	NOP 0
	NOP 0
	NOP 0
	NOP 0
	NOP 0
	NOP 0
	NOP 0
	NOP 0
	NOP 0
	NOP 0
	NOP 0
	NOP 0
	NOP 0
	NOP 0
	NOP 0
	NOP 0
	NOP 0
	NOP 0
	NOP 0
	NOP 0
	NOP 0
	NOP 0
	NOP 0
	NOP 0
	NOP 0
	NOP 0
	NOP 0
	NOP 0
	NOP 0
	NOP 0
	NOP 0
	NOP 0
	NOP 0
	NOP 0
	NOP 0
	NOP 0
	NOP 0
	NOP 0
	NOP 0
	NOP 0
	NOP 0
	NOP 0
	NOP 0
	NOP 0
	NOP 0
	NOP 0
	NOP 0
	NOP 0
	NOP 0
	NOP 0
	NOP 0
	NOP 0
	NOP 0
	NOP 0
	NOP 0
	NOP 0
	NOP 0
	NOP 0
	NOP 0
	NOP 0
	NOP 0
	NOP 0
	NOP 0
	NOP 0
	NOP 0
	NOP 0
	NOP 0
	NOP 0
	NOP 0
	NOP 0
	NOP 0
	NOP 0
	NOP 0
	NOP 0
	NOP 0
	NOP 0
	NOP 0
	NOP 0
	NOP 0
	NOP 0
	NOP 0
	NOP 0
	NOP 0
	NOP 0
	NOP 0
	NOP 0
	NOP 0
	NOP 0
	NOP 0
	NOP 0
	NOP 0
	NOP 0
	NOP 0
	NOP 0
	NOP 0
	NOP 0
	NOP 0
	NOP 0
	NOP 0
	NOP 0
	NOP 0
	NOP 0
	NOP 0
	NOP 0
	NOP 0
	NOP 0
	NOP 0
	NOP 0
	NOP 0
	NOP 0
	NOP 0
	NOP 0
	NOP 0
	NOP 0
	NOP 0
	NOP 0
	NOP 0
	NOP 0
	NOP 0
	NOP 0
	NOP 0
	NOP 0
	NOP 0
	NOP 0
	NOP 0
	NOP 0
	NOP 0
	NOP 0
	NOP 0
	NOP 0
	NOP 0
	NOP 0
	NOP 0
	NOP 0
	NOP 0
	NOP 0
	NOP 0
	NOP 0
	NOP 0
	NOP 0
	NOP 0
	NOP 0
	NOP 0
	NOP 0
	NOP 0
	NOP 0
	NOP 0
	NOP 0
	NOP 0
	NOP 0
	NOP 0
	NOP 0
	NOP 0
	NOP 0
	NOP 0
	NOP 0
	NOP 0
	NOP 0
	NOP 0
	NOP 0
	NOP 0
	NOP 0
	NOP 0
	NOP 0
	NOP 0
	NOP 0
	NOP 0
	NOP 0
	NOP 0
	NOP 0
	NOP 0
	NOP 0
	NOP 0
	NOP 0
	NOP 0
	NOP 0
	NOP 0
	NOP 0
	NOP 0
	NOP 0
	NOP 0
	NOP 0
	NOP 0
	NOP 0
	NOP 0
	NOP 0
	NOP 0
	NOP 0
	NOP 0
	NOP 0
	NOP 0
	NOP 0
	NOP 0
	NOP 0
	NOP 0
	NOP 0
	NOP 0
	NOP 0
	NOP 0
	NOP 0
	NOP 0
	NOP 0
	NOP 0
	NOP 0
	NOP 0
	NOP 0
	NOP 0
	NOP 0
	NOP 0
	NOP 0
	NOP 0
	NOP 0
	NOP 0
	NOP 0
	NOP 0
	NOP 0
	NOP 0
	NOP 0
	NOP 0
	NOP 0
	NOP 0
	NOP 0
	NOP 0
	NOP 0
	NOP 0
	NOP 0
	NOP 0
	NOP 0
	NOP 0
	NOP 0
	NOP 0
	NOP 0
	NOP 0
	NOP 0
	NOP 0
	NOP 0
	NOP 0
	NOP 0
	NOP 0
	NOP 0
	NOP 0
	NOP 0
	NOP 0
	NOP 0
	NOP 0
	NOP 0
	NOP 0
	NOP 0
	NOP 0
	NOP 0
	NOP 0
	NOP 0
	NOP 0
	NOP 0
	NOP 0
	NOP 0
	NOP 0
	NOP 0
	NOP 0
	NOP 0
	NOP 0
	NOP 0
	NOP 0
	NOP 0
	NOP 0
	NOP 0
	NOP 0
	NOP 0
	NOP 0
	NOP 0
	NOP 0
	NOP 0
	NOP 0
	NOP 0
	NOP 0
	NOP 0
	NOP 0
	NOP 0
	NOP 0
	NOP 0
	NOP 0
	NOP 0
	NOP 0
	NOP 0
	NOP 0
	NOP 0
	NOP 0
	NOP 0
	NOP 0
	NOP 0
	NOP 0
	NOP 0
	NOP 0
	NOP 0
	NOP 0
	NOP 0
	NOP 0
	NOP 0
	NOP 0
	NOP 0
	NOP 0
	NOP 0
	NOP 0
	NOP 0
	NOP 0
	NOP 0
	NOP 0
	NOP 0
	NOP 0
	NOP 0
	NOP 0
	NOP 0
	NOP 0
	NOP 0
	NOP 0
	NOP 0
	NOP 0
	NOP 0
	NOP 0
	NOP 0
	NOP 0
	NOP 0
	NOP 0
	NOP 0
	NOP 0
	NOP 0
	NOP 0
	NOP 0
	NOP 0
	NOP 0
	NOP 0
	NOP 0
	NOP 0
	NOP 0
	NOP 0
	NOP 0
	NOP 0
	NOP 0
	NOP 0
	NOP 0
	NOP 0
	NOP 0
	NOP 0
	NOP 0
	NOP 0
	NOP 0
	NOP 0
	NOP 0
	NOP 0
	NOP 0
	NOP 0
	NOP 0
	NOP 0
	NOP 0
	NOP 0
	NOP 0
	NOP 0
	NOP 0
	NOP 0
	NOP 0
	NOP 0
	NOP 0
	NOP 0
	NOP 0
	NOP 0
	NOP 0
	NOP 0
	NOP 0
	NOP 0
	NOP 0
	NOP 0
	NOP 0
	NOP 0
	NOP 0
	NOP 0
	NOP 0
	NOP 0
	NOP 0
	NOP 0
	NOP 0
	NOP 0
	NOP 0
	NOP 0
	NOP 0
	NOP 0
	NOP 0
	NOP 0
	NOP 0
	NOP 0
	NOP 0
	NOP 0
	NOP 0
	NOP 0
	NOP 0
	NOP 0
	NOP 0
	NOP 0
	NOP 0
	NOP 0
	NOP 0
	NOP 0
	NOP 0
	NOP 0
	NOP 0
	NOP 0
	NOP 0
	NOP 0
	NOP 0
	NOP 0
	NOP 0
	NOP 0
	NOP 0
	NOP 0
	NOP 0
	NOP 0
	NOP 0
	NOP 0
	NOP 0
	NOP 0
	NOP 0
	NOP 0
	NOP 0
	NOP 0
	NOP 0
	NOP 0
	NOP 0
	NOP 0
	NOP 0
	NOP 0
	NOP 0
	NOP 0
	NOP 0
	NOP 0
	NOP 0
	NOP 0
	NOP 0
	NOP 0
	NOP 0
	NOP 0
	NOP 0
	NOP 0
	NOP 0
	NOP 0
	NOP 0
	NOP 0
	NOP 0
	NOP 0
	NOP 0
	NOP 0
	NOP 0
	NOP 0
	NOP 0
	NOP 0
	NOP 0
	NOP 0
	NOP 0
	NOP 0
	NOP 0
	NOP 0
	NOP 0
	NOP 0
	NOP 0
	NOP 0
	NOP 0
	NOP 0
	NOP 0
	NOP 0
	NOP 0
	NOP 0
	NOP 0
	NOP 0
	NOP 0
	NOP 0
	NOP 0
	NOP 0
	NOP 0
	NOP 0
	NOP 0
	NOP 0
	NOP 0
	NOP 0
	NOP 0
	NOP 0
	NOP 0
	NOP 0
	NOP 0
	NOP 0
	NOP 0
	NOP 0
	NOP 0
	NOP 0
	NOP 0
	NOP 0
	NOP 0
	NOP 0
	NOP 0
	NOP 0
	NOP 0
	NOP 0
	NOP 0
	NOP 0
	NOP 0
	NOP 0
	NOP 0
	NOP 0
	NOP 0
	NOP 0
	NOP 0
	NOP 0
	NOP 0
	NOP 0
	NOP 0
	NOP 0
	NOP 0
	NOP 0
	NOP 0
	NOP 0
	NOP 0
	NOP 0
	NOP 0
	NOP 0
	NOP 0
	NOP 0
	NOP 0
	NOP 0
	NOP 0
	NOP 0
	NOP 0
	NOP 0
	NOP 0
	NOP 0
	NOP 0
	NOP 0
	NOP 0
	NOP 0
	NOP 0
	NOP 0
	NOP 0
	NOP 0
	NOP 0
	NOP 0
	NOP 0
	NOP 0
	NOP 0
	NOP 0
	NOP 0
	NOP 0
	NOP 0
	NOP 0
	NOP 0
	NOP 0
	NOP 0
	NOP 0
	NOP 0
	NOP 0
	NOP 0
	NOP 0
	NOP 0
	NOP 0
	NOP 0
	NOP 0
	NOP 0
	NOP 0
	NOP 0
	NOP 0
	NOP 0
	NOP 0
	NOP 0
	NOP 0
	NOP 0
	NOP 0
	NOP 0
	NOP 0
	NOP 0
	NOP 0
	NOP 0
	NOP 0
	NOP 0
	NOP 0
	NOP 0
	NOP 0
	NOP 0
	NOP 0
	NOP 0
	NOP 0
	NOP 0
	NOP 0
	NOP 0
	NOP 0
	NOP 0
	NOP 0
	NOP 0
	NOP 0
	NOP 0
	NOP 0
	NOP 0
	NOP 0
	NOP 0
	NOP 0
	NOP 0
	NOP 0
	NOP 0
	NOP 0
	NOP 0
	NOP 0
	NOP 0
	NOP 0
	NOP 0
	NOP 0
	NOP 0
	NOP 0
	NOP 0
	NOP 0
	NOP 0
	NOP 0
	NOP 0
	NOP 0
	NOP 0
	NOP 0
	NOP 0
	NOP 0
	NOP 0
	NOP 0
	NOP 0
	NOP 0
	NOP 0
	NOP 0
	NOP 0
	NOP 0
	NOP 0
	NOP 0
	NOP 0
	NOP 0
	NOP 0
	NOP 0
	NOP 0
	NOP 0
	NOP 0
	NOP 0
	NOP 0
	NOP 0
	NOP 0
	NOP 0
	NOP 0
	NOP 0
	NOP 0
	NOP 0
	NOP 0
	NOP 0
	NOP 0
	NOP 0
	NOP 0
	NOP 0
	NOP 0
	NOP 0
	NOP 0
	NOP 0
	NOP 0
	NOP 0
	NOP 0
	NOP 0
	NOP 0
	NOP 0
	NOP 0
	NOP 0
	NOP 0
	NOP 0
	NOP 0
	NOP 0
	NOP 0
	NOP 0
	NOP 0
	NOP 0
	NOP 0
	NOP 0
	NOP 0
	NOP 0
	NOP 0
	NOP 0
	NOP 0
	NOP 0
	NOP 0
	NOP 0
	NOP 0
	NOP 0
	NOP 0
	NOP 0
	NOP 0
	NOP 0
	NOP 0
	NOP 0
	NOP 0
	NOP 0
	NOP 0
	NOP 0
	NOP 0
	NOP 0
	NOP 0
	NOP 0
	NOP 0
	NOP 0
	NOP 0
	NOP 0
	NOP 0
	NOP 0
	NOP 0
	NOP 0
	NOP 0
	NOP 0
	NOP 0
	NOP 0
	NOP 0
	NOP 0
	NOP 0
	NOP 0
	NOP 0
	NOP 0
	NOP 0
	NOP 0
	NOP 0
	NOP 0
	NOP 0
	NOP 0
	NOP 0
	NOP 0
	NOP 0
	NOP 0
	NOP 0
	NOP 0
	NOP 0
	NOP 0
	NOP 0
	NOP 0
	NOP 0
	NOP 0
	NOP 0
	NOP 0
	NOP 0
	NOP 0
	NOP 0
	NOP 0
	NOP 0
	NOP 0
	NOP 0
	NOP 0
	NOP 0
	NOP 0
	NOP 0
	NOP 0
	NOP 0
	NOP 0
	NOP 0
	NOP 0
	NOP 0
	NOP 0
	NOP 0
	NOP 0
	NOP 0
	NOP 0
	NOP 0
	NOP 0
	NOP 0
	NOP 0
	NOP 0
	NOP 0
	NOP 0
	NOP 0
	NOP 0
	NOP 0
	NOP 0
	NOP 0
	NOP 0
	NOP 0
	NOP 0
	NOP 0
	NOP 0
	NOP 0
	NOP 0
	NOP 0
	NOP 0
	NOP 0
	NOP 0
	NOP 0
	NOP 0
	NOP 0
	NOP 0
	NOP 0
	NOP 0
	NOP 0
	NOP 0
	NOP 0
	NOP 0
	NOP 0
	NOP 0
	NOP 0
	NOP 0
	NOP 0
	NOP 0
	NOP 0
	NOP 0
	NOP 0
	NOP 0
	NOP 0
	NOP 0
	NOP 0
	NOP 0
	NOP 0
	NOP 0
	NOP 0
	NOP 0
	NOP 0
	NOP 0
	NOP 0
	NOP 0
	NOP 0
	NOP 0
	NOP 0
	NOP 0
	NOP 0
	NOP 0
	NOP 0
	NOP 0
	NOP 0
	NOP 0
	NOP 0
	NOP 0
	NOP 0
	NOP 0
	NOP 0
	NOP 0
	NOP 0
	NOP 0
	NOP 0
	NOP 0
	NOP 0
	NOP 0
	NOP 0
	NOP 0
	NOP 0
	NOP 0
	NOP 0
	NOP 0
	NOP 0
	NOP 0
	NOP 0
	NOP 0
	NOP 0
	NOP 0
	NOP 0
	NOP 0
	NOP 0
	NOP 0
	NOP 0
	NOP 0
	NOP 0
	NOP 0
	NOP 0
	NOP 0
	NOP 0
	NOP 0
	NOP 0
	NOP 0
	NOP 0
	NOP 0
	NOP 0
	NOP 0
	NOP 0
	NOP 0
	NOP 0
	NOP 0
	NOP 0
	NOP 0
	NOP 0
	NOP 0
	NOP 0
	NOP 0
	NOP 0
	NOP 0
	NOP 0
	NOP 0
	NOP 0
	NOP 0
	NOP 0
	NOP 0
	NOP 0
	NOP 0
	NOP 0
	NOP 0
	NOP 0
	NOP 0
	NOP 0
	NOP 0
	NOP 0
	NOP 0
	NOP 0
	NOP 0
	NOP 0
	NOP 0
	NOP 0
	NOP 0
	NOP 0
	NOP 0
	NOP 0
	NOP 0
	NOP 0
	NOP 0
	NOP 0
	NOP 0
	NOP 0
	NOP 0
	NOP 0
	NOP 0
	NOP 0
	NOP 0
	NOP 0
	NOP 0
	NOP 0
	NOP 0
	NOP 0
	NOP 0
	NOP 0
	NOP 0
	NOP 0
	NOP 0
	NOP 0
	NOP 0
	NOP 0
	NOP 0
	NOP 0
	NOP 0
	NOP 0
	NOP 0
	NOP 0
	NOP 0
	NOP 0
	NOP 0
	NOP 0
	NOP 0
	NOP 0
	NOP 0
	NOP 0
	NOP 0
	NOP 0
	NOP 0
	NOP 0
	NOP 0
	NOP 0
	NOP 0
	NOP 0
	NOP 0
	NOP 0
	NOP 0
	NOP 0
	NOP 0
	NOP 0
	NOP 0
	NOP 0
	NOP 0
	NOP 0
	NOP 0
	NOP 0
	NOP 0
	NOP 0
	NOP 0
	NOP 0
	NOP 0
	NOP 0
	NOP 0
	NOP 0
	NOP 0
	NOP 0
	NOP 0
	NOP 0
	NOP 0
	NOP 0
	NOP 0
	NOP 0
	NOP 0
	NOP 0
	NOP 0
	NOP 0
	NOP 0
	NOP 0
	NOP 0
	NOP 0
	NOP 0
	NOP 0
	NOP 0
	NOP 0
	NOP 0
	NOP 0
	NOP 0
	NOP 0
	NOP 0
	NOP 0
	NOP 0
	NOP 0
	NOP 0
	NOP 0
	NOP 0
	NOP 0
	NOP 0
	NOP 0
	NOP 0
	NOP 0
	NOP 0
	NOP 0
	NOP 0
	NOP 0
	NOP 0
	NOP 0
	NOP 0
	NOP 0
	NOP 0
	NOP 0
	NOP 0
	NOP 0
	NOP 0
	NOP 0
	NOP 0
	NOP 0
	NOP 0
	NOP 0
	NOP 0
	NOP 0
	NOP 0
	NOP 0
	NOP 0
	NOP 0
	NOP 0
	NOP 0
	NOP 0
	NOP 0
	NOP 0
	NOP 0
	NOP 0
	NOP 0
	NOP 0
	NOP 0
	NOP 0
	NOP 0
	NOP 0
	NOP 0
	NOP 0
	NOP 0
	NOP 0
	NOP 0
	NOP 0
	NOP 0
	NOP 0
	NOP 0
	NOP 0
	NOP 0
	NOP 0
	NOP 0
	NOP 0
	NOP 0
	NOP 0
	NOP 0
	NOP 0
	NOP 0
	NOP 0
	NOP 0
	NOP 0
	NOP 0
	NOP 0
	NOP 0
	NOP 0
	NOP 0
	NOP 0
	NOP 0
	NOP 0
	NOP 0
	NOP 0
	NOP 0
	NOP 0
	NOP 0
	NOP 0
	NOP 0
	NOP 0
	NOP 0
	NOP 0
	NOP 0
	NOP 0
	NOP 0
	NOP 0
	NOP 0
	NOP 0
	NOP 0
	NOP 0
	NOP 0
	NOP 0
	NOP 0
	NOP 0
	NOP 0
	NOP 0
	NOP 0
	NOP 0
	NOP 0
	NOP 0
	NOP 0
	NOP 0
	NOP 0
	NOP 0
	NOP 0
	NOP 0
	NOP 0
	NOP 0
	NOP 0
	NOP 0
	NOP 0
	NOP 0
	NOP 0
	NOP 0
	NOP 0
	NOP 0
	NOP 0
	NOP 0
	NOP 0
	NOP 0
	NOP 0
	NOP 0
	NOP 0
	NOP 0
	NOP 0
	NOP 0
	NOP 0
	NOP 0
	NOP 0
	NOP 0
	NOP 0
	NOP 0
	NOP 0
	NOP 0
	NOP 0
	NOP 0
	NOP 0
	NOP 0
	NOP 0
	NOP 0
	NOP 0
	NOP 0
	NOP 0
	NOP 0
	NOP 0
	NOP 0
	NOP 0
	NOP 0
	NOP 0
	NOP 0
	NOP 0
	NOP 0
	NOP 0
	NOP 0
	NOP 0
	NOP 0
	NOP 0
	NOP 0
	NOP 0
	NOP 0
	NOP 0
	NOP 0
	NOP 0
	NOP 0
	NOP 0
	NOP 0
	NOP 0
	NOP 0
	NOP 0
	NOP 0
	NOP 0
	NOP 0
	NOP 0
	NOP 0
	NOP 0
	NOP 0
	NOP 0
	NOP 0
	NOP 0
	NOP 0
	NOP 0
	NOP 0
	NOP 0
	NOP 0
	NOP 0
	NOP 0
	NOP 0
	NOP 0
	NOP 0
	NOP 0
	NOP 0
	NOP 0
	NOP 0
	NOP 0
	NOP 0
	NOP 0
	NOP 0
	NOP 0
	NOP 0
	NOP 0
	NOP 0
	NOP 0
	NOP 0
	NOP 0
	NOP 0
	NOP 0
	NOP 0
	NOP 0
	NOP 0
	NOP 0
	NOP 0
	NOP 0
	NOP 0
	NOP 0
	NOP 0
	NOP 0
	NOP 0
	NOP 0
	NOP 0
	NOP 0
	NOP 0
	NOP 0
	NOP 0
	NOP 0
	NOP 0
	NOP 0
	NOP 0
	NOP 0
	NOP 0
	NOP 0
	NOP 0
	NOP 0
	NOP 0
	NOP 0
	NOP 0
	NOP 0
	NOP 0
	NOP 0
	NOP 0
	NOP 0
	NOP 0
	NOP 0
	NOP 0
	NOP 0
	NOP 0
	NOP 0
	NOP 0
	NOP 0
	NOP 0
	NOP 0
	NOP 0
	NOP 0
	NOP 0
	NOP 0
	NOP 0
	NOP 0
	NOP 0
	NOP 0
	NOP 0
	NOP 0
	NOP 0
	NOP 0
	NOP 0
	NOP 0
	NOP 0
	NOP 0
	NOP 0
	NOP 0
	NOP 0
	NOP 0
	NOP 0
	NOP 0
	NOP 0
	NOP 0
	NOP 0
	NOP 0
	NOP 0
	NOP 0
	NOP 0
	NOP 0
	NOP 0
	NOP 0
	NOP 0
	NOP 0
	NOP 0
	NOP 0
	NOP 0
	NOP 0
	NOP 0
	NOP 0
	NOP 0
	NOP 0
	NOP 0
	NOP 0
	NOP 0
	NOP 0
	NOP 0
	NOP 0
	NOP 0
	NOP 0
	NOP 0
	NOP 0
	NOP 0
	NOP 0
	NOP 0
	NOP 0
	NOP 0
	NOP 0
	NOP 0
	NOP 0
	NOP 0
	NOP 0
	NOP 0
	NOP 0
	NOP 0
	NOP 0
	NOP 0
	NOP 0
	NOP 0
	NOP 0
	NOP 0
	NOP 0
	NOP 0
	NOP 0
	NOP 0
	NOP 0
	NOP 0
	NOP 0
	NOP 0
	NOP 0
	NOP 0
	NOP 0
	NOP 0
	NOP 0
	NOP 0
	NOP 0
	NOP 0
	NOP 0
	NOP 0
	NOP 0
	NOP 0
	NOP 0
	NOP 0
	NOP 0
	NOP 0
	NOP 0
	NOP 0
	NOP 0
	NOP 0
	NOP 0
	NOP 0
	NOP 0
	NOP 0
	NOP 0
	NOP 0
	NOP 0
	NOP 0
	NOP 0
	NOP 0
	NOP 0
	NOP 0
	NOP 0
	NOP 0
	NOP 0
	NOP 0
	NOP 0
	NOP 0
	NOP 0
	NOP 0
	NOP 0
	NOP 0
	NOP 0
	NOP 0
	NOP 0
	NOP 0
	NOP 0
	NOP 0
	NOP 0
	NOP 0
	NOP 0
	NOP 0
	NOP 0
	NOP 0
	NOP 0
	NOP 0
	NOP 0
	NOP 0
	NOP 0
	NOP 0
	NOP 0
	NOP 0
	NOP 0
	NOP 0
	NOP 0
	NOP 0
	NOP 0
	NOP 0
	NOP 0
	NOP 0
	NOP 0
	NOP 0
	NOP 0
	NOP 0
	NOP 0
	NOP 0
	NOP 0
	NOP 0
	NOP 0
	NOP 0
	NOP 0
	NOP 0
	NOP 0
	NOP 0
	NOP 0
	NOP 0
	NOP 0
	NOP 0
	NOP 0
	NOP 0
	NOP 0
	NOP 0
	NOP 0
	NOP 0
	NOP 0
	NOP 0
	NOP 0
	NOP 0
	NOP 0
	NOP 0
	NOP 0
	NOP 0
	NOP 0
	NOP 0
	NOP 0
	NOP 0
	NOP 0
	NOP 0
	NOP 0
	NOP 0
	NOP 0
	NOP 0
	NOP 0
	NOP 0
	NOP 0
	NOP 0
	NOP 0
	NOP 0
	NOP 0
	NOP 0
	NOP 0
	NOP 0
	NOP 0
	NOP 0
	NOP 0
	NOP 0
	NOP 0
	NOP 0
	NOP 0
	NOP 0
	NOP 0
	NOP 0
	NOP 0
	NOP 0
	NOP 0
	NOP 0
	NOP 0
	NOP 0
	NOP 0
	NOP 0
	NOP 0
	NOP 0
	NOP 0
	NOP 0
	NOP 0
	NOP 0
	NOP 0
	NOP 0
	NOP 0
	NOP 0
	NOP 0
	NOP 0
	NOP 0
	NOP 0
	NOP 0
	NOP 0
	NOP 0
	NOP 0
	NOP 0
	NOP 0
	NOP 0
	NOP 0
	NOP 0
	NOP 0
	NOP 0
	NOP 0
	NOP 0
	NOP 0
	NOP 0
	NOP 0
	NOP 0
	NOP 0
	NOP 0
	NOP 0
	NOP 0
	NOP 0
	NOP 0
	NOP 0
	NOP 0
	NOP 0
	NOP 0
	NOP 0
	NOP 0
	NOP 0
	NOP 0
	NOP 0
	NOP 0
	NOP 0
	NOP 0
	NOP 0
	NOP 0
	NOP 0
	NOP 0
	NOP 0
	NOP 0
	NOP 0
	NOP 0
	NOP 0
	NOP 0
	NOP 0
	NOP 0
	NOP 0
	NOP 0
	NOP 0
	NOP 0
	NOP 0
	NOP 0
	NOP 0
	NOP 0
	NOP 0
	NOP 0
	NOP 0
	NOP 0
	NOP 0
	NOP 0
	NOP 0
	NOP 0
	NOP 0
	NOP 0
	NOP 0
	NOP 0
	NOP 0
	NOP 0
	NOP 0
	NOP 0
	NOP 0
	NOP 0
	NOP 0
	NOP 0
	NOP 0
	NOP 0
	NOP 0
	NOP 0
	NOP 0
	NOP 0
	NOP 0
	NOP 0
	NOP 0
	NOP 0
	NOP 0
	NOP 0
	NOP 0
	NOP 0
	NOP 0
	NOP 0
	NOP 0
	NOP 0
	NOP 0
	NOP 0
	NOP 0
	NOP 0
	NOP 0
	NOP 0
	NOP 0
	NOP 0
	NOP 0
	NOP 0
	NOP 0
	NOP 0
	NOP 0
	NOP 0
	NOP 0
	NOP 0
	NOP 0
	NOP 0
	NOP 0
	NOP 0
	NOP 0
	NOP 0
	NOP 0
	NOP 0
	NOP 0
	NOP 0
	NOP 0
	NOP 0
	NOP 0
	NOP 0
	NOP 0
	NOP 0
	NOP 0
	NOP 0
	NOP 0
	NOP 0
	NOP 0
	NOP 0
	NOP 0
	NOP 0
	NOP 0
	NOP 0
	NOP 0
	NOP 0
	NOP 0
	NOP 0
	NOP 0
	NOP 0
	NOP 0
	NOP 0
	NOP 0
	NOP 0
	NOP 0
	NOP 0
	NOP 0
	NOP 0
	NOP 0
	NOP 0
	NOP 0
	NOP 0
	NOP 0
	NOP 0
	NOP 0
	NOP 0
	NOP 0
	NOP 0
	NOP 0
	NOP 0
	NOP 0
	NOP 0
	NOP 0
	NOP 0
	NOP 0
	NOP 0
	NOP 0
	NOP 0
	NOP 0
	NOP 0
	NOP 0
	NOP 0
	NOP 0
	NOP 0
	NOP 0
	NOP 0
	NOP 0
	NOP 0
	NOP 0
	NOP 0
	NOP 0
	NOP 0
	NOP 0
	NOP 0
	NOP 0
	NOP 0
	NOP 0
	NOP 0
	NOP 0
	NOP 0
	NOP 0
	NOP 0
	NOP 0
	NOP 0
	NOP 0
	NOP 0
	NOP 0
	NOP 0
	NOP 0
	NOP 0
	NOP 0
	NOP 0
	NOP 0
	NOP 0
	NOP 0
	NOP 0
	NOP 0
	NOP 0
	NOP 0
	NOP 0
	NOP 0
	NOP 0
	NOP 0
	NOP 0
	NOP 0
	NOP 0
	NOP 0
	NOP 0
	NOP 0
	NOP 0
	NOP 0
	NOP 0
	NOP 0
	NOP 0
	NOP 0
	NOP 0
	NOP 0
	NOP 0
	NOP 0
	NOP 0
	NOP 0
	NOP 0
	NOP 0
	NOP 0
	NOP 0
	NOP 0
	NOP 0
	NOP 0
	NOP 0
	NOP 0
	NOP 0
	NOP 0
	NOP 0
	NOP 0
	NOP 0
	NOP 0
	NOP 0
	NOP 0
	NOP 0
	NOP 0
	NOP 0
	NOP 0
	NOP 0
	NOP 0
	NOP 0
	NOP 0
	NOP 0
	NOP 0
	NOP 0
	NOP 0
	NOP 0
	NOP 0
	NOP 0
	NOP 0
	NOP 0
	NOP 0
	NOP 0
	NOP 0
	NOP 0
	NOP 0
	NOP 0
	NOP 0
	NOP 0
	NOP 0
	NOP 0
	NOP 0
	NOP 0
	NOP 0
	NOP 0
	NOP 0
	NOP 0
	NOP 0
	NOP 0
	NOP 0
	NOP 0
	NOP 0
	NOP 0
	NOP 0
	NOP 0
	NOP 0
	NOP 0
	NOP 0
	NOP 0
	NOP 0
	NOP 0
	NOP 0
	NOP 0
	NOP 0
	NOP 0
	NOP 0
	NOP 0
	NOP 0
	NOP 0
	NOP 0
	NOP 0
	NOP 0
	NOP 0
	NOP 0
	NOP 0
	NOP 0
	NOP 0
	NOP 0
	NOP 0
	NOP 0
	NOP 0
	NOP 0
	NOP 0
	NOP 0
	NOP 0
	NOP 0
	NOP 0
	NOP 0
	NOP 0
	NOP 0
	NOP 0
	NOP 0
	NOP 0
	NOP 0
	NOP 0
	NOP 0
	NOP 0
	NOP 0
	NOP 0
	NOP 0
	NOP 0
	NOP 0
	NOP 0
	NOP 0
	NOP 0
	NOP 0
	NOP 0
	NOP 0
	NOP 0
	NOP 0
	NOP 0
	NOP 0
	NOP 0
	NOP 0
	NOP 0
	NOP 0
	NOP 0
	NOP 0
	NOP 0
	NOP 0
	NOP 0
	NOP 0
	NOP 0
	NOP 0
	NOP 0
	NOP 0
	NOP 0
	NOP 0
	NOP 0
	NOP 0
	NOP 0
	NOP 0
	NOP 0
	NOP 0
	NOP 0
	NOP 0
	NOP 0
	NOP 0
	NOP 0
	NOP 0
	NOP 0
	NOP 0
	NOP 0
	NOP 0
	NOP 0
	NOP 0
	NOP 0
	NOP 0
	NOP 0
	NOP 0
	NOP 0
	NOP 0
	NOP 0
	NOP 0
	NOP 0
	NOP 0
	NOP 0
	NOP 0
	NOP 0
	NOP 0
	NOP 0
	NOP 0
	NOP 0
	NOP 0
	NOP 0
	NOP 0
	NOP 0
	NOP 0
	NOP 0
	NOP 0
	NOP 0
	NOP 0
	NOP 0
	NOP 0
	NOP 0
	NOP 0
	NOP 0
	NOP 0
	NOP 0
	NOP 0
	NOP 0
	NOP 0
	NOP 0
	NOP 0
	NOP 0
	NOP 0
	NOP 0
	NOP 0
	NOP 0
	NOP 0
	NOP 0
	NOP 0
	NOP 0
	NOP 0
	NOP 0
	NOP 0
	NOP 0
	NOP 0
	NOP 0
	NOP 0
	NOP 0
	NOP 0
	NOP 0
	NOP 0
	NOP 0
	NOP 0
	NOP 0
	NOP 0
	NOP 0
	NOP 0
	NOP 0
	NOP 0
	NOP 0
	NOP 0
	NOP 0
	NOP 0
	NOP 0
	NOP 0
	NOP 0
	NOP 0
	NOP 0
	NOP 0
	NOP 0
	NOP 0
	NOP 0
	NOP 0
	NOP 0
	NOP 0
	NOP 0
	NOP 0
	NOP 0
	NOP 0
	NOP 0
	NOP 0
	NOP 0
	NOP 0
	NOP 0
	NOP 0
	NOP 0
	NOP 0
	NOP 0
	NOP 0
	NOP 0
	NOP 0
	NOP 0
	NOP 0
	NOP 0
	NOP 0
	NOP 0
	NOP 0
	NOP 0
	NOP 0
	NOP 0
	NOP 0
	NOP 0
	NOP 0
	NOP 0
	NOP 0
	NOP 0
	NOP 0
	NOP 0
	NOP 0
	NOP 0
	NOP 0
	NOP 0
	NOP 0
	NOP 0
	NOP 0
	NOP 0
	NOP 0
	NOP 0
	NOP 0
	NOP 0
	NOP 0
	NOP 0
	NOP 0
	NOP 0
	NOP 0
	NOP 0
	NOP 0
	NOP 0
	NOP 0
	NOP 0
	NOP 0
	NOP 0
	NOP 0
	NOP 0
	NOP 0
	NOP 0
	NOP 0
	NOP 0
	NOP 0
	NOP 0
	NOP 0
	NOP 0
	NOP 0
	NOP 0
	NOP 0
	NOP 0
	NOP 0
	NOP 0
	NOP 0
	NOP 0
	NOP 0
	NOP 0
	NOP 0
	NOP 0
	NOP 0
	NOP 0
	NOP 0
	NOP 0
	NOP 0
	NOP 0
	NOP 0
	NOP 0
	NOP 0
	NOP 0
	NOP 0
	NOP 0
	NOP 0
	NOP 0
	NOP 0
	NOP 0
	NOP 0
	NOP 0
	NOP 0
	NOP 0
	NOP 0
	NOP 0
	NOP 0
	NOP 0
	NOP 0
	NOP 0
	NOP 0
	NOP 0
	NOP 0
	NOP 0
	NOP 0
	NOP 0
	NOP 0
	NOP 0
	NOP 0
	NOP 0
	NOP 0
	NOP 0
	NOP 0
	NOP 0
	NOP 0
	NOP 0
	NOP 0
	NOP 0
	NOP 0
	NOP 0
	NOP 0
	NOP 0
	NOP 0
	NOP 0
	NOP 0
	NOP 0
	NOP 0
	NOP 0
	NOP 0
	NOP 0
	NOP 0
	NOP 0
	NOP 0
	NOP 0
	NOP 0
	NOP 0
	NOP 0
	NOP 0
	NOP 0
	NOP 0
	NOP 0
	NOP 0
	NOP 0
	NOP 0
	NOP 0
	NOP 0
	NOP 0
	NOP 0
	NOP 0
	NOP 0
	NOP 0
	NOP 0
	NOP 0
	NOP 0
	NOP 0
	NOP 0
	NOP 0
	NOP 0
	NOP 0
	NOP 0
	NOP 0
	NOP 0
	NOP 0
	NOP 0
	NOP 0
	NOP 0
	NOP 0
	NOP 0
	NOP 0
	NOP 0
	NOP 0
	NOP 0
	NOP 0
	NOP 0
	NOP 0
	NOP 0
	NOP 0
	NOP 0
	NOP 0
	NOP 0
	NOP 0
	NOP 0
	NOP 0
	NOP 0
	NOP 0
	NOP 0
	NOP 0
	NOP 0
	NOP 0
	NOP 0
	NOP 0
	NOP 0
	NOP 0
	NOP 0
	NOP 0
	NOP 0
	NOP 0
	NOP 0
	NOP 0
	NOP 0
	NOP 0
	NOP 0
	NOP 0
	NOP 0
	NOP 0
	NOP 0
	NOP 0
	NOP 0
	NOP 0
	NOP 0
	NOP 0
	NOP 0
	NOP 0
	NOP 0
	NOP 0
	NOP 0
	NOP 0
	NOP 0
	NOP 0
	NOP 0
	NOP 0
	NOP 0
	NOP 0
	NOP 0
	NOP 0
	NOP 0
	NOP 0
	NOP 0
	NOP 0
	NOP 0
	NOP 0
	NOP 0
	NOP 0
	NOP 0
	NOP 0
	NOP 0
	NOP 0
	NOP 0
	NOP 0
	NOP 0
	NOP 0
	NOP 0
	NOP 0
	NOP 0
	NOP 0
	NOP 0
	NOP 0
	NOP 0
	NOP 0
	NOP 0
	NOP 0
	NOP 0
	NOP 0
	NOP 0
	NOP 0
	NOP 0
	NOP 0
	NOP 0
	NOP 0
	NOP 0
	NOP 0
	NOP 0
	NOP 0
	NOP 0
	NOP 0
	NOP 0
	NOP 0
	NOP 0
	NOP 0
	NOP 0
	NOP 0
	NOP 0
	NOP 0
	NOP 0
	NOP 0
	NOP 0
	NOP 0
	NOP 0
	NOP 0
	NOP 0
	NOP 0
	NOP 0
	NOP 0
	NOP 0
	NOP 0
	NOP 0
	NOP 0
	NOP 0
	NOP 0
	NOP 0
	NOP 0
	NOP 0
	NOP 0
	NOP 0
	NOP 0
	NOP 0
	NOP 0
	NOP 0
	NOP 0
	NOP 0
	NOP 0
	NOP 0
	NOP 0
	NOP 0
	NOP 0
	NOP 0
	NOP 0
	NOP 0
	NOP 0
	NOP 0
	NOP 0
	NOP 0
	NOP 0
	NOP 0
	NOP 0
	NOP 0
	NOP 0
	NOP 0
	NOP 0
	NOP 0
	NOP 0
	NOP 0
	NOP 0
	NOP 0
	NOP 0
	NOP 0
	NOP 0
	NOP 0
	NOP 0
	NOP 0
	NOP 0
	NOP 0
	NOP 0
	NOP 0
	NOP 0
	NOP 0
	NOP 0
	NOP 0
	NOP 0
	NOP 0
	NOP 0
	NOP 0
	NOP 0
	NOP 0
	NOP 0
	NOP 0
	NOP 0
	NOP 0
	NOP 0
	NOP 0
	NOP 0
	NOP 0
	NOP 0
	NOP 0
	NOP 0
	NOP 0
	NOP 0
	NOP 0
	NOP 0
	NOP 0
	NOP 0
	NOP 0
	NOP 0
	NOP 0
	NOP 0
	NOP 0
	NOP 0
	NOP 0
	NOP 0
	NOP 0
	NOP 0
	NOP 0
	NOP 0
	NOP 0
	NOP 0
	NOP 0
	NOP 0
	NOP 0
	NOP 0
	NOP 0
	NOP 0
	NOP 0
	NOP 0
	NOP 0
	NOP 0
	NOP 0
	NOP 0
	NOP 0
	NOP 0
	NOP 0
	NOP 0
	NOP 0
	NOP 0
	NOP 0
	NOP 0
	NOP 0
	NOP 0
	NOP 0
	NOP 0
	NOP 0
	NOP 0
	NOP 0
	NOP 0
	NOP 0
	NOP 0
	NOP 0
	NOP 0
	NOP 0
	NOP 0
	NOP 0
	NOP 0
	NOP 0
	NOP 0
	NOP 0
	NOP 0
	NOP 0
	NOP 0
	NOP 0
	NOP 0
	NOP 0
	NOP 0
	NOP 0
	NOP 0
	NOP 0
	NOP 0
	NOP 0
	NOP 0
	NOP 0
	NOP 0
	NOP 0
	NOP 0
	NOP 0
	NOP 0
	NOP 0
	NOP 0
	NOP 0
	NOP 0
	NOP 0
	NOP 0
	NOP 0
	NOP 0
	NOP 0
	NOP 0
	NOP 0
	NOP 0
	NOP 0
	NOP 0
	NOP 0
	NOP 0
	NOP 0
	NOP 0
	NOP 0
	NOP 0
	NOP 0
	NOP 0
	NOP 0
	NOP 0
	NOP 0
	NOP 0
	NOP 0
	NOP 0
	NOP 0
	NOP 0
	NOP 0
	NOP 0
	NOP 0
	NOP 0
	NOP 0
	NOP 0
	NOP 0
	NOP 0
	NOP 0
	NOP 0
	NOP 0
	NOP 0
	NOP 0
	NOP 0
	NOP 0
	NOP 0
	NOP 0
	NOP 0
	NOP 0
	NOP 0
	NOP 0
	NOP 0
	NOP 0
	NOP 0
	NOP 0
	NOP 0
	NOP 0
	NOP 0
	NOP 0
	NOP 0
	NOP 0
	NOP 0
	NOP 0
	NOP 0
	NOP 0
	NOP 0
	NOP 0
	NOP 0
	NOP 0
	NOP 0
	NOP 0
	NOP 0
	NOP 0
	NOP 0
	NOP 0
	NOP 0
	NOP 0
	NOP 0
	NOP 0
	NOP 0
	NOP 0
	NOP 0
	NOP 0
	NOP 0
	NOP 0
	NOP 0
	NOP 0
	NOP 0
	NOP 0
	NOP 0
	NOP 0
	NOP 0
	NOP 0
	NOP 0
	NOP 0
	NOP 0
	NOP 0
	NOP 0
	NOP 0
	NOP 0
	NOP 0
	NOP 0
	NOP 0
	NOP 0
	NOP 0
	NOP 0
	NOP 0
	NOP 0
	NOP 0
	NOP 0
	NOP 0
	NOP 0
	NOP 0
	NOP 0
	NOP 0
	NOP 0
	NOP 0
	NOP 0
	NOP 0
	NOP 0
	NOP 0
	NOP 0
	NOP 0
	NOP 0
	NOP 0
	NOP 0
	NOP 0
	NOP 0
	NOP 0
	NOP 0
	NOP 0
	NOP 0
	NOP 0
	NOP 0
	NOP 0
	NOP 0
	NOP 0
	NOP 0
	NOP 0
	NOP 0
	NOP 0
	NOP 0
	NOP 0
	NOP 0
	NOP 0
	NOP 0
	NOP 0
	NOP 0
	NOP 0
	NOP 0
	NOP 0
	NOP 0
	NOP 0
	NOP 0
	NOP 0
	NOP 0
	NOP 0
	NOP 0
	NOP 0
	NOP 0
	NOP 0
	NOP 0
	NOP 0
	NOP 0
	NOP 0
	NOP 0
	NOP 0
	NOP 0
	NOP 0
	NOP 0
	NOP 0
	NOP 0
	NOP 0
	NOP 0
	NOP 0
	NOP 0
	NOP 0
	NOP 0
	NOP 0
	NOP 0
	NOP 0
	NOP 0
	NOP 0
	NOP 0
	NOP 0
	NOP 0
	NOP 0
	NOP 0
	NOP 0
	NOP 0
	NOP 0
	NOP 0
	NOP 0
	NOP 0
	NOP 0
	NOP 0
	NOP 0
	NOP 0
	NOP 0
	NOP 0
	NOP 0
	NOP 0
	NOP 0
	NOP 0
	NOP 0
	NOP 0
	NOP 0
	NOP 0
	NOP 0
	NOP 0
	NOP 0
	NOP 0
	NOP 0
	NOP 0
	NOP 0
	NOP 0
	NOP 0
	NOP 0
	NOP 0
	NOP 0
	NOP 0
	NOP 0
	NOP 0
	NOP 0
	NOP 0
	NOP 0
	NOP 0
	NOP 0
	NOP 0
	NOP 0
	NOP 0
	NOP 0
	NOP 0
	NOP 0
	NOP 0
	NOP 0
	NOP 0
	NOP 0
	NOP 0
	NOP 0
	NOP 0
	NOP 0
	NOP 0
	NOP 0
	NOP 0
	NOP 0
	NOP 0
	NOP 0
	NOP 0
	NOP 0
	NOP 0
	NOP 0
	NOP 0
	NOP 0
	NOP 0
	NOP 0
	NOP 0
	NOP 0
	NOP 0
	NOP 0
	NOP 0
	NOP 0
	NOP 0
	NOP 0
	NOP 0
	NOP 0
	NOP 0
	NOP 0
	NOP 0
	NOP 0
	NOP 0
	NOP 0
	NOP 0
	NOP 0
	NOP 0
	NOP 0
	NOP 0
	NOP 0
	NOP 0
	NOP 0
	NOP 0
	NOP 0
	NOP 0
	NOP 0
	NOP 0
	NOP 0
	NOP 0
	NOP 0
	NOP 0
	NOP 0
	NOP 0
	NOP 0
	NOP 0
	NOP 0
	NOP 0
	NOP 0
	NOP 0
	NOP 0
	NOP 0
	NOP 0
	NOP 0
	NOP 0
	NOP 0
	NOP 0
	NOP 0
	NOP 0
	NOP 0
	NOP 0
	NOP 0
	NOP 0
	NOP 0
	NOP 0
	NOP 0
	NOP 0
	NOP 0
	NOP 0
	NOP 0
	NOP 0
	NOP 0
	NOP 0
	NOP 0
	NOP 0
	NOP 0
	NOP 0
	NOP 0
	NOP 0
	NOP 0
	NOP 0
	NOP 0
	NOP 0
	NOP 0
	NOP 0
	NOP 0
	NOP 0
	NOP 0
	NOP 0
	NOP 0
	NOP 0
	NOP 0
	NOP 0
	NOP 0
	NOP 0
	NOP 0
	NOP 0
	NOP 0
	NOP 0
	NOP 0
	NOP 0
	NOP 0
	NOP 0
	NOP 0
	NOP 0
	NOP 0
	NOP 0
	NOP 0
	NOP 0
	NOP 0
	NOP 0
	NOP 0
	NOP 0
	NOP 0
	NOP 0
	NOP 0
	NOP 0
	NOP 0
	NOP 0
	NOP 0
	NOP 0
	NOP 0
	NOP 0
	NOP 0
	NOP 0
	NOP 0
	NOP 0
	NOP 0
	NOP 0
	NOP 0
	NOP 0
	NOP 0
	NOP 0
	NOP 0
	NOP 0
	NOP 0
	NOP 0
	NOP 0
	NOP 0
	NOP 0
	NOP 0
	NOP 0
	NOP 0
	NOP 0
	NOP 0
	NOP 0
	NOP 0
	NOP 0
	NOP 0
	NOP 0
	NOP 0
	NOP 0
	NOP 0
	NOP 0
	NOP 0
	NOP 0
	NOP 0
	NOP 0
	NOP 0
	NOP 0
	NOP 0
	NOP 0
	NOP 0
	NOP 0
	NOP 0
	NOP 0
	NOP 0
	NOP 0
	NOP 0
	NOP 0
	NOP 0
	NOP 0
	NOP 0
	NOP 0
	NOP 0
	NOP 0
	NOP 0
	NOP 0
	NOP 0
	NOP 0
	NOP 0
	NOP 0
	NOP 0
	NOP 0
	NOP 0
	NOP 0
	NOP 0
	NOP 0
	NOP 0
	NOP 0
	NOP 0
	NOP 0
	NOP 0
	NOP 0
	NOP 0
	NOP 0
	NOP 0
	NOP 0
	NOP 0
	NOP 0
	NOP 0
	NOP 0
	NOP 0
	NOP 0
	NOP 0
	NOP 0
	NOP 0
	NOP 0
	NOP 0
	NOP 0
	NOP 0
	NOP 0
	NOP 0
	NOP 0
	NOP 0
	NOP 0
	NOP 0
	NOP 0
	NOP 0
	NOP 0
	NOP 0
	NOP 0
	NOP 0
	NOP 0
	NOP 0
	NOP 0
	NOP 0
	NOP 0
	NOP 0
	NOP 0
	NOP 0
	NOP 0
	NOP 0
	NOP 0
	NOP 0
	NOP 0
	NOP 0
	NOP 0
	NOP 0
	NOP 0
	NOP 0
	NOP 0
	NOP 0
	NOP 0
	NOP 0
	NOP 0
	NOP 0
	NOP 0
	NOP 0
	NOP 0
	NOP 0
	NOP 0
	NOP 0
	NOP 0
	NOP 0
	NOP 0
	NOP 0
	NOP 0
	NOP 0
	NOP 0
	NOP 0
	NOP 0
	NOP 0
	NOP 0
	NOP 0
	NOP 0
	NOP 0
	NOP 0
	NOP 0
	NOP 0
	NOP 0
	NOP 0
	NOP 0
	NOP 0
	NOP 0
	NOP 0
	NOP 0
	NOP 0
	NOP 0
	NOP 0
	NOP 0
	NOP 0
	NOP 0
	NOP 0
	NOP 0
	NOP 0
	NOP 0
	NOP 0
	NOP 0
	NOP 0
	NOP 0
	NOP 0
	NOP 0
	NOP 0
	NOP 0
	NOP 0
	NOP 0
	NOP 0
	NOP 0
	NOP 0
	NOP 0
	NOP 0
	NOP 0
	NOP 0
	NOP 0
	NOP 0
	NOP 0
	NOP 0
	NOP 0
	NOP 0
	NOP 0
	NOP 0
	NOP 0
	NOP 0
	NOP 0
	NOP 0
	NOP 0
	NOP 0
	NOP 0
	NOP 0
	NOP 0
	NOP 0
	NOP 0
	NOP 0
	NOP 0
	NOP 0
	NOP 0
	NOP 0
	NOP 0
	NOP 0
	NOP 0
	NOP 0
	NOP 0
	NOP 0
	NOP 0
	NOP 0
	NOP 0
	NOP 0
	NOP 0
	NOP 0
	NOP 0
	NOP 0
	NOP 0
	NOP 0
	NOP 0
	NOP 0
	NOP 0
	NOP 0
	NOP 0
	NOP 0
	NOP 0
	NOP 0
	NOP 0
	NOP 0
	NOP 0
	NOP 0
	NOP 0
	NOP 0
	NOP 0
	NOP 0
	NOP 0
	NOP 0
	NOP 0
	NOP 0
	NOP 0
	NOP 0
	NOP 0
	NOP 0
	NOP 0
	NOP 0
	NOP 0
	NOP 0
	NOP 0
	NOP 0
	NOP 0
	NOP 0
	NOP 0
	NOP 0
	NOP 0
	NOP 0
	NOP 0
	NOP 0
	NOP 0
	NOP 0
	NOP 0
	NOP 0
	NOP 0
	NOP 0
	NOP 0
	NOP 0
	NOP 0
	NOP 0
	NOP 0
	NOP 0
	NOP 0
	NOP 0
	NOP 0
	NOP 0
	NOP 0
	NOP 0
	NOP 0
	NOP 0
	NOP 0
	NOP 0
	NOP 0
	NOP 0
	NOP 0
	NOP 0
	NOP 0
	NOP 0
	NOP 0
	NOP 0
	NOP 0
	NOP 0
	NOP 0
	NOP 0
	NOP 0
	NOP 0
	NOP 0
	NOP 0
	NOP 0
	NOP 0
	NOP 0
	NOP 0
	NOP 0
	NOP 0
	NOP 0
	NOP 0
	NOP 0
	NOP 0
	NOP 0
	NOP 0
	NOP 0
	NOP 0
	NOP 0
	NOP 0
	NOP 0
	NOP 0
	NOP 0
	NOP 0
	NOP 0
	NOP 0
	NOP 0
	NOP 0
	NOP 0
	NOP 0
	NOP 0
	NOP 0
	NOP 0
	NOP 0
	NOP 0
	NOP 0
	NOP 0
	NOP 0
	NOP 0
	NOP 0
	NOP 0
	NOP 0
	NOP 0
	NOP 0
	NOP 0
	NOP 0
	NOP 0
	NOP 0
	NOP 0
	NOP 0
	NOP 0
	NOP 0
	NOP 0
	NOP 0
	NOP 0
	NOP 0
	NOP 0
	NOP 0
	NOP 0
	NOP 0
	NOP 0
	NOP 0
	NOP 0
	NOP 0
	NOP 0
	NOP 0
	NOP 0
	NOP 0
	NOP 0
	NOP 0
	NOP 0
	NOP 0
	NOP 0
	NOP 0
	NOP 0
	NOP 0
	NOP 0
	NOP 0
	NOP 0
	NOP 0
	NOP 0
	NOP 0
	NOP 0
	NOP 0
	NOP 0
	NOP 0
	NOP 0
	NOP 0
	NOP 0
	NOP 0
	NOP 0
	NOP 0
	NOP 0
	NOP 0
	NOP 0
	NOP 0
	NOP 0
	NOP 0
	NOP 0
	NOP 0
	NOP 0
	NOP 0
	NOP 0
	NOP 0
	NOP 0
	NOP 0
	NOP 0
	NOP 0
	NOP 0
	NOP 0
	NOP 0
	NOP 0
	NOP 0
	NOP 0
	NOP 0
	NOP 0
	NOP 0
	NOP 0
	NOP 0
	NOP 0
	NOP 0
	NOP 0
	NOP 0
	NOP 0
	NOP 0
	NOP 0
	NOP 0
	NOP 0
	NOP 0
	NOP 0
	NOP 0
	NOP 0
	NOP 0
	NOP 0
	NOP 0
	NOP 0
	NOP 0
	NOP 0
	NOP 0
	NOP 0
	NOP 0
	NOP 0
	NOP 0
	NOP 0
	NOP 0
	NOP 0
	NOP 0
	NOP 0
	NOP 0
	NOP 0
	NOP 0
	NOP 0
	NOP 0
	NOP 0
	NOP 0
	NOP 0
	NOP 0
	NOP 0
	NOP 0
	NOP 0
	NOP 0
	NOP 0
	NOP 0
	NOP 0
	NOP 0
	NOP 0
	NOP 0
	NOP 0
	NOP 0
	NOP 0
	NOP 0
	NOP 0
	NOP 0
	NOP 0
	NOP 0
	NOP 0
	NOP 0
	NOP 0
	NOP 0
	NOP 0
	NOP 0
	NOP 0
	NOP 0
	NOP 0
	NOP 0
	NOP 0
	NOP 0
	NOP 0
	NOP 0
	NOP 0
	NOP 0
	NOP 0
	NOP 0
	NOP 0
	NOP 0
	NOP 0
	NOP 0
	NOP 0
	NOP 0
	NOP 0
	NOP 0
	NOP 0
	NOP 0
	NOP 0
	NOP 0
	NOP 0
	NOP 0
	NOP 0
	NOP 0
	NOP 0
	NOP 0
	NOP 0
	NOP 0
	NOP 0
	NOP 0
	NOP 0
	NOP 0
	NOP 0
	NOP 0
	NOP 0
	NOP 0
	NOP 0
	NOP 0
	NOP 0
	NOP 0
	NOP 0
	NOP 0
	NOP 0
	NOP 0
	NOP 0
	NOP 0
	NOP 0
	NOP 0
	NOP 0
	NOP 0
	NOP 0
	NOP 0
	NOP 0
	NOP 0
	NOP 0
	NOP 0
	NOP 0
	NOP 0
	NOP 0
	NOP 0
	NOP 0
	NOP 0
	NOP 0
	NOP 0
	NOP 0
	NOP 0
	NOP 0
	NOP 0
	NOP 0
	NOP 0
	NOP 0
	NOP 0
	NOP 0
	NOP 0
	NOP 0
	NOP 0
	NOP 0
	NOP 0
	NOP 0
	NOP 0
	NOP 0
	NOP 0
	NOP 0
	NOP 0
	NOP 0
	NOP 0
	NOP 0
	NOP 0
	NOP 0
	NOP 0
	NOP 0
	NOP 0
	NOP 0
	NOP 0
	NOP 0
	NOP 0
	NOP 0
	NOP 0
	NOP 0
	NOP 0
	NOP 0
	NOP 0
	NOP 0
	NOP 0
	NOP 0
	NOP 0
	NOP 0
	NOP 0
	NOP 0
	NOP 0
	NOP 0
	NOP 0
	NOP 0
	NOP 0
	NOP 0
	NOP 0
	NOP 0
	NOP 0
	NOP 0
	NOP 0
	NOP 0
	NOP 0
	NOP 0
	NOP 0
	NOP 0
	NOP 0
	NOP 0
	NOP 0
	NOP 0
	NOP 0
	NOP 0
	NOP 0
	NOP 0
	NOP 0
	NOP 0
	NOP 0
	NOP 0
	NOP 0
	NOP 0
	NOP 0
	NOP 0
	NOP 0
	NOP 0
	NOP 0
	NOP 0
	NOP 0
	NOP 0
	NOP 0
	NOP 0
	NOP 0
	NOP 0
	NOP 0
	NOP 0
	NOP 0
	NOP 0
	NOP 0
	NOP 0
	NOP 0
	NOP 0
	NOP 0
	NOP 0
	NOP 0
	NOP 0
	NOP 0
	NOP 0
	NOP 0
	NOP 0
	NOP 0
	NOP 0
	NOP 0
	NOP 0
	NOP 0
	NOP 0
	NOP 0
	NOP 0
	NOP 0
	NOP 0
	NOP 0
	NOP 0
	NOP 0
	NOP 0
	NOP 0
	NOP 0
	NOP 0
	NOP 0
	NOP 0
	NOP 0
	NOP 0
	NOP 0
	NOP 0
	NOP 0
	NOP 0
	NOP 0
	NOP 0
	NOP 0
	NOP 0
	NOP 0
	NOP 0
	NOP 0
	NOP 0
	NOP 0
	NOP 0
	NOP 0
	NOP 0
	NOP 0
	NOP 0
	NOP 0
	NOP 0
	NOP 0
	NOP 0
	NOP 0
	NOP 0
	NOP 0
	NOP 0
	NOP 0
	NOP 0
	NOP 0
	NOP 0
	NOP 0
	NOP 0
	NOP 0
	NOP 0
	NOP 0
	NOP 0
	NOP 0
	NOP 0
	NOP 0
	NOP 0
	NOP 0
	NOP 0
	NOP 0
	NOP 0
	NOP 0
	NOP 0
	NOP 0
	NOP 0
	NOP 0
	NOP 0
	NOP 0
	NOP 0
	NOP 0
	NOP 0
	NOP 0
	NOP 0
	NOP 0
	NOP 0
	NOP 0
	NOP 0
	NOP 0
	NOP 0
	NOP 0
	NOP 0
	NOP 0
	NOP 0
	NOP 0
	NOP 0
	NOP 0
	NOP 0
	NOP 0
	NOP 0
	NOP 0
	NOP 0
	NOP 0
	NOP 0
	NOP 0
	NOP 0
	NOP 0
	NOP 0
	NOP 0
	NOP 0
	NOP 0
	NOP 0
	NOP 0
	NOP 0
	NOP 0
	NOP 0
	NOP 0
	NOP 0
	NOP 0
	NOP 0
	NOP 0
	NOP 0
	NOP 0
	NOP 0
	NOP 0
	NOP 0
	NOP 0
	NOP 0
	NOP 0
	NOP 0
	NOP 0
	NOP 0
	NOP 0
	NOP 0
	NOP 0
	NOP 0
	NOP 0
	NOP 0
	NOP 0
	NOP 0
	NOP 0
	NOP 0
	NOP 0
	NOP 0
	NOP 0
	NOP 0
	NOP 0
	NOP 0
	NOP 0
	NOP 0
	NOP 0
	NOP 0
	NOP 0
	NOP 0
	NOP 0
	NOP 0
	NOP 0
	NOP 0
	NOP 0
	NOP 0
	NOP 0
	NOP 0
	NOP 0
	NOP 0
	NOP 0
	NOP 0
	NOP 0
	NOP 0
	NOP 0
	NOP 0
	NOP 0
	NOP 0
	NOP 0
	NOP 0
	NOP 0
	NOP 0
	NOP 0
	NOP 0
	NOP 0
	NOP 0
	NOP 0
	NOP 0
	NOP 0
	NOP 0
	NOP 0
	NOP 0
	NOP 0
	NOP 0
	NOP 0
	NOP 0
	NOP 0
	NOP 0
	NOP 0
	NOP 0
	NOP 0
	NOP 0
	NOP 0
	NOP 0
	NOP 0
	NOP 0
	NOP 0
	NOP 0
	NOP 0
	NOP 0
	NOP 0
	NOP 0
	NOP 0
	NOP 0
	NOP 0
	NOP 0
	NOP 0
	NOP 0
	NOP 0
	NOP 0
	NOP 0
	NOP 0
	NOP 0
	NOP 0
	NOP 0
	NOP 0
	NOP 0
	NOP 0
	NOP 0
	NOP 0
	NOP 0
	NOP 0
	NOP 0
	NOP 0
	NOP 0
	NOP 0
	NOP 0
	NOP 0
	NOP 0
	NOP 0
	NOP 0
	NOP 0
	NOP 0
	NOP 0
	NOP 0
	NOP 0
	NOP 0
	NOP 0
	NOP 0
	NOP 0
	NOP 0
	NOP 0
	NOP 0
	NOP 0
	NOP 0
	NOP 0
	NOP 0
	NOP 0
	NOP 0
	NOP 0
	NOP 0
	NOP 0
	NOP 0
	NOP 0
	NOP 0
	NOP 0
	NOP 0
	NOP 0
	NOP 0
	NOP 0
	NOP 0
	NOP 0
	NOP 0
	NOP 0
	NOP 0
	NOP 0
	NOP 0
	NOP 0
	NOP 0
	NOP 0
	NOP 0
	NOP 0
	NOP 0
	NOP 0
	NOP 0
	NOP 0
	NOP 0
	NOP 0
	NOP 0
	NOP 0
	NOP 0
	NOP 0
	NOP 0
	NOP 0
	NOP 0
	NOP 0
	NOP 0
	NOP 0
	NOP 0
	NOP 0
	NOP 0
	NOP 0
	NOP 0
	NOP 0
	NOP 0
	NOP 0
	NOP 0
	NOP 0
	NOP 0
	NOP 0
	NOP 0
	NOP 0
	NOP 0
	NOP 0
	NOP 0
	NOP 0
	NOP 0
	NOP 0
	NOP 0
	NOP 0
	NOP 0
	NOP 0
	NOP 0
	NOP 0
	NOP 0
	NOP 0
	NOP 0
	NOP 0
	NOP 0
	NOP 0
	NOP 0
	NOP 0
	NOP 0
	NOP 0
	NOP 0
	NOP 0
	NOP 0
	NOP 0
	NOP 0
	NOP 0
	NOP 0
	NOP 0
	NOP 0
	NOP 0
	NOP 0
	NOP 0
	NOP 0
	NOP 0
	NOP 0
	NOP 0
	NOP 0
	NOP 0
	NOP 0
	NOP 0
	NOP 0
	NOP 0
	NOP 0
	NOP 0
	NOP 0
	NOP 0
	NOP 0
	NOP 0
	NOP 0
	NOP 0
	NOP 0
	NOP 0
	NOP 0
	NOP 0
	NOP 0
	NOP 0
	NOP 0
	NOP 0
	NOP 0
	NOP 0
	NOP 0
	NOP 0
	NOP 0
	NOP 0
	NOP 0
	NOP 0
	NOP 0
	NOP 0
	NOP 0
	NOP 0
	NOP 0
	NOP 0
	NOP 0
	NOP 0
	NOP 0
	NOP 0
	NOP 0
	NOP 0
	NOP 0
	NOP 0
	NOP 0
	NOP 0
	NOP 0
	NOP 0
	NOP 0
	NOP 0
	NOP 0
	NOP 0
	NOP 0
	NOP 0
	NOP 0
	NOP 0
	NOP 0
	NOP 0
	NOP 0
	NOP 0
	NOP 0
	NOP 0
	NOP 0
	NOP 0
	NOP 0
	NOP 0
	NOP 0
	NOP 0
	NOP 0
	NOP 0
	NOP 0
	NOP 0
	NOP 0
	NOP 0
	NOP 0
	NOP 0
	NOP 0
	NOP 0
	NOP 0
	NOP 0
	NOP 0
	NOP 0
	NOP 0
	NOP 0
	NOP 0
	NOP 0
	NOP 0
	NOP 0
	NOP 0
	NOP 0
	NOP 0
	NOP 0
	NOP 0
	NOP 0
	NOP 0
	NOP 0
	NOP 0
	NOP 0
	NOP 0
	NOP 0
	NOP 0
	NOP 0
	NOP 0
	NOP 0
	NOP 0
	NOP 0
	NOP 0
	NOP 0
	NOP 0
	NOP 0
	NOP 0
	NOP 0
	NOP 0
	NOP 0
	NOP 0
	NOP 0
	NOP 0
	NOP 0
	NOP 0
	NOP 0
	NOP 0
	NOP 0
	NOP 0
	NOP 0
	NOP 0
	NOP 0
	NOP 0
	NOP 0
	NOP 0
	NOP 0
	NOP 0
	NOP 0
	NOP 0
	NOP 0
	NOP 0
	NOP 0
	NOP 0
	NOP 0
	NOP 0
	NOP 0
	NOP 0
	NOP 0
	NOP 0
	NOP 0
	NOP 0
	NOP 0
	NOP 0
	NOP 0
	NOP 0
	NOP 0
	NOP 0
	NOP 0
	NOP 0
	NOP 0
	NOP 0
	NOP 0
	NOP 0
	NOP 0
	NOP 0
	NOP 0
	NOP 0
	NOP 0
	NOP 0
	NOP 0
	NOP 0
	NOP 0
	NOP 0
	NOP 0
	NOP 0
	NOP 0
	NOP 0
	NOP 0
	NOP 0
	NOP 0
	NOP 0
	NOP 0
	NOP 0
	NOP 0
	NOP 0
	NOP 0
	NOP 0
	NOP 0
	NOP 0
	NOP 0
	NOP 0
	NOP 0
	NOP 0
	NOP 0
	NOP 0
	NOP 0
	NOP 0
	NOP 0
	NOP 0
	NOP 0
	NOP 0
	NOP 0
	NOP 0
	NOP 0
	NOP 0
	NOP 0
	NOP 0
	NOP 0
	NOP 0
	NOP 0
	NOP 0
	NOP 0
	NOP 0
	NOP 0
